// TIA Portal V17 export
// export: Created 2025-07-01T14:26:11.8460779Z, ExportSetting WithDefaults, DisplayName Totally Integrated Automation Portal, DisplayVersion V17 Update 8, DisplayName TIA Portal Openness, DisplayVersion V17 Update 8, DisplayName TIA Portal Version Control Interface, DisplayVersion V17, DisplayName SINAMICS Startdrive Advanced, DisplayVersion V17 SP2, DisplayName SINAMICS Startdrive G110M, G120, G120C, G120D, G120P, G115D, DisplayVersion V17 SP2, DisplayName SINAMICS Startdrive G130, G150, S120, S150, SINAMICS MV, S210, DisplayVersion V17 SP2, DisplayName STEP 7 Professional, DisplayVersion V17 Update 8, DisplayName SINUMERIK ONE STEP 7 Toolbox, DisplayVersion V17 Update 12, DisplayName SINUMERIK ONE PLC Basic Program Plus, DisplayVersion V17 Update 12, DisplayName SINUMERIK 840D sl STEP 7 Toolbox, DisplayVersion V17 Update 12, DisplayName STEP 7 Safety, DisplayVersion V17 Update 6, DisplayName WinCC Advanced, DisplayVersion V17 Update 8
FUNCTION "FC16013_METHOD_CALLS_U2_STA2_MEAS" : Void   // FC16013, LAD
{ S7_Optimized_Access := 'FALSE' }
VERSION : 0.1
// STATUS VALUES:
// 0 = IDLE
// 1 = CALIBRATING
// 2 = ANALYZING 
// -1 = ERROR
// stored: AutoNumber false, IsIECCheckEnabled false, SetENOAutomatically false, UDAEnableTagReadback false
   VAR_TEMP
      AUX_WSTRING_PART_ID_STA2 : WString;
      AUX_WCHARS : Array[0..63] of WChar;
      index : Int;
      ALARM_AUX : Bool;
      STATUS_BLKMOV : Int;   // STATUS BLKMOV
      ZERO : Int;
   END_VAR
   VAR CONSTANT
      VERSIONS_MAJOR : UInt := 2;
      VERSIONS_MINOR : UInt;
      FC_NUMBER : DInt := 16013;
   END_VAR
   VAR_TEMP   // added for the SCL form of the ladder/FBD networks
      _w1 : Bool;
      _w2 : Bool;
      _w3 : Bool;
      _w4 : Bool;
   END_VAR
BEGIN

REGION Network 1: ZERO
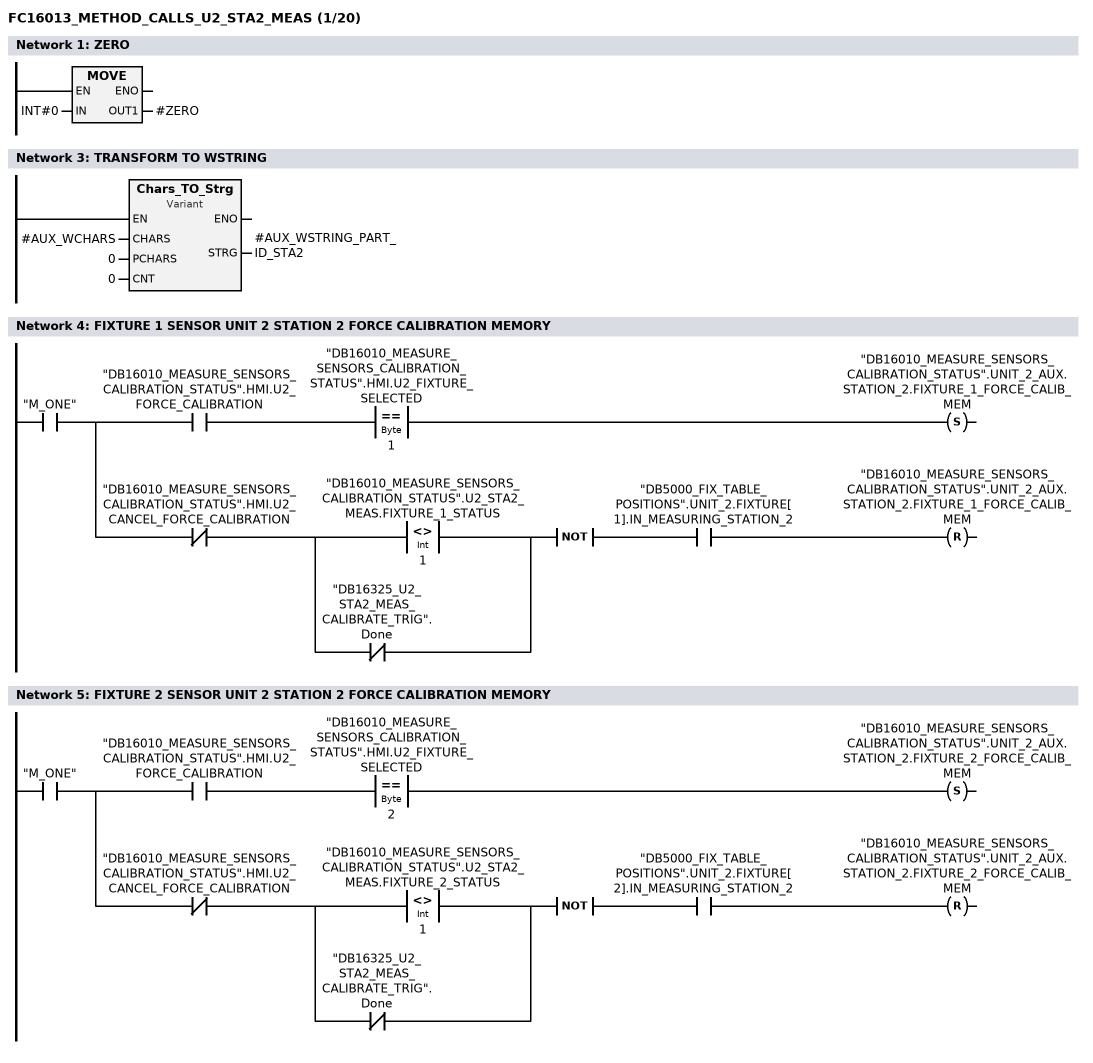
   RUNG wire#powerrail
      { S7_GenerateENO := "TRUE" } Move(in := INT#0, out1 => #ZERO)
   END_RUNG
   // the same network as SCL:
   #ZERO := INT#0;
END_REGION

REGION Network 2 (SCL): TRANSFORM TO WCHARS
   FOR #index := 0 TO 63 DO
       #AUX_WCHARS[#index] := CHAR_TO_WCHAR("DB8000_PART_STATUS".UNIT_2.STATION_2.PART_A.PART_ID[#index]);
   END_FOR;
END_REGION

REGION Network 3: TRANSFORM TO WSTRING
   RUNG wire#powerrail
      { S7_Templates := "[ptr_type := Variant, str_type := WString]" } Chars_TO_Strg(Chars := #AUX_WCHARS, pChars := 0, Cnt := 0, Strg => #AUX_WSTRING_PART_ID_STA2)
   END_RUNG
   // the same network as SCL:
   Chars_TO_Strg(Chars := #AUX_WCHARS, pChars := 0, Cnt := 0, Strg => #AUX_WSTRING_PART_ID_STA2);
END_REGION

REGION Network 4: FIXTURE 1 SENSOR UNIT 2 STATION 2 FORCE CALIBRATION MEMORY
   RUNG wire#powerrail
      Contact( "M_ONE" )
      wire#w1
      Contact( "DB16010_MEASURE_SENSORS_CALIBRATION_STATUS".HMI.U2_FORCE_CALIBRATION )
      { S7_Templates := "SrcType := Byte" } EQ_Contact(in1 := "DB16010_MEASURE_SENSORS_CALIBRATION_STATUS".HMI.U2_FIXTURE_SELECTED, in2 := 1)
      S_Coil( "DB16010_MEASURE_SENSORS_CALIBRATION_STATUS".UNIT_2_AUX.STATION_2.FIXTURE_1_FORCE_CALIB_MEM )
   END_RUNG
   RUNG wire#w1
      I_Contact( "DB16010_MEASURE_SENSORS_CALIBRATION_STATUS".HMI.U2_CANCEL_FORCE_CALIBRATION )
      wire#w2
      { S7_Templates := "SrcType := Int" } NE_Contact(in1 := "DB16010_MEASURE_SENSORS_CALIBRATION_STATUS".U2_STA2_MEAS.FIXTURE_1_STATUS, in2 := 1)
      wire#w3
      Not()
      Contact( "DB5000_FIX_TABLE_POSITIONS".UNIT_2.FIXTURE[1].IN_MEASURING_STATION_2 )
      R_Coil( "DB16010_MEASURE_SENSORS_CALIBRATION_STATUS".UNIT_2_AUX.STATION_2.FIXTURE_1_FORCE_CALIB_MEM )
   END_RUNG
   RUNG wire#w2
      I_Contact( "DB16325_U2_STA2_MEAS_CALIBRATE_TRIG".Done )
   END_RUNG wire#w3
   // the same network as SCL:
   IF "M_ONE" AND "DB16010_MEASURE_SENSORS_CALIBRATION_STATUS".HMI.U2_FORCE_CALIBRATION AND ("DB16010_MEASURE_SENSORS_CALIBRATION_STATUS".HMI.U2_FIXTURE_SELECTED = 1) THEN
       "DB16010_MEASURE_SENSORS_CALIBRATION_STATUS".UNIT_2_AUX.STATION_2.FIXTURE_1_FORCE_CALIB_MEM := TRUE;
   END_IF;
   IF NOT ("M_ONE" AND NOT "DB16010_MEASURE_SENSORS_CALIBRATION_STATUS".HMI.U2_CANCEL_FORCE_CALIBRATION AND (("DB16010_MEASURE_SENSORS_CALIBRATION_STATUS".U2_STA2_MEAS.FIXTURE_1_STATUS <> 1) OR NOT "DB16325_U2_STA2_MEAS_CALIBRATE_TRIG".Done)) AND "DB5000_FIX_TABLE_POSITIONS".UNIT_2.FIXTURE[1].IN_MEASURING_STATION_2 THEN
       "DB16010_MEASURE_SENSORS_CALIBRATION_STATUS".UNIT_2_AUX.STATION_2.FIXTURE_1_FORCE_CALIB_MEM := FALSE;
   END_IF;
END_REGION

REGION Network 5: FIXTURE 2 SENSOR UNIT 2 STATION 2 FORCE CALIBRATION MEMORY
   RUNG wire#powerrail
      Contact( "M_ONE" )
      wire#w1
      Contact( "DB16010_MEASURE_SENSORS_CALIBRATION_STATUS".HMI.U2_FORCE_CALIBRATION )
      { S7_Templates := "SrcType := Byte" } EQ_Contact(in1 := "DB16010_MEASURE_SENSORS_CALIBRATION_STATUS".HMI.U2_FIXTURE_SELECTED, in2 := 2)
      S_Coil( "DB16010_MEASURE_SENSORS_CALIBRATION_STATUS".UNIT_2_AUX.STATION_2.FIXTURE_2_FORCE_CALIB_MEM )
   END_RUNG
   RUNG wire#w1
      I_Contact( "DB16010_MEASURE_SENSORS_CALIBRATION_STATUS".HMI.U2_CANCEL_FORCE_CALIBRATION )
      wire#w2
      { S7_Templates := "SrcType := Int" } NE_Contact(in1 := "DB16010_MEASURE_SENSORS_CALIBRATION_STATUS".U2_STA2_MEAS.FIXTURE_2_STATUS, in2 := 1)
      wire#w3
      Not()
      Contact( "DB5000_FIX_TABLE_POSITIONS".UNIT_2.FIXTURE[2].IN_MEASURING_STATION_2 )
      R_Coil( "DB16010_MEASURE_SENSORS_CALIBRATION_STATUS".UNIT_2_AUX.STATION_2.FIXTURE_2_FORCE_CALIB_MEM )
   END_RUNG
   RUNG wire#w2
      I_Contact( "DB16325_U2_STA2_MEAS_CALIBRATE_TRIG".Done )
   END_RUNG wire#w3
   // the same network as SCL:
   IF "M_ONE" AND "DB16010_MEASURE_SENSORS_CALIBRATION_STATUS".HMI.U2_FORCE_CALIBRATION AND ("DB16010_MEASURE_SENSORS_CALIBRATION_STATUS".HMI.U2_FIXTURE_SELECTED = 2) THEN
       "DB16010_MEASURE_SENSORS_CALIBRATION_STATUS".UNIT_2_AUX.STATION_2.FIXTURE_2_FORCE_CALIB_MEM := TRUE;
   END_IF;
   IF NOT ("M_ONE" AND NOT "DB16010_MEASURE_SENSORS_CALIBRATION_STATUS".HMI.U2_CANCEL_FORCE_CALIBRATION AND (("DB16010_MEASURE_SENSORS_CALIBRATION_STATUS".U2_STA2_MEAS.FIXTURE_2_STATUS <> 1) OR NOT "DB16325_U2_STA2_MEAS_CALIBRATE_TRIG".Done)) AND "DB5000_FIX_TABLE_POSITIONS".UNIT_2.FIXTURE[2].IN_MEASURING_STATION_2 THEN
       "DB16010_MEASURE_SENSORS_CALIBRATION_STATUS".UNIT_2_AUX.STATION_2.FIXTURE_2_FORCE_CALIB_MEM := FALSE;
   END_IF;
END_REGION

REGION Network 6: FIXTURE 3 SENSOR UNIT 2 STATION 2 FORCE CALIBRATION MEMORY
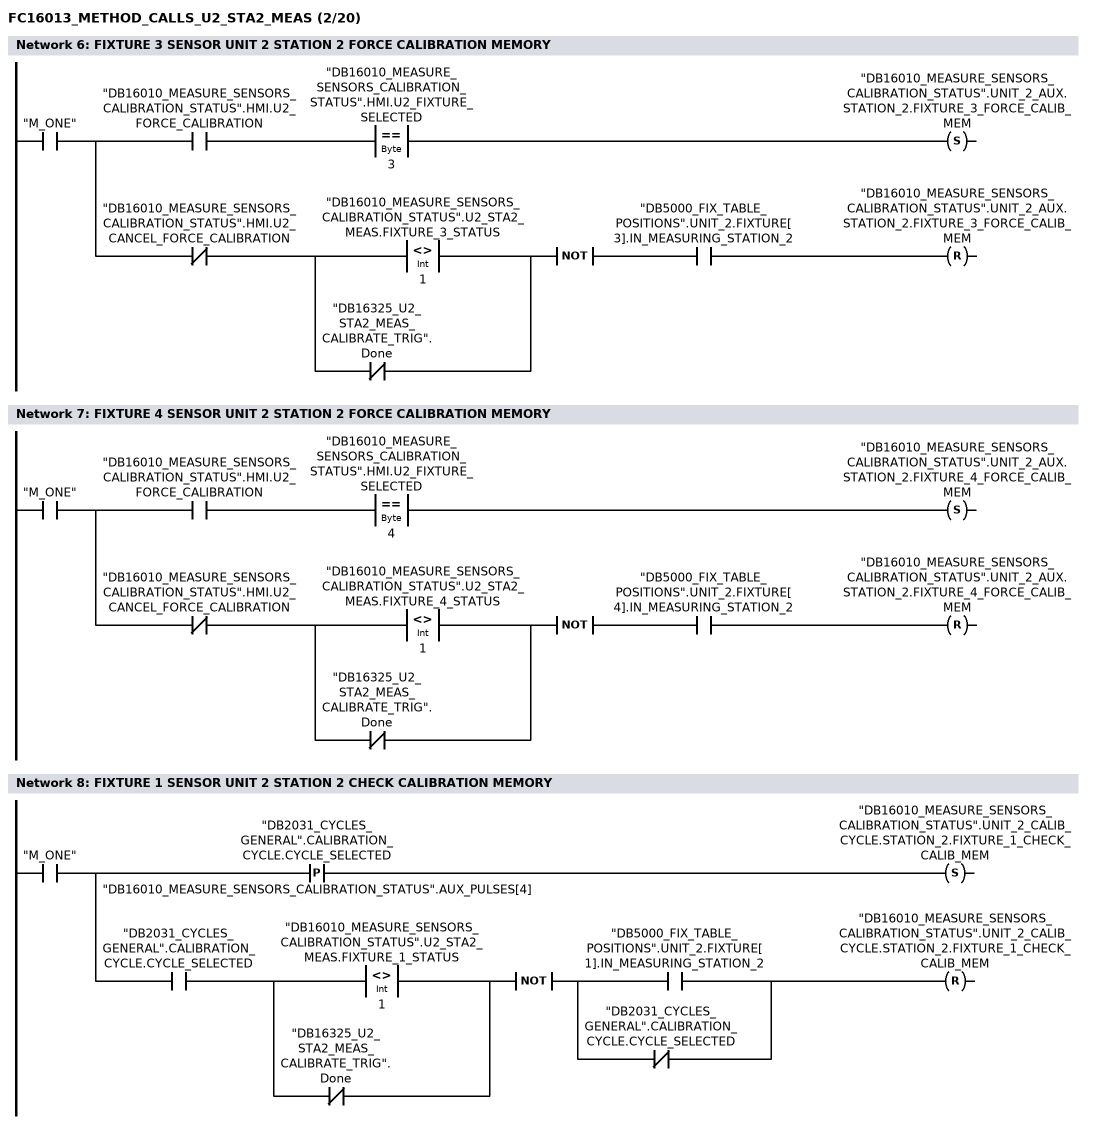
   RUNG wire#powerrail
      Contact( "M_ONE" )
      wire#w1
      Contact( "DB16010_MEASURE_SENSORS_CALIBRATION_STATUS".HMI.U2_FORCE_CALIBRATION )
      { S7_Templates := "SrcType := Byte" } EQ_Contact(in1 := "DB16010_MEASURE_SENSORS_CALIBRATION_STATUS".HMI.U2_FIXTURE_SELECTED, in2 := 3)
      S_Coil( "DB16010_MEASURE_SENSORS_CALIBRATION_STATUS".UNIT_2_AUX.STATION_2.FIXTURE_3_FORCE_CALIB_MEM )
   END_RUNG
   RUNG wire#w1
      I_Contact( "DB16010_MEASURE_SENSORS_CALIBRATION_STATUS".HMI.U2_CANCEL_FORCE_CALIBRATION )
      wire#w2
      { S7_Templates := "SrcType := Int" } NE_Contact(in1 := "DB16010_MEASURE_SENSORS_CALIBRATION_STATUS".U2_STA2_MEAS.FIXTURE_3_STATUS, in2 := 1)
      wire#w3
      Not()
      Contact( "DB5000_FIX_TABLE_POSITIONS".UNIT_2.FIXTURE[3].IN_MEASURING_STATION_2 )
      R_Coil( "DB16010_MEASURE_SENSORS_CALIBRATION_STATUS".UNIT_2_AUX.STATION_2.FIXTURE_3_FORCE_CALIB_MEM )
   END_RUNG
   RUNG wire#w2
      I_Contact( "DB16325_U2_STA2_MEAS_CALIBRATE_TRIG".Done )
   END_RUNG wire#w3
   // the same network as SCL:
   IF "M_ONE" AND "DB16010_MEASURE_SENSORS_CALIBRATION_STATUS".HMI.U2_FORCE_CALIBRATION AND ("DB16010_MEASURE_SENSORS_CALIBRATION_STATUS".HMI.U2_FIXTURE_SELECTED = 3) THEN
       "DB16010_MEASURE_SENSORS_CALIBRATION_STATUS".UNIT_2_AUX.STATION_2.FIXTURE_3_FORCE_CALIB_MEM := TRUE;
   END_IF;
   IF NOT ("M_ONE" AND NOT "DB16010_MEASURE_SENSORS_CALIBRATION_STATUS".HMI.U2_CANCEL_FORCE_CALIBRATION AND (("DB16010_MEASURE_SENSORS_CALIBRATION_STATUS".U2_STA2_MEAS.FIXTURE_3_STATUS <> 1) OR NOT "DB16325_U2_STA2_MEAS_CALIBRATE_TRIG".Done)) AND "DB5000_FIX_TABLE_POSITIONS".UNIT_2.FIXTURE[3].IN_MEASURING_STATION_2 THEN
       "DB16010_MEASURE_SENSORS_CALIBRATION_STATUS".UNIT_2_AUX.STATION_2.FIXTURE_3_FORCE_CALIB_MEM := FALSE;
   END_IF;
END_REGION

REGION Network 7: FIXTURE 4 SENSOR UNIT 2 STATION 2 FORCE CALIBRATION MEMORY
   RUNG wire#powerrail
      Contact( "M_ONE" )
      wire#w1
      Contact( "DB16010_MEASURE_SENSORS_CALIBRATION_STATUS".HMI.U2_FORCE_CALIBRATION )
      { S7_Templates := "SrcType := Byte" } EQ_Contact(in1 := "DB16010_MEASURE_SENSORS_CALIBRATION_STATUS".HMI.U2_FIXTURE_SELECTED, in2 := 4)
      S_Coil( "DB16010_MEASURE_SENSORS_CALIBRATION_STATUS".UNIT_2_AUX.STATION_2.FIXTURE_4_FORCE_CALIB_MEM )
   END_RUNG
   RUNG wire#w1
      I_Contact( "DB16010_MEASURE_SENSORS_CALIBRATION_STATUS".HMI.U2_CANCEL_FORCE_CALIBRATION )
      wire#w2
      { S7_Templates := "SrcType := Int" } NE_Contact(in1 := "DB16010_MEASURE_SENSORS_CALIBRATION_STATUS".U2_STA2_MEAS.FIXTURE_4_STATUS, in2 := 1)
      wire#w3
      Not()
      Contact( "DB5000_FIX_TABLE_POSITIONS".UNIT_2.FIXTURE[4].IN_MEASURING_STATION_2 )
      R_Coil( "DB16010_MEASURE_SENSORS_CALIBRATION_STATUS".UNIT_2_AUX.STATION_2.FIXTURE_4_FORCE_CALIB_MEM )
   END_RUNG
   RUNG wire#w2
      I_Contact( "DB16325_U2_STA2_MEAS_CALIBRATE_TRIG".Done )
   END_RUNG wire#w3
   // the same network as SCL:
   IF "M_ONE" AND "DB16010_MEASURE_SENSORS_CALIBRATION_STATUS".HMI.U2_FORCE_CALIBRATION AND ("DB16010_MEASURE_SENSORS_CALIBRATION_STATUS".HMI.U2_FIXTURE_SELECTED = 4) THEN
       "DB16010_MEASURE_SENSORS_CALIBRATION_STATUS".UNIT_2_AUX.STATION_2.FIXTURE_4_FORCE_CALIB_MEM := TRUE;
   END_IF;
   IF NOT ("M_ONE" AND NOT "DB16010_MEASURE_SENSORS_CALIBRATION_STATUS".HMI.U2_CANCEL_FORCE_CALIBRATION AND (("DB16010_MEASURE_SENSORS_CALIBRATION_STATUS".U2_STA2_MEAS.FIXTURE_4_STATUS <> 1) OR NOT "DB16325_U2_STA2_MEAS_CALIBRATE_TRIG".Done)) AND "DB5000_FIX_TABLE_POSITIONS".UNIT_2.FIXTURE[4].IN_MEASURING_STATION_2 THEN
       "DB16010_MEASURE_SENSORS_CALIBRATION_STATUS".UNIT_2_AUX.STATION_2.FIXTURE_4_FORCE_CALIB_MEM := FALSE;
   END_IF;
END_REGION

REGION Network 8: FIXTURE 1 SENSOR UNIT 2 STATION 2 CHECK CALIBRATION MEMORY
   RUNG wire#powerrail
      Contact( "M_ONE" )
      wire#w1
      P_Contact(operand := "DB2031_CYCLES_GENERAL".CALIBRATION_CYCLE.CYCLE_SELECTED, bit := "DB16010_MEASURE_SENSORS_CALIBRATION_STATUS".AUX_PULSES[4])
      S_Coil( "DB16010_MEASURE_SENSORS_CALIBRATION_STATUS".UNIT_2_CALIB_CYCLE.STATION_2.FIXTURE_1_CHECK_CALIB_MEM )
   END_RUNG
   RUNG wire#w1
      Contact( "DB2031_CYCLES_GENERAL".CALIBRATION_CYCLE.CYCLE_SELECTED )
      wire#w2
      { S7_Templates := "SrcType := Int" } NE_Contact(in1 := "DB16010_MEASURE_SENSORS_CALIBRATION_STATUS".U2_STA2_MEAS.FIXTURE_1_STATUS, in2 := 1)
      wire#w3
      Not()
      wire#w4
      Contact( "DB5000_FIX_TABLE_POSITIONS".UNIT_2.FIXTURE[1].IN_MEASURING_STATION_2 )
      wire#w5
      R_Coil( "DB16010_MEASURE_SENSORS_CALIBRATION_STATUS".UNIT_2_CALIB_CYCLE.STATION_2.FIXTURE_1_CHECK_CALIB_MEM )
   END_RUNG
   RUNG wire#w2
      I_Contact( "DB16325_U2_STA2_MEAS_CALIBRATE_TRIG".Done )
   END_RUNG wire#w3
   RUNG wire#w4
      I_Contact( "DB2031_CYCLES_GENERAL".CALIBRATION_CYCLE.CYCLE_SELECTED )
   END_RUNG wire#w5
   // the same network as SCL:
   #_w1 := "M_ONE" AND "DB2031_CYCLES_GENERAL".CALIBRATION_CYCLE.CYCLE_SELECTED AND NOT "DB16010_MEASURE_SENSORS_CALIBRATION_STATUS".AUX_PULSES[4];   // rising edge of "DB2031_CYCLES_GENERAL".CALIBRATION_CYCLE.CYCLE_SELECTED
   "DB16010_MEASURE_SENSORS_CALIBRATION_STATUS".AUX_PULSES[4] := "DB2031_CYCLES_GENERAL".CALIBRATION_CYCLE.CYCLE_SELECTED;
   IF #_w1 THEN
       "DB16010_MEASURE_SENSORS_CALIBRATION_STATUS".UNIT_2_CALIB_CYCLE.STATION_2.FIXTURE_1_CHECK_CALIB_MEM := TRUE;
   END_IF;
   IF NOT ("M_ONE" AND "DB2031_CYCLES_GENERAL".CALIBRATION_CYCLE.CYCLE_SELECTED AND (("DB16010_MEASURE_SENSORS_CALIBRATION_STATUS".U2_STA2_MEAS.FIXTURE_1_STATUS <> 1) OR NOT "DB16325_U2_STA2_MEAS_CALIBRATE_TRIG".Done)) AND ("DB5000_FIX_TABLE_POSITIONS".UNIT_2.FIXTURE[1].IN_MEASURING_STATION_2 OR NOT "DB2031_CYCLES_GENERAL".CALIBRATION_CYCLE.CYCLE_SELECTED) THEN
       "DB16010_MEASURE_SENSORS_CALIBRATION_STATUS".UNIT_2_CALIB_CYCLE.STATION_2.FIXTURE_1_CHECK_CALIB_MEM := FALSE;
   END_IF;
END_REGION

REGION Network 9: FIXTURE 2 SENSOR UNIT 2 STATION 2 CHECK CALIBRATION MEMORY
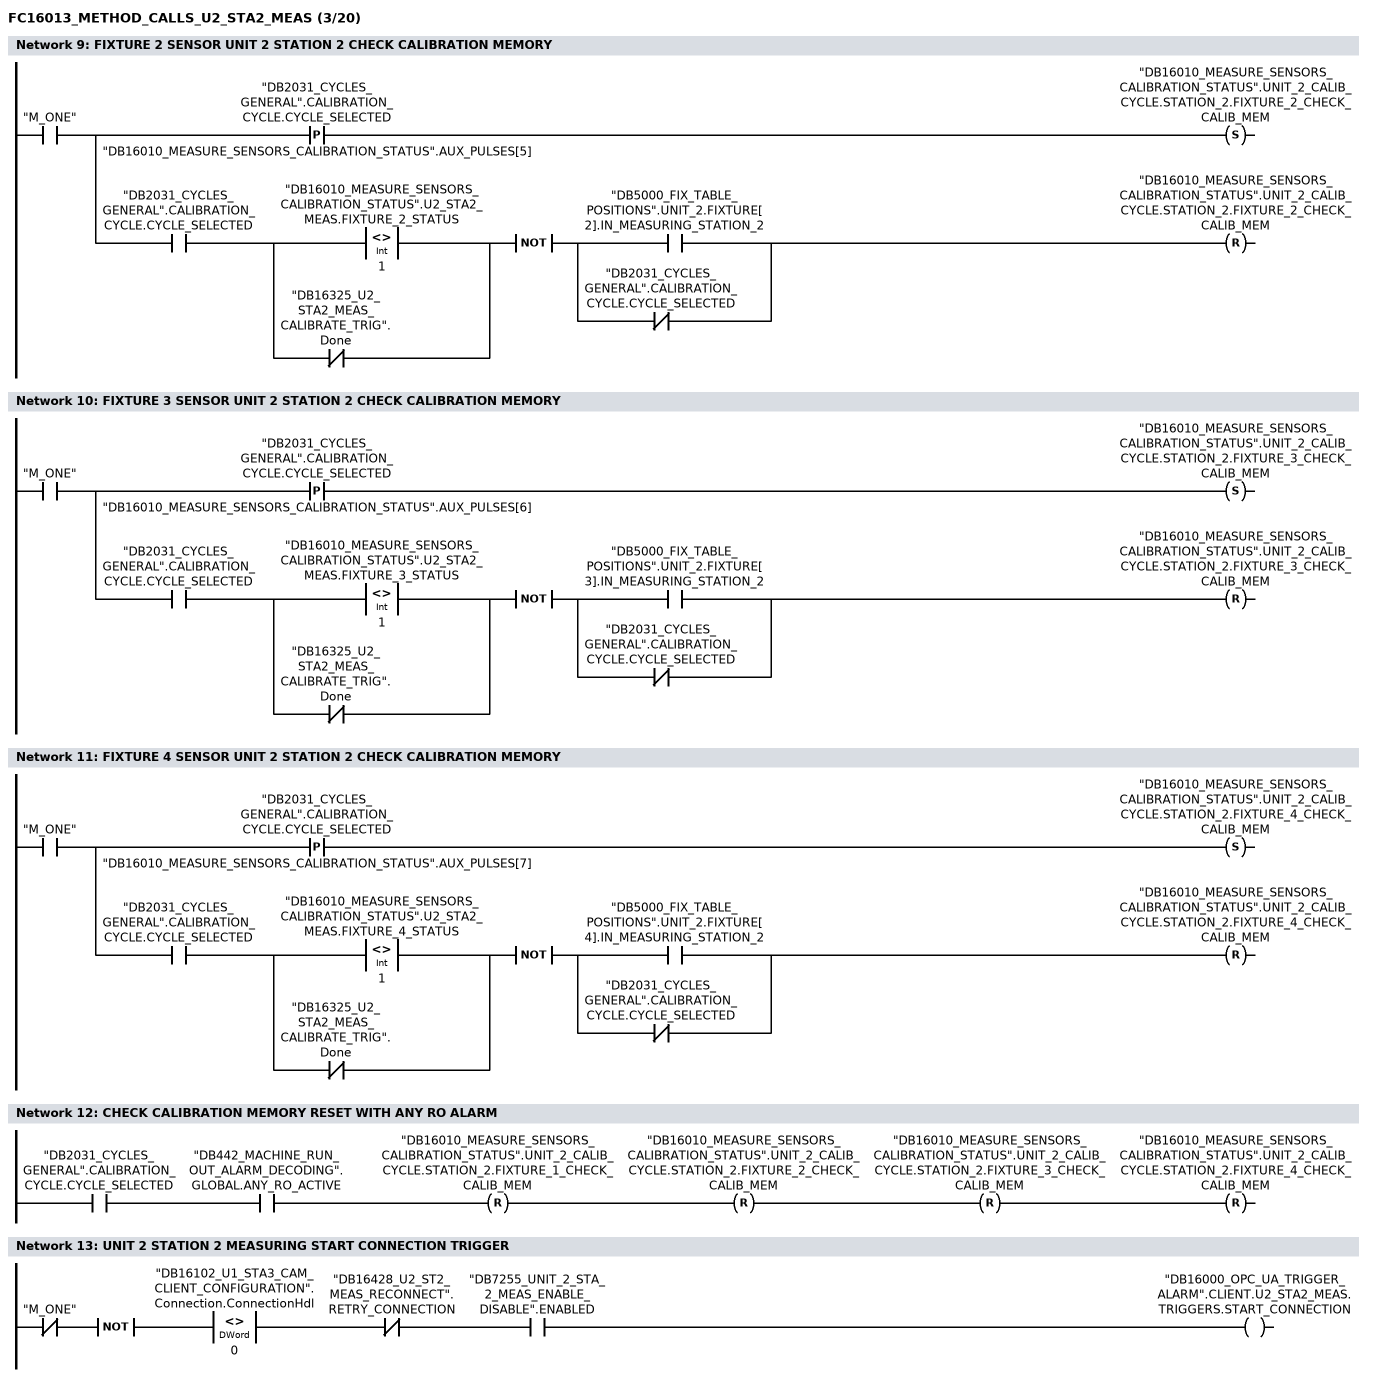
   RUNG wire#powerrail
      Contact( "M_ONE" )
      wire#w1
      P_Contact(operand := "DB2031_CYCLES_GENERAL".CALIBRATION_CYCLE.CYCLE_SELECTED, bit := "DB16010_MEASURE_SENSORS_CALIBRATION_STATUS".AUX_PULSES[5])
      S_Coil( "DB16010_MEASURE_SENSORS_CALIBRATION_STATUS".UNIT_2_CALIB_CYCLE.STATION_2.FIXTURE_2_CHECK_CALIB_MEM )
   END_RUNG
   RUNG wire#w1
      Contact( "DB2031_CYCLES_GENERAL".CALIBRATION_CYCLE.CYCLE_SELECTED )
      wire#w2
      { S7_Templates := "SrcType := Int" } NE_Contact(in1 := "DB16010_MEASURE_SENSORS_CALIBRATION_STATUS".U2_STA2_MEAS.FIXTURE_2_STATUS, in2 := 1)
      wire#w3
      Not()
      wire#w4
      Contact( "DB5000_FIX_TABLE_POSITIONS".UNIT_2.FIXTURE[2].IN_MEASURING_STATION_2 )
      wire#w5
      R_Coil( "DB16010_MEASURE_SENSORS_CALIBRATION_STATUS".UNIT_2_CALIB_CYCLE.STATION_2.FIXTURE_2_CHECK_CALIB_MEM )
   END_RUNG
   RUNG wire#w2
      I_Contact( "DB16325_U2_STA2_MEAS_CALIBRATE_TRIG".Done )
   END_RUNG wire#w3
   RUNG wire#w4
      I_Contact( "DB2031_CYCLES_GENERAL".CALIBRATION_CYCLE.CYCLE_SELECTED )
   END_RUNG wire#w5
   // the same network as SCL:
   #_w1 := "M_ONE" AND "DB2031_CYCLES_GENERAL".CALIBRATION_CYCLE.CYCLE_SELECTED AND NOT "DB16010_MEASURE_SENSORS_CALIBRATION_STATUS".AUX_PULSES[5];   // rising edge of "DB2031_CYCLES_GENERAL".CALIBRATION_CYCLE.CYCLE_SELECTED
   "DB16010_MEASURE_SENSORS_CALIBRATION_STATUS".AUX_PULSES[5] := "DB2031_CYCLES_GENERAL".CALIBRATION_CYCLE.CYCLE_SELECTED;
   IF #_w1 THEN
       "DB16010_MEASURE_SENSORS_CALIBRATION_STATUS".UNIT_2_CALIB_CYCLE.STATION_2.FIXTURE_2_CHECK_CALIB_MEM := TRUE;
   END_IF;
   IF NOT ("M_ONE" AND "DB2031_CYCLES_GENERAL".CALIBRATION_CYCLE.CYCLE_SELECTED AND (("DB16010_MEASURE_SENSORS_CALIBRATION_STATUS".U2_STA2_MEAS.FIXTURE_2_STATUS <> 1) OR NOT "DB16325_U2_STA2_MEAS_CALIBRATE_TRIG".Done)) AND ("DB5000_FIX_TABLE_POSITIONS".UNIT_2.FIXTURE[2].IN_MEASURING_STATION_2 OR NOT "DB2031_CYCLES_GENERAL".CALIBRATION_CYCLE.CYCLE_SELECTED) THEN
       "DB16010_MEASURE_SENSORS_CALIBRATION_STATUS".UNIT_2_CALIB_CYCLE.STATION_2.FIXTURE_2_CHECK_CALIB_MEM := FALSE;
   END_IF;
END_REGION

REGION Network 10: FIXTURE 3 SENSOR UNIT 2 STATION 2 CHECK CALIBRATION MEMORY
   RUNG wire#powerrail
      Contact( "M_ONE" )
      wire#w1
      P_Contact(operand := "DB2031_CYCLES_GENERAL".CALIBRATION_CYCLE.CYCLE_SELECTED, bit := "DB16010_MEASURE_SENSORS_CALIBRATION_STATUS".AUX_PULSES[6])
      S_Coil( "DB16010_MEASURE_SENSORS_CALIBRATION_STATUS".UNIT_2_CALIB_CYCLE.STATION_2.FIXTURE_3_CHECK_CALIB_MEM )
   END_RUNG
   RUNG wire#w1
      Contact( "DB2031_CYCLES_GENERAL".CALIBRATION_CYCLE.CYCLE_SELECTED )
      wire#w2
      { S7_Templates := "SrcType := Int" } NE_Contact(in1 := "DB16010_MEASURE_SENSORS_CALIBRATION_STATUS".U2_STA2_MEAS.FIXTURE_3_STATUS, in2 := 1)
      wire#w3
      Not()
      wire#w4
      Contact( "DB5000_FIX_TABLE_POSITIONS".UNIT_2.FIXTURE[3].IN_MEASURING_STATION_2 )
      wire#w5
      R_Coil( "DB16010_MEASURE_SENSORS_CALIBRATION_STATUS".UNIT_2_CALIB_CYCLE.STATION_2.FIXTURE_3_CHECK_CALIB_MEM )
   END_RUNG
   RUNG wire#w2
      I_Contact( "DB16325_U2_STA2_MEAS_CALIBRATE_TRIG".Done )
   END_RUNG wire#w3
   RUNG wire#w4
      I_Contact( "DB2031_CYCLES_GENERAL".CALIBRATION_CYCLE.CYCLE_SELECTED )
   END_RUNG wire#w5
   // the same network as SCL:
   #_w1 := "M_ONE" AND "DB2031_CYCLES_GENERAL".CALIBRATION_CYCLE.CYCLE_SELECTED AND NOT "DB16010_MEASURE_SENSORS_CALIBRATION_STATUS".AUX_PULSES[6];   // rising edge of "DB2031_CYCLES_GENERAL".CALIBRATION_CYCLE.CYCLE_SELECTED
   "DB16010_MEASURE_SENSORS_CALIBRATION_STATUS".AUX_PULSES[6] := "DB2031_CYCLES_GENERAL".CALIBRATION_CYCLE.CYCLE_SELECTED;
   IF #_w1 THEN
       "DB16010_MEASURE_SENSORS_CALIBRATION_STATUS".UNIT_2_CALIB_CYCLE.STATION_2.FIXTURE_3_CHECK_CALIB_MEM := TRUE;
   END_IF;
   IF NOT ("M_ONE" AND "DB2031_CYCLES_GENERAL".CALIBRATION_CYCLE.CYCLE_SELECTED AND (("DB16010_MEASURE_SENSORS_CALIBRATION_STATUS".U2_STA2_MEAS.FIXTURE_3_STATUS <> 1) OR NOT "DB16325_U2_STA2_MEAS_CALIBRATE_TRIG".Done)) AND ("DB5000_FIX_TABLE_POSITIONS".UNIT_2.FIXTURE[3].IN_MEASURING_STATION_2 OR NOT "DB2031_CYCLES_GENERAL".CALIBRATION_CYCLE.CYCLE_SELECTED) THEN
       "DB16010_MEASURE_SENSORS_CALIBRATION_STATUS".UNIT_2_CALIB_CYCLE.STATION_2.FIXTURE_3_CHECK_CALIB_MEM := FALSE;
   END_IF;
END_REGION

REGION Network 11: FIXTURE 4 SENSOR UNIT 2 STATION 2 CHECK CALIBRATION MEMORY
   RUNG wire#powerrail
      Contact( "M_ONE" )
      wire#w1
      P_Contact(operand := "DB2031_CYCLES_GENERAL".CALIBRATION_CYCLE.CYCLE_SELECTED, bit := "DB16010_MEASURE_SENSORS_CALIBRATION_STATUS".AUX_PULSES[7])
      S_Coil( "DB16010_MEASURE_SENSORS_CALIBRATION_STATUS".UNIT_2_CALIB_CYCLE.STATION_2.FIXTURE_4_CHECK_CALIB_MEM )
   END_RUNG
   RUNG wire#w1
      Contact( "DB2031_CYCLES_GENERAL".CALIBRATION_CYCLE.CYCLE_SELECTED )
      wire#w2
      { S7_Templates := "SrcType := Int" } NE_Contact(in1 := "DB16010_MEASURE_SENSORS_CALIBRATION_STATUS".U2_STA2_MEAS.FIXTURE_4_STATUS, in2 := 1)
      wire#w3
      Not()
      wire#w4
      Contact( "DB5000_FIX_TABLE_POSITIONS".UNIT_2.FIXTURE[4].IN_MEASURING_STATION_2 )
      wire#w5
      R_Coil( "DB16010_MEASURE_SENSORS_CALIBRATION_STATUS".UNIT_2_CALIB_CYCLE.STATION_2.FIXTURE_4_CHECK_CALIB_MEM )
   END_RUNG
   RUNG wire#w2
      I_Contact( "DB16325_U2_STA2_MEAS_CALIBRATE_TRIG".Done )
   END_RUNG wire#w3
   RUNG wire#w4
      I_Contact( "DB2031_CYCLES_GENERAL".CALIBRATION_CYCLE.CYCLE_SELECTED )
   END_RUNG wire#w5
   // the same network as SCL:
   #_w1 := "M_ONE" AND "DB2031_CYCLES_GENERAL".CALIBRATION_CYCLE.CYCLE_SELECTED AND NOT "DB16010_MEASURE_SENSORS_CALIBRATION_STATUS".AUX_PULSES[7];   // rising edge of "DB2031_CYCLES_GENERAL".CALIBRATION_CYCLE.CYCLE_SELECTED
   "DB16010_MEASURE_SENSORS_CALIBRATION_STATUS".AUX_PULSES[7] := "DB2031_CYCLES_GENERAL".CALIBRATION_CYCLE.CYCLE_SELECTED;
   IF #_w1 THEN
       "DB16010_MEASURE_SENSORS_CALIBRATION_STATUS".UNIT_2_CALIB_CYCLE.STATION_2.FIXTURE_4_CHECK_CALIB_MEM := TRUE;
   END_IF;
   IF NOT ("M_ONE" AND "DB2031_CYCLES_GENERAL".CALIBRATION_CYCLE.CYCLE_SELECTED AND (("DB16010_MEASURE_SENSORS_CALIBRATION_STATUS".U2_STA2_MEAS.FIXTURE_4_STATUS <> 1) OR NOT "DB16325_U2_STA2_MEAS_CALIBRATE_TRIG".Done)) AND ("DB5000_FIX_TABLE_POSITIONS".UNIT_2.FIXTURE[4].IN_MEASURING_STATION_2 OR NOT "DB2031_CYCLES_GENERAL".CALIBRATION_CYCLE.CYCLE_SELECTED) THEN
       "DB16010_MEASURE_SENSORS_CALIBRATION_STATUS".UNIT_2_CALIB_CYCLE.STATION_2.FIXTURE_4_CHECK_CALIB_MEM := FALSE;
   END_IF;
END_REGION

REGION Network 12: CHECK CALIBRATION MEMORY RESET WITH ANY RO ALARM
   RUNG wire#powerrail
      Contact( "DB2031_CYCLES_GENERAL".CALIBRATION_CYCLE.CYCLE_SELECTED )
      Contact( "DB442_MACHINE_RUN_OUT_ALARM_DECODING".GLOBAL.ANY_RO_ACTIVE )
      R_Coil( "DB16010_MEASURE_SENSORS_CALIBRATION_STATUS".UNIT_2_CALIB_CYCLE.STATION_2.FIXTURE_1_CHECK_CALIB_MEM )
      R_Coil( "DB16010_MEASURE_SENSORS_CALIBRATION_STATUS".UNIT_2_CALIB_CYCLE.STATION_2.FIXTURE_2_CHECK_CALIB_MEM )
      R_Coil( "DB16010_MEASURE_SENSORS_CALIBRATION_STATUS".UNIT_2_CALIB_CYCLE.STATION_2.FIXTURE_3_CHECK_CALIB_MEM )
      R_Coil( "DB16010_MEASURE_SENSORS_CALIBRATION_STATUS".UNIT_2_CALIB_CYCLE.STATION_2.FIXTURE_4_CHECK_CALIB_MEM )
   END_RUNG
   // the same network as SCL:
   IF "DB2031_CYCLES_GENERAL".CALIBRATION_CYCLE.CYCLE_SELECTED AND "DB442_MACHINE_RUN_OUT_ALARM_DECODING".GLOBAL.ANY_RO_ACTIVE THEN
       "DB16010_MEASURE_SENSORS_CALIBRATION_STATUS".UNIT_2_CALIB_CYCLE.STATION_2.FIXTURE_1_CHECK_CALIB_MEM := FALSE;
       "DB16010_MEASURE_SENSORS_CALIBRATION_STATUS".UNIT_2_CALIB_CYCLE.STATION_2.FIXTURE_2_CHECK_CALIB_MEM := FALSE;
       "DB16010_MEASURE_SENSORS_CALIBRATION_STATUS".UNIT_2_CALIB_CYCLE.STATION_2.FIXTURE_3_CHECK_CALIB_MEM := FALSE;
       "DB16010_MEASURE_SENSORS_CALIBRATION_STATUS".UNIT_2_CALIB_CYCLE.STATION_2.FIXTURE_4_CHECK_CALIB_MEM := FALSE;
   END_IF;
END_REGION

REGION Network 13: UNIT 2 STATION 2 MEASURING START CONNECTION TRIGGER
   RUNG wire#powerrail
      I_Contact( "M_ONE" )
      Not()
      { S7_Templates := "SrcType := DWord" } NE_Contact(in1 := "DB16102_U1_STA3_CAM_CLIENT_CONFIGURATION".Connection.ConnectionHdl, in2 := 0)
      I_Contact( "DB16428_U2_ST2_MEAS_RECONNECT".RETRY_CONNECTION )
      Contact( "DB7255_UNIT_2_STA_2_MEAS_ENABLE_DISABLE".ENABLED )
      Coil( "DB16000_OPC_UA_TRIGGER_ALARM".CLIENT.U2_STA2_MEAS.TRIGGERS.START_CONNECTION )
   END_RUNG
   // the same network as SCL:
   "DB16000_OPC_UA_TRIGGER_ALARM".CLIENT.U2_STA2_MEAS.TRIGGERS.START_CONNECTION := NOT (NOT "M_ONE") AND ("DB16102_U1_STA3_CAM_CLIENT_CONFIGURATION".Connection.ConnectionHdl <> 0) AND NOT "DB16428_U2_ST2_MEAS_RECONNECT".RETRY_CONNECTION AND "DB7255_UNIT_2_STA_2_MEAS_ENABLE_DISABLE".ENABLED;
END_REGION

REGION Network 14: UNIT 2 STATION 2 MEASURING GET INDEX LIST TRIGGER
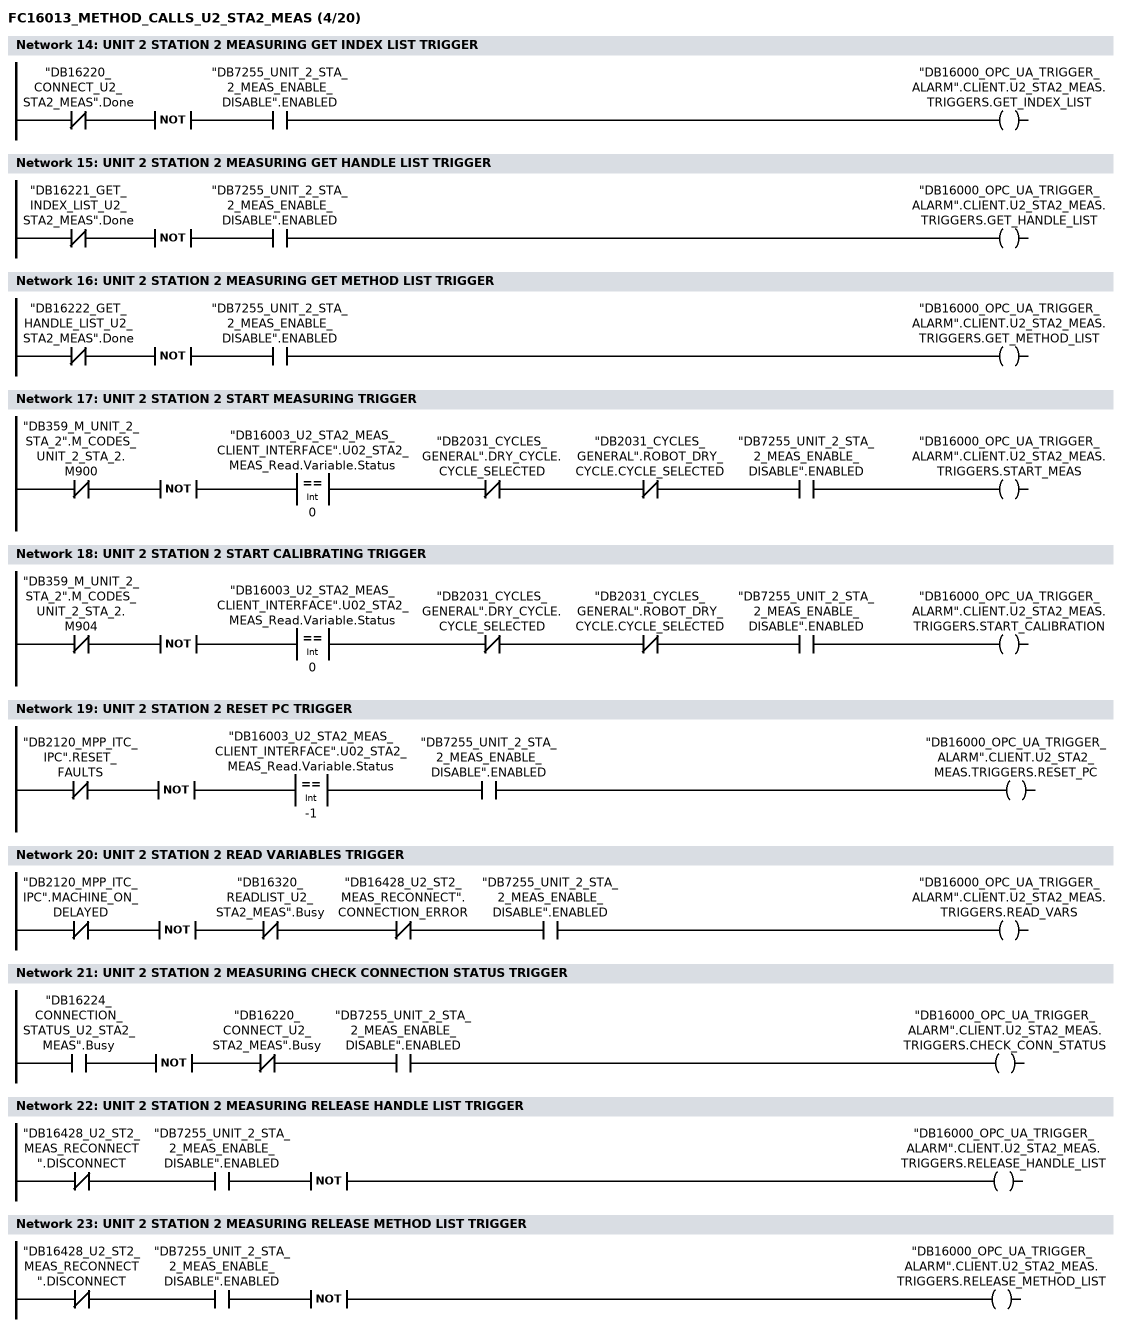
   RUNG wire#powerrail
      I_Contact( "DB16220_CONNECT_U2_STA2_MEAS".Done )
      Not()
      Contact( "DB7255_UNIT_2_STA_2_MEAS_ENABLE_DISABLE".ENABLED )
      Coil( "DB16000_OPC_UA_TRIGGER_ALARM".CLIENT.U2_STA2_MEAS.TRIGGERS.GET_INDEX_LIST )
   END_RUNG
   // the same network as SCL:
   "DB16000_OPC_UA_TRIGGER_ALARM".CLIENT.U2_STA2_MEAS.TRIGGERS.GET_INDEX_LIST := NOT (NOT "DB16220_CONNECT_U2_STA2_MEAS".Done) AND "DB7255_UNIT_2_STA_2_MEAS_ENABLE_DISABLE".ENABLED;
END_REGION

REGION Network 15: UNIT 2 STATION 2 MEASURING GET HANDLE LIST TRIGGER
   RUNG wire#powerrail
      I_Contact( "DB16221_GET_INDEX_LIST_U2_STA2_MEAS".Done )
      Not()
      Contact( "DB7255_UNIT_2_STA_2_MEAS_ENABLE_DISABLE".ENABLED )
      Coil( "DB16000_OPC_UA_TRIGGER_ALARM".CLIENT.U2_STA2_MEAS.TRIGGERS.GET_HANDLE_LIST )
   END_RUNG
   // the same network as SCL:
   "DB16000_OPC_UA_TRIGGER_ALARM".CLIENT.U2_STA2_MEAS.TRIGGERS.GET_HANDLE_LIST := NOT (NOT "DB16221_GET_INDEX_LIST_U2_STA2_MEAS".Done) AND "DB7255_UNIT_2_STA_2_MEAS_ENABLE_DISABLE".ENABLED;
END_REGION

REGION Network 16: UNIT 2 STATION 2 MEASURING GET METHOD LIST TRIGGER
   RUNG wire#powerrail
      I_Contact( "DB16222_GET_HANDLE_LIST_U2_STA2_MEAS".Done )
      Not()
      Contact( "DB7255_UNIT_2_STA_2_MEAS_ENABLE_DISABLE".ENABLED )
      Coil( "DB16000_OPC_UA_TRIGGER_ALARM".CLIENT.U2_STA2_MEAS.TRIGGERS.GET_METHOD_LIST )
   END_RUNG
   // the same network as SCL:
   "DB16000_OPC_UA_TRIGGER_ALARM".CLIENT.U2_STA2_MEAS.TRIGGERS.GET_METHOD_LIST := NOT (NOT "DB16222_GET_HANDLE_LIST_U2_STA2_MEAS".Done) AND "DB7255_UNIT_2_STA_2_MEAS_ENABLE_DISABLE".ENABLED;
END_REGION

REGION Network 17: UNIT 2 STATION 2 START MEASURING TRIGGER
   RUNG wire#powerrail
      I_Contact( "DB359_M_UNIT_2_STA_2".M_CODES_UNIT_2_STA_2.M900 )
      Not()
      { S7_Templates := "SrcType := Int" } EQ_Contact(in1 := "DB16003_U2_STA2_MEAS_CLIENT_INTERFACE".U02_STA2_MEAS_Read.Variable.Status, in2 := 0)
      I_Contact( "DB2031_CYCLES_GENERAL".DRY_CYCLE.CYCLE_SELECTED )
      I_Contact( "DB2031_CYCLES_GENERAL".ROBOT_DRY_CYCLE.CYCLE_SELECTED )
      Contact( "DB7255_UNIT_2_STA_2_MEAS_ENABLE_DISABLE".ENABLED )
      Coil( "DB16000_OPC_UA_TRIGGER_ALARM".CLIENT.U2_STA2_MEAS.TRIGGERS.START_MEAS )
   END_RUNG
   // the same network as SCL:
   "DB16000_OPC_UA_TRIGGER_ALARM".CLIENT.U2_STA2_MEAS.TRIGGERS.START_MEAS := NOT (NOT "DB359_M_UNIT_2_STA_2".M_CODES_UNIT_2_STA_2.M900) AND ("DB16003_U2_STA2_MEAS_CLIENT_INTERFACE".U02_STA2_MEAS_Read.Variable.Status = 0) AND NOT "DB2031_CYCLES_GENERAL".DRY_CYCLE.CYCLE_SELECTED AND NOT "DB2031_CYCLES_GENERAL".ROBOT_DRY_CYCLE.CYCLE_SELECTED AND "DB7255_UNIT_2_STA_2_MEAS_ENABLE_DISABLE".ENABLED;
END_REGION

REGION Network 18: UNIT 2 STATION 2 START CALIBRATING TRIGGER
   RUNG wire#powerrail
      I_Contact( "DB359_M_UNIT_2_STA_2".M_CODES_UNIT_2_STA_2.M904 )
      Not()
      { S7_Templates := "SrcType := Int" } EQ_Contact(in1 := "DB16003_U2_STA2_MEAS_CLIENT_INTERFACE".U02_STA2_MEAS_Read.Variable.Status, in2 := 0)
      I_Contact( "DB2031_CYCLES_GENERAL".DRY_CYCLE.CYCLE_SELECTED )
      I_Contact( "DB2031_CYCLES_GENERAL".ROBOT_DRY_CYCLE.CYCLE_SELECTED )
      Contact( "DB7255_UNIT_2_STA_2_MEAS_ENABLE_DISABLE".ENABLED )
      Coil( "DB16000_OPC_UA_TRIGGER_ALARM".CLIENT.U2_STA2_MEAS.TRIGGERS.START_CALIBRATION )
   END_RUNG
   // the same network as SCL:
   "DB16000_OPC_UA_TRIGGER_ALARM".CLIENT.U2_STA2_MEAS.TRIGGERS.START_CALIBRATION := NOT (NOT "DB359_M_UNIT_2_STA_2".M_CODES_UNIT_2_STA_2.M904) AND ("DB16003_U2_STA2_MEAS_CLIENT_INTERFACE".U02_STA2_MEAS_Read.Variable.Status = 0) AND NOT "DB2031_CYCLES_GENERAL".DRY_CYCLE.CYCLE_SELECTED AND NOT "DB2031_CYCLES_GENERAL".ROBOT_DRY_CYCLE.CYCLE_SELECTED AND "DB7255_UNIT_2_STA_2_MEAS_ENABLE_DISABLE".ENABLED;
END_REGION

REGION Network 19: UNIT 2 STATION 2 RESET PC TRIGGER
   RUNG wire#powerrail
      I_Contact( "DB2120_MPP_ITC_IPC".RESET_FAULTS )
      Not()
      { S7_Templates := "SrcType := Int" } EQ_Contact(in1 := "DB16003_U2_STA2_MEAS_CLIENT_INTERFACE".U02_STA2_MEAS_Read.Variable.Status, in2 := -1)
      Contact( "DB7255_UNIT_2_STA_2_MEAS_ENABLE_DISABLE".ENABLED )
      Coil( "DB16000_OPC_UA_TRIGGER_ALARM".CLIENT.U2_STA2_MEAS.TRIGGERS.RESET_PC )
   END_RUNG
   // the same network as SCL:
   "DB16000_OPC_UA_TRIGGER_ALARM".CLIENT.U2_STA2_MEAS.TRIGGERS.RESET_PC := NOT (NOT "DB2120_MPP_ITC_IPC".RESET_FAULTS) AND ("DB16003_U2_STA2_MEAS_CLIENT_INTERFACE".U02_STA2_MEAS_Read.Variable.Status = (-1)) AND "DB7255_UNIT_2_STA_2_MEAS_ENABLE_DISABLE".ENABLED;
END_REGION

REGION Network 20: UNIT 2 STATION 2 READ VARIABLES TRIGGER
   RUNG wire#powerrail
      I_Contact( "DB2120_MPP_ITC_IPC".MACHINE_ON_DELAYED )
      Not()
      I_Contact( "DB16320_READLIST_U2_STA2_MEAS".Busy )
      I_Contact( "DB16428_U2_ST2_MEAS_RECONNECT".CONNECTION_ERROR )
      Contact( "DB7255_UNIT_2_STA_2_MEAS_ENABLE_DISABLE".ENABLED )
      Coil( "DB16000_OPC_UA_TRIGGER_ALARM".CLIENT.U2_STA2_MEAS.TRIGGERS.READ_VARS )
   END_RUNG
   // the same network as SCL:
   "DB16000_OPC_UA_TRIGGER_ALARM".CLIENT.U2_STA2_MEAS.TRIGGERS.READ_VARS := NOT (NOT "DB2120_MPP_ITC_IPC".MACHINE_ON_DELAYED) AND NOT "DB16320_READLIST_U2_STA2_MEAS".Busy AND NOT "DB16428_U2_ST2_MEAS_RECONNECT".CONNECTION_ERROR AND "DB7255_UNIT_2_STA_2_MEAS_ENABLE_DISABLE".ENABLED;
END_REGION

REGION Network 21: UNIT 2 STATION 2 MEASURING CHECK CONNECTION STATUS TRIGGER
   RUNG wire#powerrail
      Contact( "DB16224_CONNECTION_STATUS_U2_STA2_MEAS".Busy )
      Not()
      I_Contact( "DB16220_CONNECT_U2_STA2_MEAS".Busy )
      Contact( "DB7255_UNIT_2_STA_2_MEAS_ENABLE_DISABLE".ENABLED )
      Coil( "DB16000_OPC_UA_TRIGGER_ALARM".CLIENT.U2_STA2_MEAS.TRIGGERS.CHECK_CONN_STATUS )
   END_RUNG
   // the same network as SCL:
   "DB16000_OPC_UA_TRIGGER_ALARM".CLIENT.U2_STA2_MEAS.TRIGGERS.CHECK_CONN_STATUS := NOT "DB16224_CONNECTION_STATUS_U2_STA2_MEAS".Busy AND NOT "DB16220_CONNECT_U2_STA2_MEAS".Busy AND "DB7255_UNIT_2_STA_2_MEAS_ENABLE_DISABLE".ENABLED;
END_REGION

REGION Network 22: UNIT 2 STATION 2 MEASURING RELEASE HANDLE LIST TRIGGER
   RUNG wire#powerrail
      I_Contact( "DB16428_U2_ST2_MEAS_RECONNECT".DISCONNECT )
      Contact( "DB7255_UNIT_2_STA_2_MEAS_ENABLE_DISABLE".ENABLED )
      Not()
      Coil( "DB16000_OPC_UA_TRIGGER_ALARM".CLIENT.U2_STA2_MEAS.TRIGGERS.RELEASE_HANDLE_LIST )
   END_RUNG
   // the same network as SCL:
   "DB16000_OPC_UA_TRIGGER_ALARM".CLIENT.U2_STA2_MEAS.TRIGGERS.RELEASE_HANDLE_LIST := NOT (NOT "DB16428_U2_ST2_MEAS_RECONNECT".DISCONNECT AND "DB7255_UNIT_2_STA_2_MEAS_ENABLE_DISABLE".ENABLED);
END_REGION

REGION Network 23: UNIT 2 STATION 2 MEASURING RELEASE METHOD LIST TRIGGER
   RUNG wire#powerrail
      I_Contact( "DB16428_U2_ST2_MEAS_RECONNECT".DISCONNECT )
      Contact( "DB7255_UNIT_2_STA_2_MEAS_ENABLE_DISABLE".ENABLED )
      Not()
      Coil( "DB16000_OPC_UA_TRIGGER_ALARM".CLIENT.U2_STA2_MEAS.TRIGGERS.RELEASE_METHOD_LIST )
   END_RUNG
   // the same network as SCL:
   "DB16000_OPC_UA_TRIGGER_ALARM".CLIENT.U2_STA2_MEAS.TRIGGERS.RELEASE_METHOD_LIST := NOT (NOT "DB16428_U2_ST2_MEAS_RECONNECT".DISCONNECT AND "DB7255_UNIT_2_STA_2_MEAS_ENABLE_DISABLE".ENABLED);
END_REGION

REGION Network 24: UNIT 2 STATION 2 MEASURING STOP CONNECTION TRIGGER
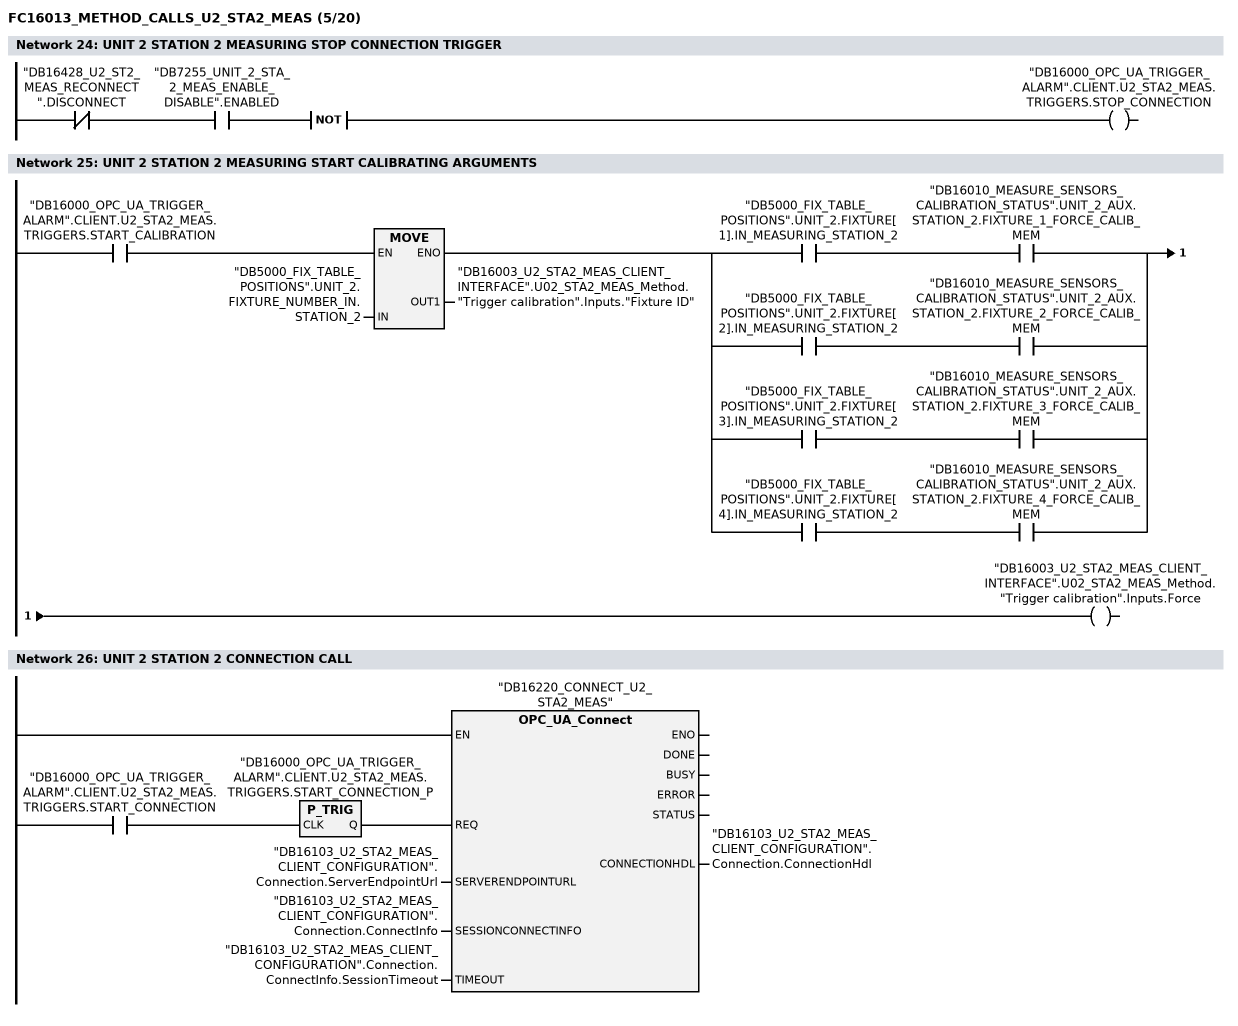
   RUNG wire#powerrail
      I_Contact( "DB16428_U2_ST2_MEAS_RECONNECT".DISCONNECT )
      Contact( "DB7255_UNIT_2_STA_2_MEAS_ENABLE_DISABLE".ENABLED )
      Not()
      Coil( "DB16000_OPC_UA_TRIGGER_ALARM".CLIENT.U2_STA2_MEAS.TRIGGERS.STOP_CONNECTION )
   END_RUNG
   // the same network as SCL:
   "DB16000_OPC_UA_TRIGGER_ALARM".CLIENT.U2_STA2_MEAS.TRIGGERS.STOP_CONNECTION := NOT (NOT "DB16428_U2_ST2_MEAS_RECONNECT".DISCONNECT AND "DB7255_UNIT_2_STA_2_MEAS_ENABLE_DISABLE".ENABLED);
END_REGION

REGION Network 25: UNIT 2 STATION 2 MEASURING START CALIBRATING ARGUMENTS
   RUNG wire#powerrail
      Contact( "DB16000_OPC_UA_TRIGGER_ALARM".CLIENT.U2_STA2_MEAS.TRIGGERS.START_CALIBRATION )
      Move(in := "DB5000_FIX_TABLE_POSITIONS".UNIT_2.FIXTURE_NUMBER_IN.STATION_2, out1 => "DB16003_U2_STA2_MEAS_CLIENT_INTERFACE".U02_STA2_MEAS_Method."Trigger calibration".Inputs."Fixture ID")
      wire#w1
      Contact( "DB5000_FIX_TABLE_POSITIONS".UNIT_2.FIXTURE[1].IN_MEASURING_STATION_2 )
      Contact( "DB16010_MEASURE_SENSORS_CALIBRATION_STATUS".UNIT_2_AUX.STATION_2.FIXTURE_1_FORCE_CALIB_MEM )
      wire#w2
      Coil( "DB16003_U2_STA2_MEAS_CLIENT_INTERFACE".U02_STA2_MEAS_Method."Trigger calibration".Inputs.Force )
   END_RUNG
   RUNG wire#w1
      Contact( "DB5000_FIX_TABLE_POSITIONS".UNIT_2.FIXTURE[2].IN_MEASURING_STATION_2 )
      Contact( "DB16010_MEASURE_SENSORS_CALIBRATION_STATUS".UNIT_2_AUX.STATION_2.FIXTURE_2_FORCE_CALIB_MEM )
   END_RUNG wire#w2
   RUNG wire#w1
      Contact( "DB5000_FIX_TABLE_POSITIONS".UNIT_2.FIXTURE[3].IN_MEASURING_STATION_2 )
      Contact( "DB16010_MEASURE_SENSORS_CALIBRATION_STATUS".UNIT_2_AUX.STATION_2.FIXTURE_3_FORCE_CALIB_MEM )
   END_RUNG wire#w2
   RUNG wire#w1
      Contact( "DB5000_FIX_TABLE_POSITIONS".UNIT_2.FIXTURE[4].IN_MEASURING_STATION_2 )
      Contact( "DB16010_MEASURE_SENSORS_CALIBRATION_STATUS".UNIT_2_AUX.STATION_2.FIXTURE_4_FORCE_CALIB_MEM )
   END_RUNG wire#w2
   // the same network as SCL:
   IF "DB16000_OPC_UA_TRIGGER_ALARM".CLIENT.U2_STA2_MEAS.TRIGGERS.START_CALIBRATION THEN
       "DB16003_U2_STA2_MEAS_CLIENT_INTERFACE".U02_STA2_MEAS_Method."Trigger calibration".Inputs."Fixture ID" := "DB5000_FIX_TABLE_POSITIONS".UNIT_2.FIXTURE_NUMBER_IN.STATION_2;
   END_IF;
   "DB16003_U2_STA2_MEAS_CLIENT_INTERFACE".U02_STA2_MEAS_Method."Trigger calibration".Inputs.Force := "DB16000_OPC_UA_TRIGGER_ALARM".CLIENT.U2_STA2_MEAS.TRIGGERS.START_CALIBRATION AND (("DB5000_FIX_TABLE_POSITIONS".UNIT_2.FIXTURE[1].IN_MEASURING_STATION_2 AND "DB16010_MEASURE_SENSORS_CALIBRATION_STATUS".UNIT_2_AUX.STATION_2.FIXTURE_1_FORCE_CALIB_MEM) OR ("DB5000_FIX_TABLE_POSITIONS".UNIT_2.FIXTURE[2].IN_MEASURING_STATION_2 AND "DB16010_MEASURE_SENSORS_CALIBRATION_STATUS".UNIT_2_AUX.STATION_2.FIXTURE_2_FORCE_CALIB_MEM) OR ("DB5000_FIX_TABLE_POSITIONS".UNIT_2.FIXTURE[3].IN_MEASURING_STATION_2 AND "DB16010_MEASURE_SENSORS_CALIBRATION_STATUS".UNIT_2_AUX.STATION_2.FIXTURE_3_FORCE_CALIB_MEM) OR ("DB5000_FIX_TABLE_POSITIONS".UNIT_2.FIXTURE[4].IN_MEASURING_STATION_2 AND "DB16010_MEASURE_SENSORS_CALIBRATION_STATUS".UNIT_2_AUX.STATION_2.FIXTURE_4_FORCE_CALIB_MEM));
END_REGION

REGION Network 26: UNIT 2 STATION 2 CONNECTION CALL
   RUNG wire#powerrail
      "DB16220_CONNECT_U2_STA2_MEAS".OPC_UA_Connect(REQ := wire#w1, ServerEndpointUrl := "DB16103_U2_STA2_MEAS_CLIENT_CONFIGURATION".Connection.ServerEndpointUrl, SessionConnectInfo := "DB16103_U2_STA2_MEAS_CLIENT_CONFIGURATION".Connection.ConnectInfo, Timeout := "DB16103_U2_STA2_MEAS_CLIENT_CONFIGURATION".Connection.ConnectInfo.SessionTimeout, Done =>, Busy =>, Error =>, Status =>, ConnectionHdl => "DB16103_U2_STA2_MEAS_CLIENT_CONFIGURATION".Connection.ConnectionHdl)
   END_RUNG
   RUNG wire#powerrail
      Contact( "DB16000_OPC_UA_TRIGGER_ALARM".CLIENT.U2_STA2_MEAS.TRIGGERS.START_CONNECTION )
      P_Trig( "DB16000_OPC_UA_TRIGGER_ALARM".CLIENT.U2_STA2_MEAS.TRIGGERS.START_CONNECTION_P )
   END_RUNG wire#w1
   // the same network as SCL:
   #_w1 := "DB16000_OPC_UA_TRIGGER_ALARM".CLIENT.U2_STA2_MEAS.TRIGGERS.START_CONNECTION AND NOT "DB16000_OPC_UA_TRIGGER_ALARM".CLIENT.U2_STA2_MEAS.TRIGGERS.START_CONNECTION_P;   // rising edge
   "DB16000_OPC_UA_TRIGGER_ALARM".CLIENT.U2_STA2_MEAS.TRIGGERS.START_CONNECTION_P := "DB16000_OPC_UA_TRIGGER_ALARM".CLIENT.U2_STA2_MEAS.TRIGGERS.START_CONNECTION;
   "DB16220_CONNECT_U2_STA2_MEAS"(REQ := #_w1,   // OPC_UA_Connect
                           ServerEndpointUrl := "DB16103_U2_STA2_MEAS_CLIENT_CONFIGURATION".Connection.ServerEndpointUrl,
                           SessionConnectInfo := "DB16103_U2_STA2_MEAS_CLIENT_CONFIGURATION".Connection.ConnectInfo,
                           Timeout := "DB16103_U2_STA2_MEAS_CLIENT_CONFIGURATION".Connection.ConnectInfo.SessionTimeout,
                           ConnectionHdl => "DB16103_U2_STA2_MEAS_CLIENT_CONFIGURATION".Connection.ConnectionHdl);
END_REGION

REGION Network 27: UNIT 2 STATION 2 GET INDEX LIST CALL
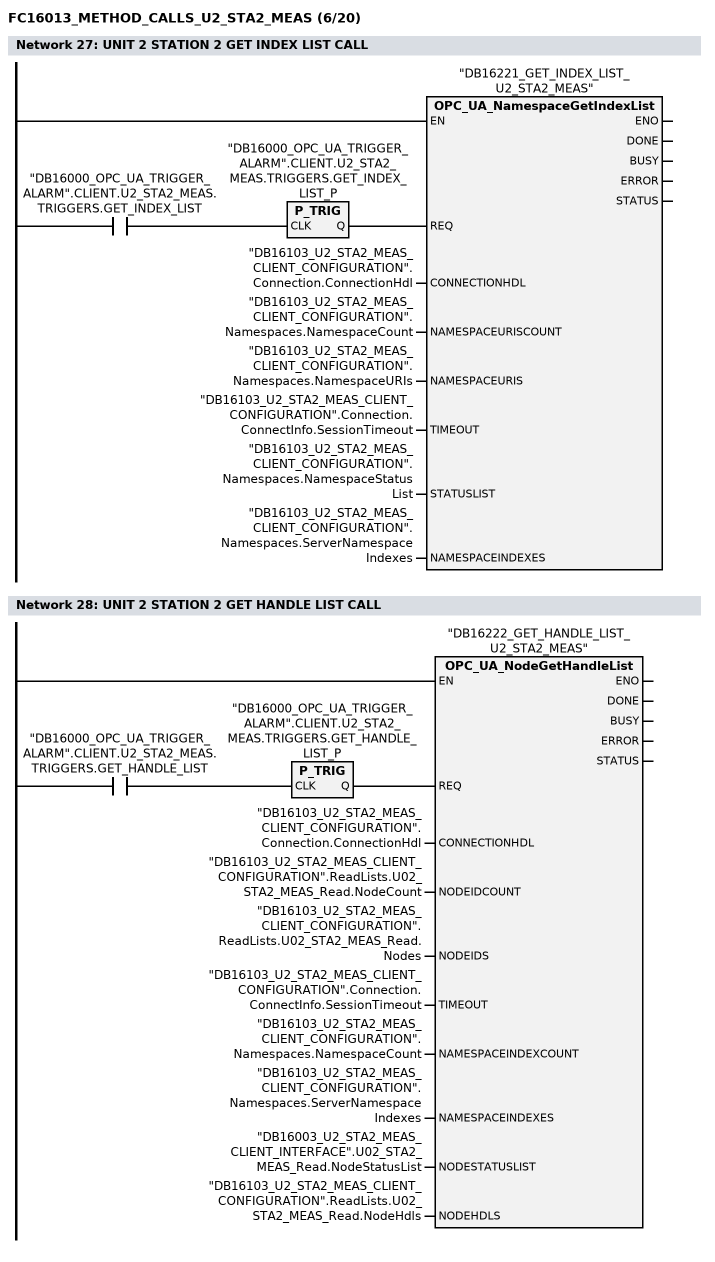
   RUNG wire#powerrail
      "DB16221_GET_INDEX_LIST_U2_STA2_MEAS".OPC_UA_NamespaceGetIndexList(REQ := wire#w1, ConnectionHdl := "DB16103_U2_STA2_MEAS_CLIENT_CONFIGURATION".Connection.ConnectionHdl, NamespaceUrisCount := "DB16103_U2_STA2_MEAS_CLIENT_CONFIGURATION".Namespaces.NamespaceCount, NamespaceUris := "DB16103_U2_STA2_MEAS_CLIENT_CONFIGURATION".Namespaces.NamespaceURIs, Timeout := "DB16103_U2_STA2_MEAS_CLIENT_CONFIGURATION".Connection.ConnectInfo.SessionTimeout, StatusList := "DB16103_U2_STA2_MEAS_CLIENT_CONFIGURATION".Namespaces.NamespaceStatusList, NamespaceIndexes := "DB16103_U2_STA2_MEAS_CLIENT_CONFIGURATION".Namespaces.ServerNamespaceIndexes, Done =>, Busy =>, Error =>, Status =>)
   END_RUNG
   RUNG wire#powerrail
      Contact( "DB16000_OPC_UA_TRIGGER_ALARM".CLIENT.U2_STA2_MEAS.TRIGGERS.GET_INDEX_LIST )
      P_Trig( "DB16000_OPC_UA_TRIGGER_ALARM".CLIENT.U2_STA2_MEAS.TRIGGERS.GET_INDEX_LIST_P )
   END_RUNG wire#w1
   // the same network as SCL:
   #_w1 := "DB16000_OPC_UA_TRIGGER_ALARM".CLIENT.U2_STA2_MEAS.TRIGGERS.GET_INDEX_LIST AND NOT "DB16000_OPC_UA_TRIGGER_ALARM".CLIENT.U2_STA2_MEAS.TRIGGERS.GET_INDEX_LIST_P;   // rising edge
   "DB16000_OPC_UA_TRIGGER_ALARM".CLIENT.U2_STA2_MEAS.TRIGGERS.GET_INDEX_LIST_P := "DB16000_OPC_UA_TRIGGER_ALARM".CLIENT.U2_STA2_MEAS.TRIGGERS.GET_INDEX_LIST;
   "DB16221_GET_INDEX_LIST_U2_STA2_MEAS"(REQ := #_w1,   // OPC_UA_NamespaceGetIndexList
                           ConnectionHdl := "DB16103_U2_STA2_MEAS_CLIENT_CONFIGURATION".Connection.ConnectionHdl,
                           NamespaceUrisCount := "DB16103_U2_STA2_MEAS_CLIENT_CONFIGURATION".Namespaces.NamespaceCount,
                           NamespaceUris := "DB16103_U2_STA2_MEAS_CLIENT_CONFIGURATION".Namespaces.NamespaceURIs,
                           Timeout := "DB16103_U2_STA2_MEAS_CLIENT_CONFIGURATION".Connection.ConnectInfo.SessionTimeout,
                           StatusList := "DB16103_U2_STA2_MEAS_CLIENT_CONFIGURATION".Namespaces.NamespaceStatusList,
                           NamespaceIndexes := "DB16103_U2_STA2_MEAS_CLIENT_CONFIGURATION".Namespaces.ServerNamespaceIndexes);
END_REGION

REGION Network 28: UNIT 2 STATION 2 GET HANDLE LIST CALL
   RUNG wire#powerrail
      "DB16222_GET_HANDLE_LIST_U2_STA2_MEAS".OPC_UA_NodeGetHandleList(REQ := wire#w1, ConnectionHdl := "DB16103_U2_STA2_MEAS_CLIENT_CONFIGURATION".Connection.ConnectionHdl, NodeIDCount := "DB16103_U2_STA2_MEAS_CLIENT_CONFIGURATION".ReadLists.U02_STA2_MEAS_Read.NodeCount, NodeIDs := "DB16103_U2_STA2_MEAS_CLIENT_CONFIGURATION".ReadLists.U02_STA2_MEAS_Read.Nodes, Timeout := "DB16103_U2_STA2_MEAS_CLIENT_CONFIGURATION".Connection.ConnectInfo.SessionTimeout, NamespaceIndexCount := "DB16103_U2_STA2_MEAS_CLIENT_CONFIGURATION".Namespaces.NamespaceCount, NamespaceIndexes := "DB16103_U2_STA2_MEAS_CLIENT_CONFIGURATION".Namespaces.ServerNamespaceIndexes, NodeStatusList := "DB16003_U2_STA2_MEAS_CLIENT_INTERFACE".U02_STA2_MEAS_Read.NodeStatusList, NodeHdls := "DB16103_U2_STA2_MEAS_CLIENT_CONFIGURATION".ReadLists.U02_STA2_MEAS_Read.NodeHdls, Done =>, Busy =>, Error =>, Status =>)
   END_RUNG
   RUNG wire#powerrail
      Contact( "DB16000_OPC_UA_TRIGGER_ALARM".CLIENT.U2_STA2_MEAS.TRIGGERS.GET_HANDLE_LIST )
      P_Trig( "DB16000_OPC_UA_TRIGGER_ALARM".CLIENT.U2_STA2_MEAS.TRIGGERS.GET_HANDLE_LIST_P )
   END_RUNG wire#w1
   // the same network as SCL:
   #_w1 := "DB16000_OPC_UA_TRIGGER_ALARM".CLIENT.U2_STA2_MEAS.TRIGGERS.GET_HANDLE_LIST AND NOT "DB16000_OPC_UA_TRIGGER_ALARM".CLIENT.U2_STA2_MEAS.TRIGGERS.GET_HANDLE_LIST_P;   // rising edge
   "DB16000_OPC_UA_TRIGGER_ALARM".CLIENT.U2_STA2_MEAS.TRIGGERS.GET_HANDLE_LIST_P := "DB16000_OPC_UA_TRIGGER_ALARM".CLIENT.U2_STA2_MEAS.TRIGGERS.GET_HANDLE_LIST;
   "DB16222_GET_HANDLE_LIST_U2_STA2_MEAS"(REQ := #_w1,   // OPC_UA_NodeGetHandleList
                           ConnectionHdl := "DB16103_U2_STA2_MEAS_CLIENT_CONFIGURATION".Connection.ConnectionHdl,
                           NodeIDCount := "DB16103_U2_STA2_MEAS_CLIENT_CONFIGURATION".ReadLists.U02_STA2_MEAS_Read.NodeCount,
                           NodeIDs := "DB16103_U2_STA2_MEAS_CLIENT_CONFIGURATION".ReadLists.U02_STA2_MEAS_Read.Nodes,
                           Timeout := "DB16103_U2_STA2_MEAS_CLIENT_CONFIGURATION".Connection.ConnectInfo.SessionTimeout,
                           NamespaceIndexCount := "DB16103_U2_STA2_MEAS_CLIENT_CONFIGURATION".Namespaces.NamespaceCount,
                           NamespaceIndexes := "DB16103_U2_STA2_MEAS_CLIENT_CONFIGURATION".Namespaces.ServerNamespaceIndexes,
                           NodeStatusList := "DB16003_U2_STA2_MEAS_CLIENT_INTERFACE".U02_STA2_MEAS_Read.NodeStatusList,
                           NodeHdls := "DB16103_U2_STA2_MEAS_CLIENT_CONFIGURATION".ReadLists.U02_STA2_MEAS_Read.NodeHdls);
END_REGION

REGION Network 29: UNIT 2 STATION 2 GET METHOD LIST CALL
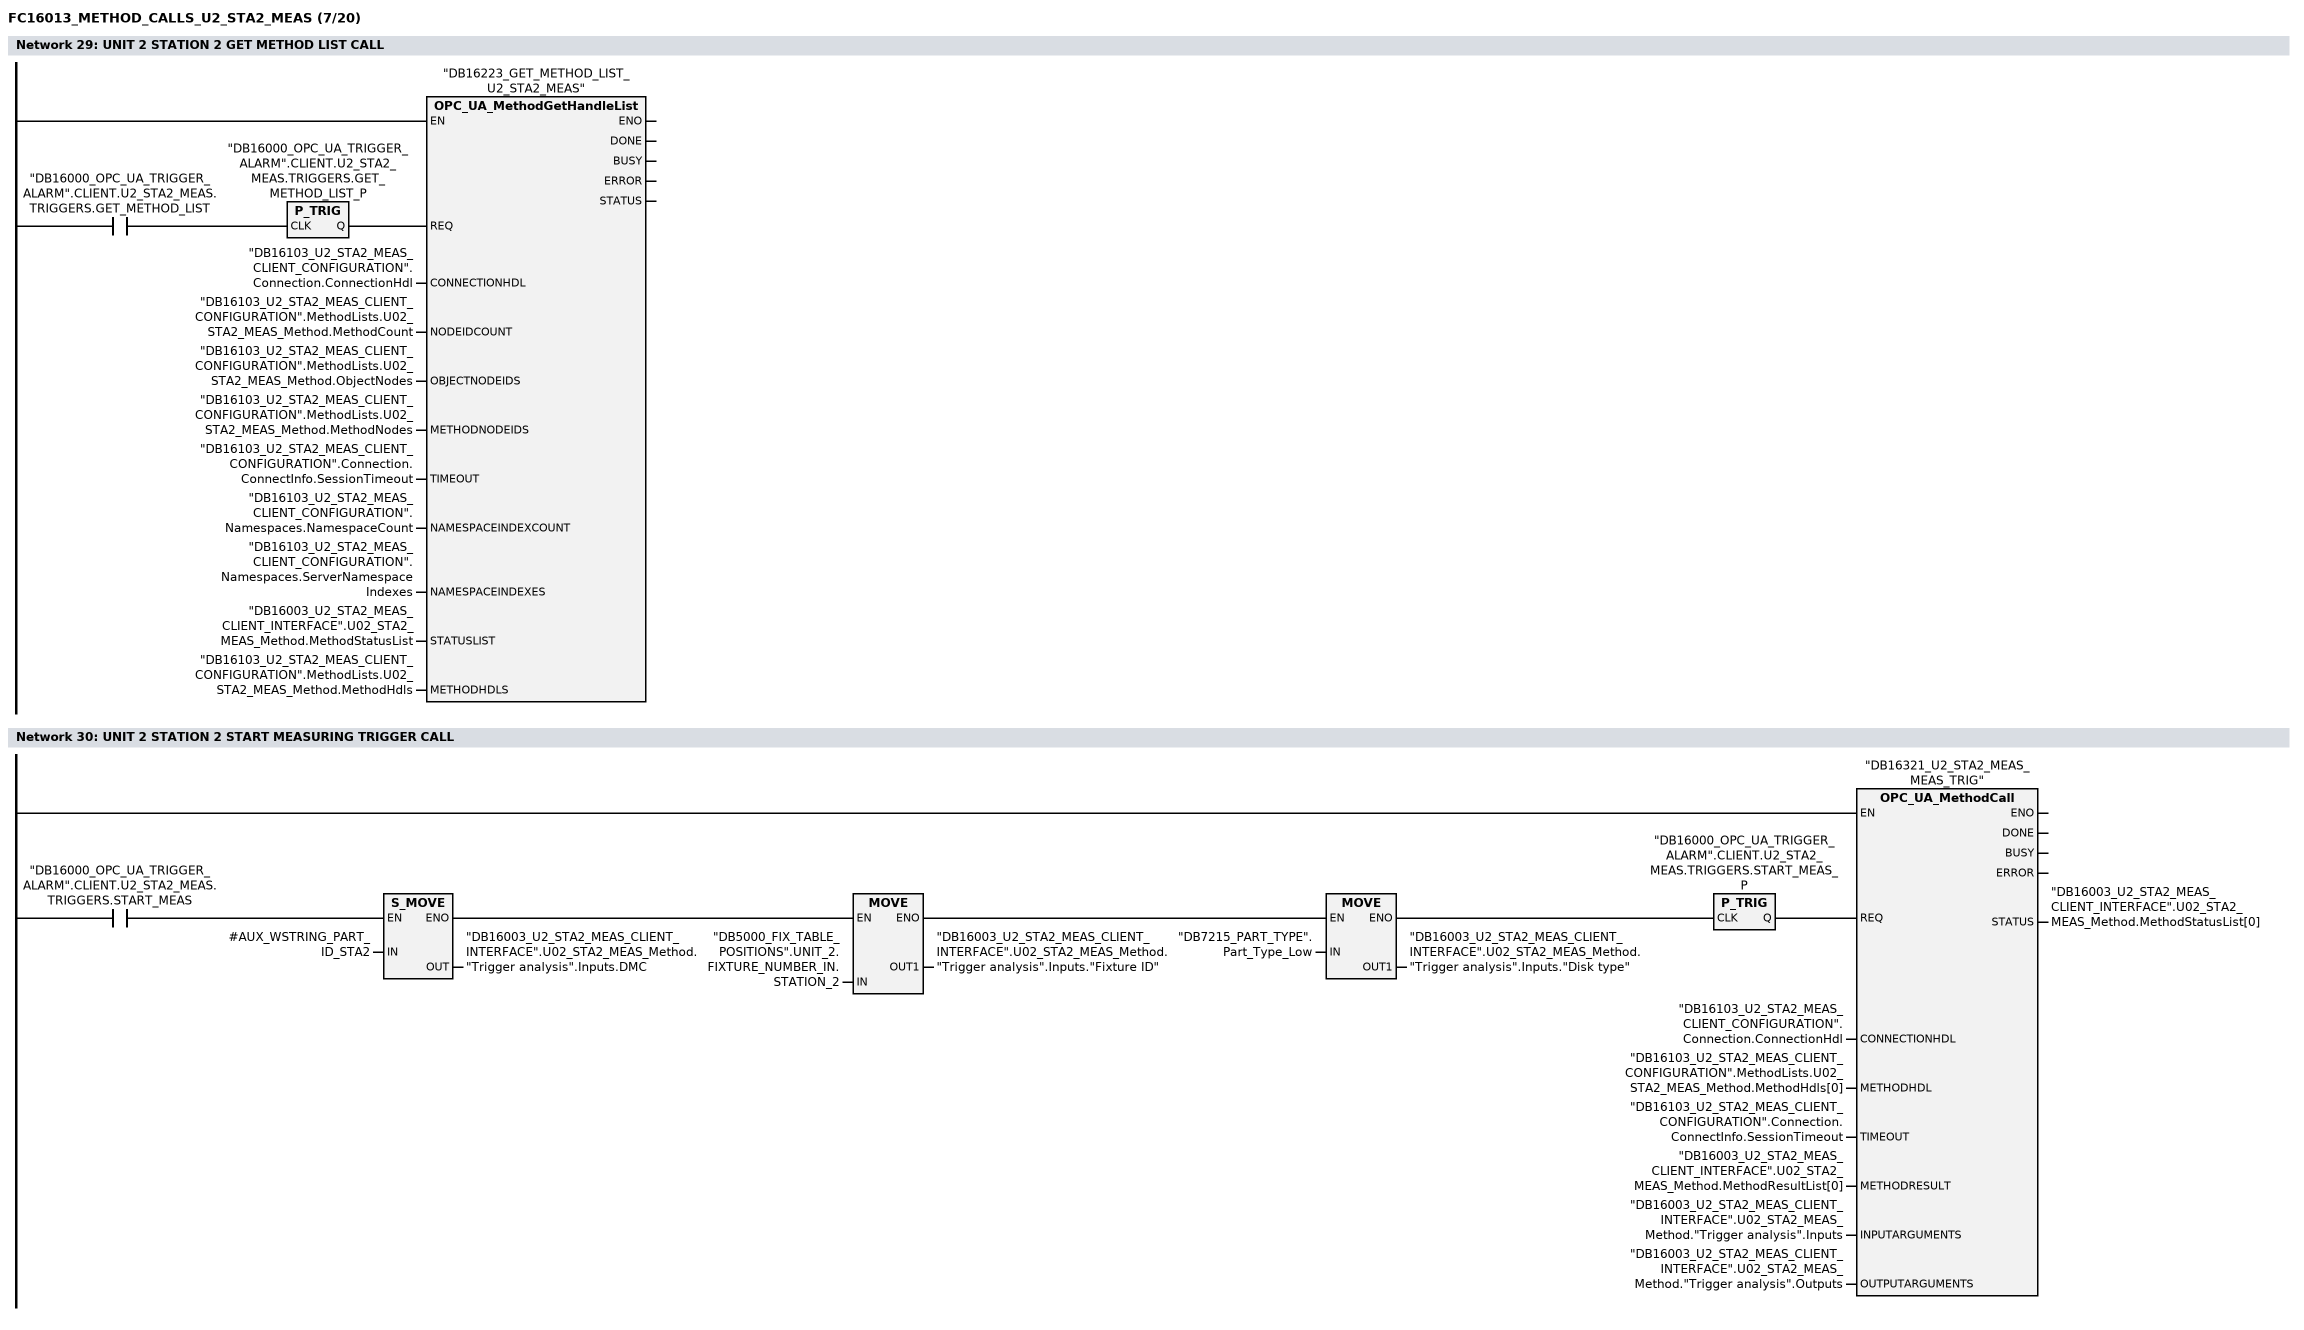
   RUNG wire#powerrail
      "DB16223_GET_METHOD_LIST_U2_STA2_MEAS".OPC_UA_MethodGetHandleList(REQ := wire#w1, ConnectionHdl := "DB16103_U2_STA2_MEAS_CLIENT_CONFIGURATION".Connection.ConnectionHdl, NodeIDCount := "DB16103_U2_STA2_MEAS_CLIENT_CONFIGURATION".MethodLists.U02_STA2_MEAS_Method.MethodCount, ObjectNodeIDs := "DB16103_U2_STA2_MEAS_CLIENT_CONFIGURATION".MethodLists.U02_STA2_MEAS_Method.ObjectNodes, MethodNodeIDs := "DB16103_U2_STA2_MEAS_CLIENT_CONFIGURATION".MethodLists.U02_STA2_MEAS_Method.MethodNodes, Timeout := "DB16103_U2_STA2_MEAS_CLIENT_CONFIGURATION".Connection.ConnectInfo.SessionTimeout, NamespaceIndexCount := "DB16103_U2_STA2_MEAS_CLIENT_CONFIGURATION".Namespaces.NamespaceCount, NamespaceIndexes := "DB16103_U2_STA2_MEAS_CLIENT_CONFIGURATION".Namespaces.ServerNamespaceIndexes, StatusList := "DB16003_U2_STA2_MEAS_CLIENT_INTERFACE".U02_STA2_MEAS_Method.MethodStatusList, MethodHdls := "DB16103_U2_STA2_MEAS_CLIENT_CONFIGURATION".MethodLists.U02_STA2_MEAS_Method.MethodHdls, Done =>, Busy =>, Error =>, Status =>)
   END_RUNG
   RUNG wire#powerrail
      Contact( "DB16000_OPC_UA_TRIGGER_ALARM".CLIENT.U2_STA2_MEAS.TRIGGERS.GET_METHOD_LIST )
      P_Trig( "DB16000_OPC_UA_TRIGGER_ALARM".CLIENT.U2_STA2_MEAS.TRIGGERS.GET_METHOD_LIST_P )
   END_RUNG wire#w1
   // the same network as SCL:
   #_w1 := "DB16000_OPC_UA_TRIGGER_ALARM".CLIENT.U2_STA2_MEAS.TRIGGERS.GET_METHOD_LIST AND NOT "DB16000_OPC_UA_TRIGGER_ALARM".CLIENT.U2_STA2_MEAS.TRIGGERS.GET_METHOD_LIST_P;   // rising edge
   "DB16000_OPC_UA_TRIGGER_ALARM".CLIENT.U2_STA2_MEAS.TRIGGERS.GET_METHOD_LIST_P := "DB16000_OPC_UA_TRIGGER_ALARM".CLIENT.U2_STA2_MEAS.TRIGGERS.GET_METHOD_LIST;
   "DB16223_GET_METHOD_LIST_U2_STA2_MEAS"(REQ := #_w1,   // OPC_UA_MethodGetHandleList
                           ConnectionHdl := "DB16103_U2_STA2_MEAS_CLIENT_CONFIGURATION".Connection.ConnectionHdl,
                           NodeIDCount := "DB16103_U2_STA2_MEAS_CLIENT_CONFIGURATION".MethodLists.U02_STA2_MEAS_Method.MethodCount,
                           ObjectNodeIDs := "DB16103_U2_STA2_MEAS_CLIENT_CONFIGURATION".MethodLists.U02_STA2_MEAS_Method.ObjectNodes,
                           MethodNodeIDs := "DB16103_U2_STA2_MEAS_CLIENT_CONFIGURATION".MethodLists.U02_STA2_MEAS_Method.MethodNodes,
                           Timeout := "DB16103_U2_STA2_MEAS_CLIENT_CONFIGURATION".Connection.ConnectInfo.SessionTimeout,
                           NamespaceIndexCount := "DB16103_U2_STA2_MEAS_CLIENT_CONFIGURATION".Namespaces.NamespaceCount,
                           NamespaceIndexes := "DB16103_U2_STA2_MEAS_CLIENT_CONFIGURATION".Namespaces.ServerNamespaceIndexes,
                           StatusList := "DB16003_U2_STA2_MEAS_CLIENT_INTERFACE".U02_STA2_MEAS_Method.MethodStatusList,
                           MethodHdls := "DB16103_U2_STA2_MEAS_CLIENT_CONFIGURATION".MethodLists.U02_STA2_MEAS_Method.MethodHdls);
END_REGION

REGION Network 30: UNIT 2 STATION 2 START MEASURING TRIGGER CALL
   RUNG wire#powerrail
      "DB16321_U2_STA2_MEAS_MEAS_TRIG".OPC_UA_MethodCall(REQ := wire#w1, ConnectionHdl := "DB16103_U2_STA2_MEAS_CLIENT_CONFIGURATION".Connection.ConnectionHdl, MethodHdl := "DB16103_U2_STA2_MEAS_CLIENT_CONFIGURATION".MethodLists.U02_STA2_MEAS_Method.MethodHdls[0], Timeout := "DB16103_U2_STA2_MEAS_CLIENT_CONFIGURATION".Connection.ConnectInfo.SessionTimeout, MethodResult := "DB16003_U2_STA2_MEAS_CLIENT_INTERFACE".U02_STA2_MEAS_Method.MethodResultList[0], InputArguments := "DB16003_U2_STA2_MEAS_CLIENT_INTERFACE".U02_STA2_MEAS_Method."Trigger analysis".Inputs, OutputArguments := "DB16003_U2_STA2_MEAS_CLIENT_INTERFACE".U02_STA2_MEAS_Method."Trigger analysis".Outputs, Done =>, Busy =>, Error =>, Status => "DB16003_U2_STA2_MEAS_CLIENT_INTERFACE".U02_STA2_MEAS_Method.MethodStatusList[0])
   END_RUNG
   RUNG wire#powerrail
      Contact( "DB16000_OPC_UA_TRIGGER_ALARM".CLIENT.U2_STA2_MEAS.TRIGGERS.START_MEAS )
      S_Move(in := #AUX_WSTRING_PART_ID_STA2, out => "DB16003_U2_STA2_MEAS_CLIENT_INTERFACE".U02_STA2_MEAS_Method."Trigger analysis".Inputs.DMC)
      Move(in := "DB5000_FIX_TABLE_POSITIONS".UNIT_2.FIXTURE_NUMBER_IN.STATION_2, out1 => "DB16003_U2_STA2_MEAS_CLIENT_INTERFACE".U02_STA2_MEAS_Method."Trigger analysis".Inputs."Fixture ID")
      Move(in := "DB7215_PART_TYPE".Part_Type_Low, out1 => "DB16003_U2_STA2_MEAS_CLIENT_INTERFACE".U02_STA2_MEAS_Method."Trigger analysis".Inputs."Disk type")
      P_Trig( "DB16000_OPC_UA_TRIGGER_ALARM".CLIENT.U2_STA2_MEAS.TRIGGERS.START_MEAS_P )
   END_RUNG wire#w1
   // the same network as SCL:
   IF "DB16000_OPC_UA_TRIGGER_ALARM".CLIENT.U2_STA2_MEAS.TRIGGERS.START_MEAS THEN
       "DB16003_U2_STA2_MEAS_CLIENT_INTERFACE".U02_STA2_MEAS_Method."Trigger analysis".Inputs.DMC := #AUX_WSTRING_PART_ID_STA2;
       "DB16003_U2_STA2_MEAS_CLIENT_INTERFACE".U02_STA2_MEAS_Method."Trigger analysis".Inputs."Fixture ID" := "DB5000_FIX_TABLE_POSITIONS".UNIT_2.FIXTURE_NUMBER_IN.STATION_2;
       "DB16003_U2_STA2_MEAS_CLIENT_INTERFACE".U02_STA2_MEAS_Method."Trigger analysis".Inputs."Disk type" := "DB7215_PART_TYPE".Part_Type_Low;
   END_IF;
   #_w1 := "DB16000_OPC_UA_TRIGGER_ALARM".CLIENT.U2_STA2_MEAS.TRIGGERS.START_MEAS AND NOT "DB16000_OPC_UA_TRIGGER_ALARM".CLIENT.U2_STA2_MEAS.TRIGGERS.START_MEAS_P;   // rising edge
   "DB16000_OPC_UA_TRIGGER_ALARM".CLIENT.U2_STA2_MEAS.TRIGGERS.START_MEAS_P := "DB16000_OPC_UA_TRIGGER_ALARM".CLIENT.U2_STA2_MEAS.TRIGGERS.START_MEAS;
   "DB16321_U2_STA2_MEAS_MEAS_TRIG"(REQ := #_w1,   // OPC_UA_MethodCall
                           ConnectionHdl := "DB16103_U2_STA2_MEAS_CLIENT_CONFIGURATION".Connection.ConnectionHdl,
                           MethodHdl := "DB16103_U2_STA2_MEAS_CLIENT_CONFIGURATION".MethodLists.U02_STA2_MEAS_Method.MethodHdls[0],
                           Timeout := "DB16103_U2_STA2_MEAS_CLIENT_CONFIGURATION".Connection.ConnectInfo.SessionTimeout,
                           MethodResult := "DB16003_U2_STA2_MEAS_CLIENT_INTERFACE".U02_STA2_MEAS_Method.MethodResultList[0],
                           InputArguments := "DB16003_U2_STA2_MEAS_CLIENT_INTERFACE".U02_STA2_MEAS_Method."Trigger analysis".Inputs,
                           OutputArguments := "DB16003_U2_STA2_MEAS_CLIENT_INTERFACE".U02_STA2_MEAS_Method."Trigger analysis".Outputs,
                           Status => "DB16003_U2_STA2_MEAS_CLIENT_INTERFACE".U02_STA2_MEAS_Method.MethodStatusList[0]);
END_REGION

REGION Network 31: UNIT 2 STATION 2 START CALIBRATING TRIGGER CALL
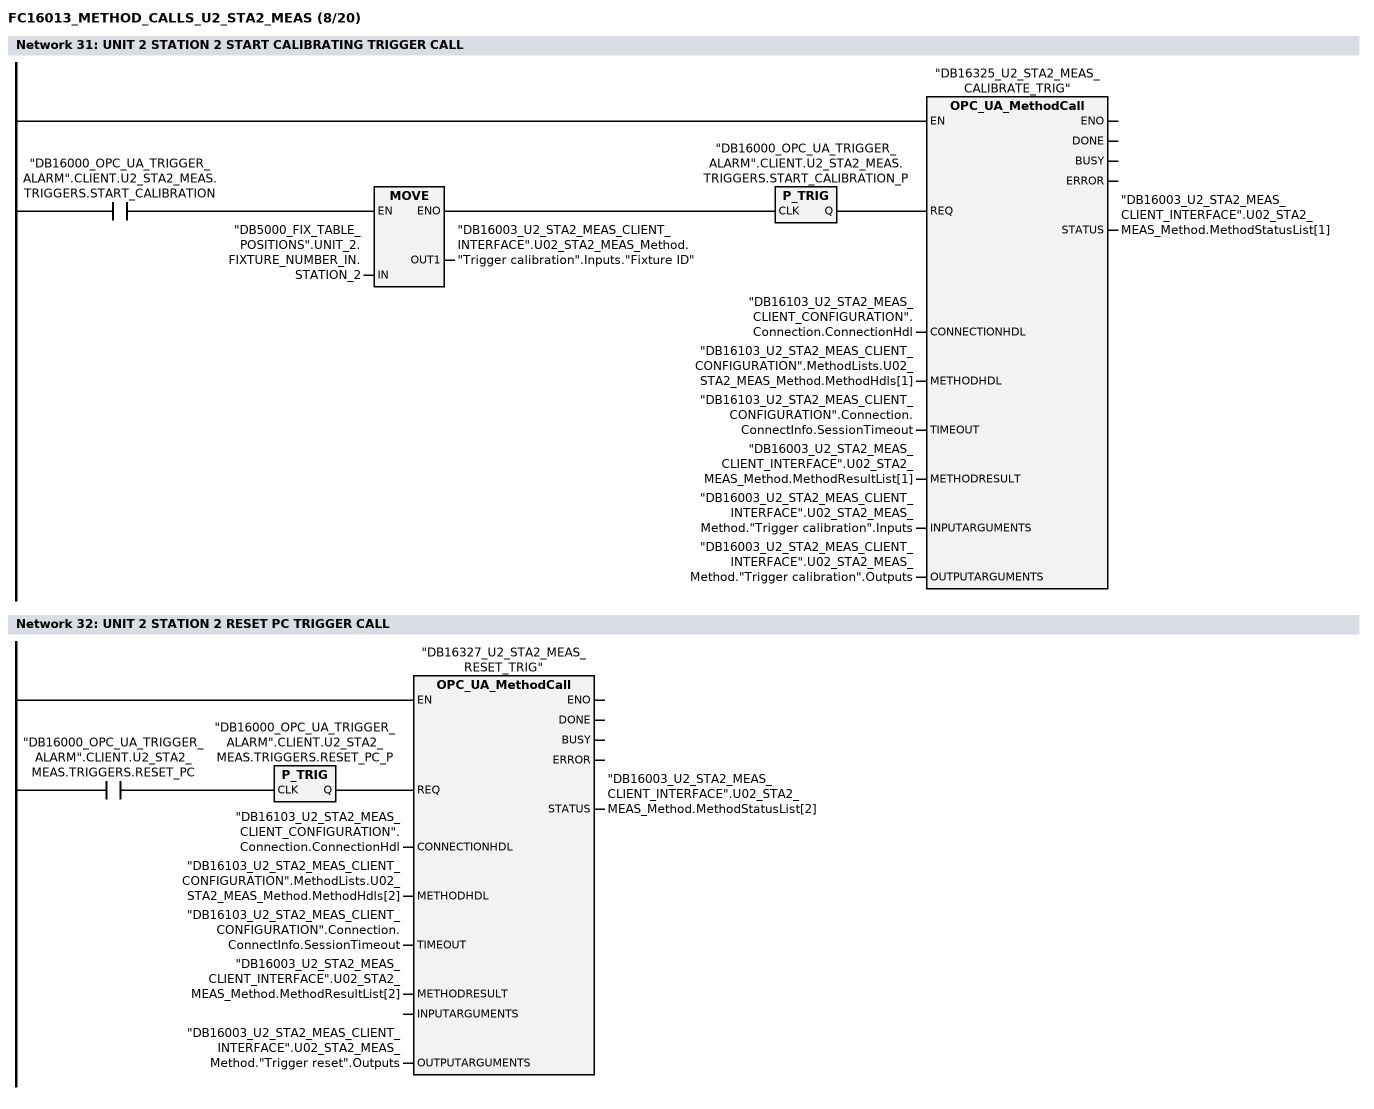
   RUNG wire#powerrail
      "DB16325_U2_STA2_MEAS_CALIBRATE_TRIG".OPC_UA_MethodCall(REQ := wire#w1, ConnectionHdl := "DB16103_U2_STA2_MEAS_CLIENT_CONFIGURATION".Connection.ConnectionHdl, MethodHdl := "DB16103_U2_STA2_MEAS_CLIENT_CONFIGURATION".MethodLists.U02_STA2_MEAS_Method.MethodHdls[1], Timeout := "DB16103_U2_STA2_MEAS_CLIENT_CONFIGURATION".Connection.ConnectInfo.SessionTimeout, MethodResult := "DB16003_U2_STA2_MEAS_CLIENT_INTERFACE".U02_STA2_MEAS_Method.MethodResultList[1], InputArguments := "DB16003_U2_STA2_MEAS_CLIENT_INTERFACE".U02_STA2_MEAS_Method."Trigger calibration".Inputs, OutputArguments := "DB16003_U2_STA2_MEAS_CLIENT_INTERFACE".U02_STA2_MEAS_Method."Trigger calibration".Outputs, Done =>, Busy =>, Error =>, Status => "DB16003_U2_STA2_MEAS_CLIENT_INTERFACE".U02_STA2_MEAS_Method.MethodStatusList[1])
   END_RUNG
   RUNG wire#powerrail
      Contact( "DB16000_OPC_UA_TRIGGER_ALARM".CLIENT.U2_STA2_MEAS.TRIGGERS.START_CALIBRATION )
      Move(in := "DB5000_FIX_TABLE_POSITIONS".UNIT_2.FIXTURE_NUMBER_IN.STATION_2, out1 => "DB16003_U2_STA2_MEAS_CLIENT_INTERFACE".U02_STA2_MEAS_Method."Trigger calibration".Inputs."Fixture ID")
      P_Trig( "DB16000_OPC_UA_TRIGGER_ALARM".CLIENT.U2_STA2_MEAS.TRIGGERS.START_CALIBRATION_P )
   END_RUNG wire#w1
   // the same network as SCL:
   IF "DB16000_OPC_UA_TRIGGER_ALARM".CLIENT.U2_STA2_MEAS.TRIGGERS.START_CALIBRATION THEN
       "DB16003_U2_STA2_MEAS_CLIENT_INTERFACE".U02_STA2_MEAS_Method."Trigger calibration".Inputs."Fixture ID" := "DB5000_FIX_TABLE_POSITIONS".UNIT_2.FIXTURE_NUMBER_IN.STATION_2;
   END_IF;
   #_w1 := "DB16000_OPC_UA_TRIGGER_ALARM".CLIENT.U2_STA2_MEAS.TRIGGERS.START_CALIBRATION AND NOT "DB16000_OPC_UA_TRIGGER_ALARM".CLIENT.U2_STA2_MEAS.TRIGGERS.START_CALIBRATION_P;   // rising edge
   "DB16000_OPC_UA_TRIGGER_ALARM".CLIENT.U2_STA2_MEAS.TRIGGERS.START_CALIBRATION_P := "DB16000_OPC_UA_TRIGGER_ALARM".CLIENT.U2_STA2_MEAS.TRIGGERS.START_CALIBRATION;
   "DB16325_U2_STA2_MEAS_CALIBRATE_TRIG"(REQ := #_w1,   // OPC_UA_MethodCall
                           ConnectionHdl := "DB16103_U2_STA2_MEAS_CLIENT_CONFIGURATION".Connection.ConnectionHdl,
                           MethodHdl := "DB16103_U2_STA2_MEAS_CLIENT_CONFIGURATION".MethodLists.U02_STA2_MEAS_Method.MethodHdls[1],
                           Timeout := "DB16103_U2_STA2_MEAS_CLIENT_CONFIGURATION".Connection.ConnectInfo.SessionTimeout,
                           MethodResult := "DB16003_U2_STA2_MEAS_CLIENT_INTERFACE".U02_STA2_MEAS_Method.MethodResultList[1],
                           InputArguments := "DB16003_U2_STA2_MEAS_CLIENT_INTERFACE".U02_STA2_MEAS_Method."Trigger calibration".Inputs,
                           OutputArguments := "DB16003_U2_STA2_MEAS_CLIENT_INTERFACE".U02_STA2_MEAS_Method."Trigger calibration".Outputs,
                           Status => "DB16003_U2_STA2_MEAS_CLIENT_INTERFACE".U02_STA2_MEAS_Method.MethodStatusList[1]);
END_REGION

REGION Network 32: UNIT 2 STATION 2 RESET PC TRIGGER CALL
   RUNG wire#powerrail
      "DB16327_U2_STA2_MEAS_RESET_TRIG".OPC_UA_MethodCall(REQ := wire#w1, ConnectionHdl := "DB16103_U2_STA2_MEAS_CLIENT_CONFIGURATION".Connection.ConnectionHdl, MethodHdl := "DB16103_U2_STA2_MEAS_CLIENT_CONFIGURATION".MethodLists.U02_STA2_MEAS_Method.MethodHdls[2], Timeout := "DB16103_U2_STA2_MEAS_CLIENT_CONFIGURATION".Connection.ConnectInfo.SessionTimeout, MethodResult := "DB16003_U2_STA2_MEAS_CLIENT_INTERFACE".U02_STA2_MEAS_Method.MethodResultList[2], InputArguments :=, OutputArguments := "DB16003_U2_STA2_MEAS_CLIENT_INTERFACE".U02_STA2_MEAS_Method."Trigger reset".Outputs, Done =>, Busy =>, Error =>, Status => "DB16003_U2_STA2_MEAS_CLIENT_INTERFACE".U02_STA2_MEAS_Method.MethodStatusList[2])
   END_RUNG
   RUNG wire#powerrail
      Contact( "DB16000_OPC_UA_TRIGGER_ALARM".CLIENT.U2_STA2_MEAS.TRIGGERS.RESET_PC )
      P_Trig( "DB16000_OPC_UA_TRIGGER_ALARM".CLIENT.U2_STA2_MEAS.TRIGGERS.RESET_PC_P )
   END_RUNG wire#w1
   // the same network as SCL:
   #_w1 := "DB16000_OPC_UA_TRIGGER_ALARM".CLIENT.U2_STA2_MEAS.TRIGGERS.RESET_PC AND NOT "DB16000_OPC_UA_TRIGGER_ALARM".CLIENT.U2_STA2_MEAS.TRIGGERS.RESET_PC_P;   // rising edge
   "DB16000_OPC_UA_TRIGGER_ALARM".CLIENT.U2_STA2_MEAS.TRIGGERS.RESET_PC_P := "DB16000_OPC_UA_TRIGGER_ALARM".CLIENT.U2_STA2_MEAS.TRIGGERS.RESET_PC;
   "DB16327_U2_STA2_MEAS_RESET_TRIG"(REQ := #_w1,   // OPC_UA_MethodCall
                           ConnectionHdl := "DB16103_U2_STA2_MEAS_CLIENT_CONFIGURATION".Connection.ConnectionHdl,
                           MethodHdl := "DB16103_U2_STA2_MEAS_CLIENT_CONFIGURATION".MethodLists.U02_STA2_MEAS_Method.MethodHdls[2],
                           Timeout := "DB16103_U2_STA2_MEAS_CLIENT_CONFIGURATION".Connection.ConnectInfo.SessionTimeout,
                           MethodResult := "DB16003_U2_STA2_MEAS_CLIENT_INTERFACE".U02_STA2_MEAS_Method.MethodResultList[2],
                           OutputArguments := "DB16003_U2_STA2_MEAS_CLIENT_INTERFACE".U02_STA2_MEAS_Method."Trigger reset".Outputs,
                           Status => "DB16003_U2_STA2_MEAS_CLIENT_INTERFACE".U02_STA2_MEAS_Method.MethodStatusList[2]);
END_REGION

REGION Network 33: UNIT 2 STATION 2 READ VARIABLES TRIGGER CALL
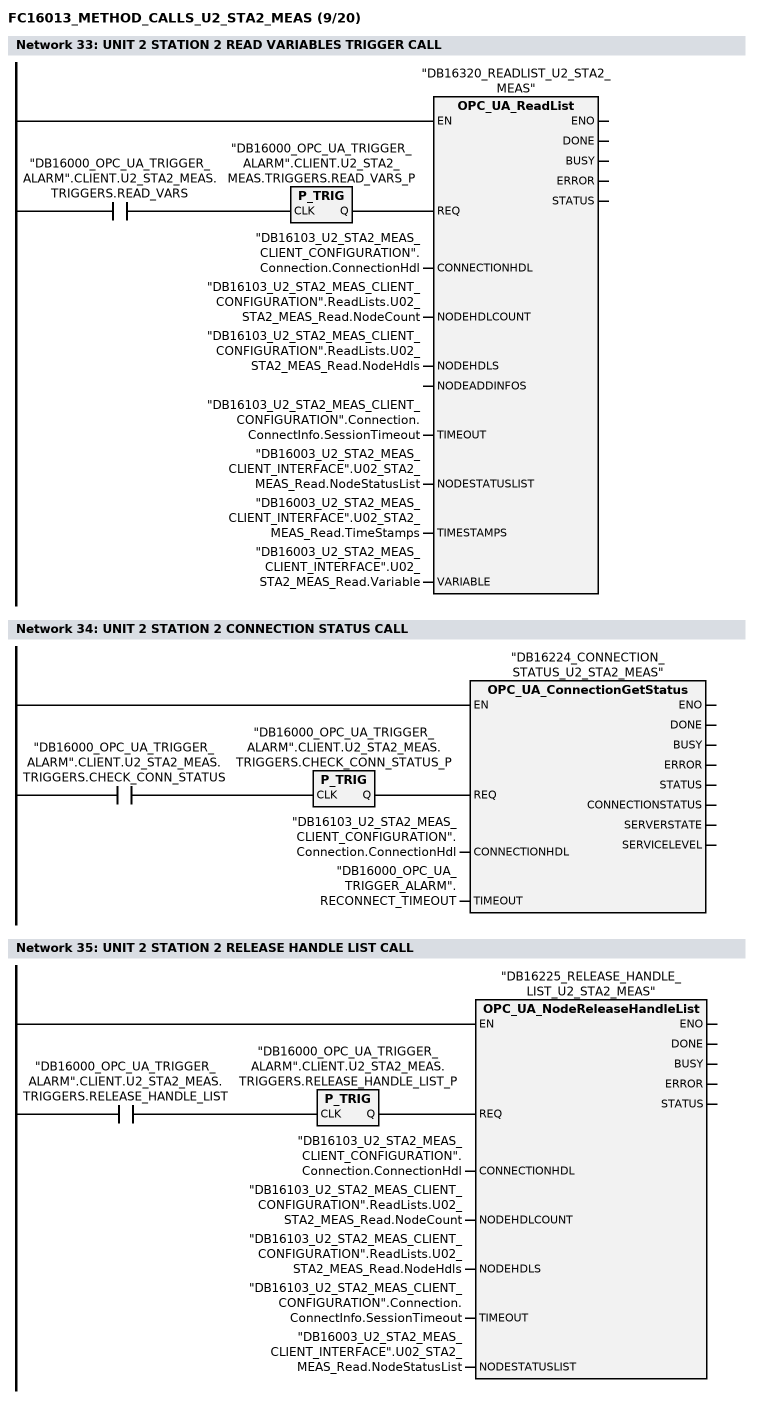
   RUNG wire#powerrail
      "DB16320_READLIST_U2_STA2_MEAS".OPC_UA_ReadList(REQ := wire#w1, ConnectionHdl := "DB16103_U2_STA2_MEAS_CLIENT_CONFIGURATION".Connection.ConnectionHdl, NodeHdlCount := "DB16103_U2_STA2_MEAS_CLIENT_CONFIGURATION".ReadLists.U02_STA2_MEAS_Read.NodeCount, NodeHdls := "DB16103_U2_STA2_MEAS_CLIENT_CONFIGURATION".ReadLists.U02_STA2_MEAS_Read.NodeHdls, NodeAddInfos :=, Timeout := "DB16103_U2_STA2_MEAS_CLIENT_CONFIGURATION".Connection.ConnectInfo.SessionTimeout, NodeStatusList := "DB16003_U2_STA2_MEAS_CLIENT_INTERFACE".U02_STA2_MEAS_Read.NodeStatusList, TimeStamps := "DB16003_U2_STA2_MEAS_CLIENT_INTERFACE".U02_STA2_MEAS_Read.TimeStamps, Variable := "DB16003_U2_STA2_MEAS_CLIENT_INTERFACE".U02_STA2_MEAS_Read.Variable, Done =>, Busy =>, Error =>, Status =>)
   END_RUNG
   RUNG wire#powerrail
      Contact( "DB16000_OPC_UA_TRIGGER_ALARM".CLIENT.U2_STA2_MEAS.TRIGGERS.READ_VARS )
      P_Trig( "DB16000_OPC_UA_TRIGGER_ALARM".CLIENT.U2_STA2_MEAS.TRIGGERS.READ_VARS_P )
   END_RUNG wire#w1
   // the same network as SCL:
   #_w1 := "DB16000_OPC_UA_TRIGGER_ALARM".CLIENT.U2_STA2_MEAS.TRIGGERS.READ_VARS AND NOT "DB16000_OPC_UA_TRIGGER_ALARM".CLIENT.U2_STA2_MEAS.TRIGGERS.READ_VARS_P;   // rising edge
   "DB16000_OPC_UA_TRIGGER_ALARM".CLIENT.U2_STA2_MEAS.TRIGGERS.READ_VARS_P := "DB16000_OPC_UA_TRIGGER_ALARM".CLIENT.U2_STA2_MEAS.TRIGGERS.READ_VARS;
   "DB16320_READLIST_U2_STA2_MEAS"(REQ := #_w1,   // OPC_UA_ReadList
                           ConnectionHdl := "DB16103_U2_STA2_MEAS_CLIENT_CONFIGURATION".Connection.ConnectionHdl,
                           NodeHdlCount := "DB16103_U2_STA2_MEAS_CLIENT_CONFIGURATION".ReadLists.U02_STA2_MEAS_Read.NodeCount,
                           NodeHdls := "DB16103_U2_STA2_MEAS_CLIENT_CONFIGURATION".ReadLists.U02_STA2_MEAS_Read.NodeHdls,
                           Timeout := "DB16103_U2_STA2_MEAS_CLIENT_CONFIGURATION".Connection.ConnectInfo.SessionTimeout,
                           NodeStatusList := "DB16003_U2_STA2_MEAS_CLIENT_INTERFACE".U02_STA2_MEAS_Read.NodeStatusList,
                           TimeStamps := "DB16003_U2_STA2_MEAS_CLIENT_INTERFACE".U02_STA2_MEAS_Read.TimeStamps,
                           Variable := "DB16003_U2_STA2_MEAS_CLIENT_INTERFACE".U02_STA2_MEAS_Read.Variable);
END_REGION

REGION Network 34: UNIT 2 STATION 2 CONNECTION STATUS CALL
   RUNG wire#powerrail
      "DB16224_CONNECTION_STATUS_U2_STA2_MEAS".OPC_UA_ConnectionGetStatus(REQ := wire#w1, ConnectionHdl := "DB16103_U2_STA2_MEAS_CLIENT_CONFIGURATION".Connection.ConnectionHdl, Timeout := "DB16000_OPC_UA_TRIGGER_ALARM".RECONNECT_TIMEOUT, Done =>, Busy =>, Error =>, Status =>, ConnectionStatus =>, ServerState =>, ServiceLevel =>)
   END_RUNG
   RUNG wire#powerrail
      Contact( "DB16000_OPC_UA_TRIGGER_ALARM".CLIENT.U2_STA2_MEAS.TRIGGERS.CHECK_CONN_STATUS )
      P_Trig( "DB16000_OPC_UA_TRIGGER_ALARM".CLIENT.U2_STA2_MEAS.TRIGGERS.CHECK_CONN_STATUS_P )
   END_RUNG wire#w1
   // the same network as SCL:
   #_w1 := "DB16000_OPC_UA_TRIGGER_ALARM".CLIENT.U2_STA2_MEAS.TRIGGERS.CHECK_CONN_STATUS AND NOT "DB16000_OPC_UA_TRIGGER_ALARM".CLIENT.U2_STA2_MEAS.TRIGGERS.CHECK_CONN_STATUS_P;   // rising edge
   "DB16000_OPC_UA_TRIGGER_ALARM".CLIENT.U2_STA2_MEAS.TRIGGERS.CHECK_CONN_STATUS_P := "DB16000_OPC_UA_TRIGGER_ALARM".CLIENT.U2_STA2_MEAS.TRIGGERS.CHECK_CONN_STATUS;
   "DB16224_CONNECTION_STATUS_U2_STA2_MEAS"(REQ := #_w1,   // OPC_UA_ConnectionGetStatus
                           ConnectionHdl := "DB16103_U2_STA2_MEAS_CLIENT_CONFIGURATION".Connection.ConnectionHdl,
                           Timeout := "DB16000_OPC_UA_TRIGGER_ALARM".RECONNECT_TIMEOUT);
END_REGION

REGION Network 35: UNIT 2 STATION 2 RELEASE HANDLE LIST CALL
   RUNG wire#powerrail
      "DB16225_RELEASE_HANDLE_LIST_U2_STA2_MEAS".OPC_UA_NodeReleaseHandleList(REQ := wire#w1, ConnectionHdl := "DB16103_U2_STA2_MEAS_CLIENT_CONFIGURATION".Connection.ConnectionHdl, NodeHdlCount := "DB16103_U2_STA2_MEAS_CLIENT_CONFIGURATION".ReadLists.U02_STA2_MEAS_Read.NodeCount, NodeHdls := "DB16103_U2_STA2_MEAS_CLIENT_CONFIGURATION".ReadLists.U02_STA2_MEAS_Read.NodeHdls, Timeout := "DB16103_U2_STA2_MEAS_CLIENT_CONFIGURATION".Connection.ConnectInfo.SessionTimeout, NodeStatusList := "DB16003_U2_STA2_MEAS_CLIENT_INTERFACE".U02_STA2_MEAS_Read.NodeStatusList, Done =>, Busy =>, Error =>, Status =>)
   END_RUNG
   RUNG wire#powerrail
      Contact( "DB16000_OPC_UA_TRIGGER_ALARM".CLIENT.U2_STA2_MEAS.TRIGGERS.RELEASE_HANDLE_LIST )
      P_Trig( "DB16000_OPC_UA_TRIGGER_ALARM".CLIENT.U2_STA2_MEAS.TRIGGERS.RELEASE_HANDLE_LIST_P )
   END_RUNG wire#w1
   // the same network as SCL:
   #_w1 := "DB16000_OPC_UA_TRIGGER_ALARM".CLIENT.U2_STA2_MEAS.TRIGGERS.RELEASE_HANDLE_LIST AND NOT "DB16000_OPC_UA_TRIGGER_ALARM".CLIENT.U2_STA2_MEAS.TRIGGERS.RELEASE_HANDLE_LIST_P;   // rising edge
   "DB16000_OPC_UA_TRIGGER_ALARM".CLIENT.U2_STA2_MEAS.TRIGGERS.RELEASE_HANDLE_LIST_P := "DB16000_OPC_UA_TRIGGER_ALARM".CLIENT.U2_STA2_MEAS.TRIGGERS.RELEASE_HANDLE_LIST;
   "DB16225_RELEASE_HANDLE_LIST_U2_STA2_MEAS"(REQ := #_w1,   // OPC_UA_NodeReleaseHandleList
                           ConnectionHdl := "DB16103_U2_STA2_MEAS_CLIENT_CONFIGURATION".Connection.ConnectionHdl,
                           NodeHdlCount := "DB16103_U2_STA2_MEAS_CLIENT_CONFIGURATION".ReadLists.U02_STA2_MEAS_Read.NodeCount,
                           NodeHdls := "DB16103_U2_STA2_MEAS_CLIENT_CONFIGURATION".ReadLists.U02_STA2_MEAS_Read.NodeHdls,
                           Timeout := "DB16103_U2_STA2_MEAS_CLIENT_CONFIGURATION".Connection.ConnectInfo.SessionTimeout,
                           NodeStatusList := "DB16003_U2_STA2_MEAS_CLIENT_INTERFACE".U02_STA2_MEAS_Read.NodeStatusList);
END_REGION

REGION Network 36: UNIT 2 STATION 2 RELEASE METHOD HANDLE LIST CALL
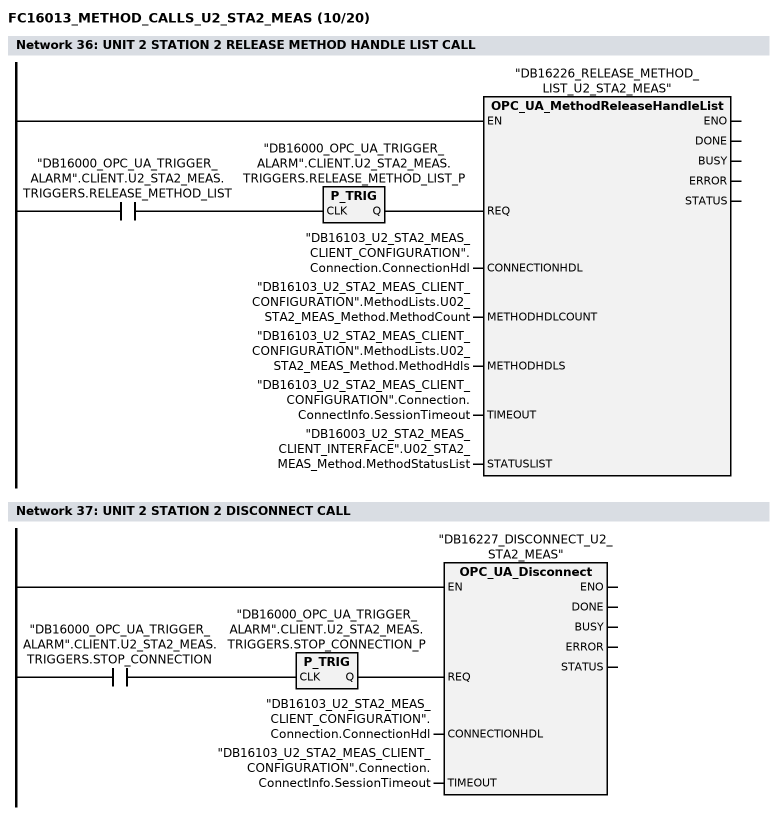
   RUNG wire#powerrail
      "DB16226_RELEASE_METHOD_LIST_U2_STA2_MEAS".OPC_UA_MethodReleaseHandleList(REQ := wire#w1, ConnectionHdl := "DB16103_U2_STA2_MEAS_CLIENT_CONFIGURATION".Connection.ConnectionHdl, MethodHdlCount := "DB16103_U2_STA2_MEAS_CLIENT_CONFIGURATION".MethodLists.U02_STA2_MEAS_Method.MethodCount, MethodHdls := "DB16103_U2_STA2_MEAS_CLIENT_CONFIGURATION".MethodLists.U02_STA2_MEAS_Method.MethodHdls, Timeout := "DB16103_U2_STA2_MEAS_CLIENT_CONFIGURATION".Connection.ConnectInfo.SessionTimeout, StatusList := "DB16003_U2_STA2_MEAS_CLIENT_INTERFACE".U02_STA2_MEAS_Method.MethodStatusList, Done =>, Busy =>, Error =>, Status =>)
   END_RUNG
   RUNG wire#powerrail
      Contact( "DB16000_OPC_UA_TRIGGER_ALARM".CLIENT.U2_STA2_MEAS.TRIGGERS.RELEASE_METHOD_LIST )
      P_Trig( "DB16000_OPC_UA_TRIGGER_ALARM".CLIENT.U2_STA2_MEAS.TRIGGERS.RELEASE_METHOD_LIST_P )
   END_RUNG wire#w1
   // the same network as SCL:
   #_w1 := "DB16000_OPC_UA_TRIGGER_ALARM".CLIENT.U2_STA2_MEAS.TRIGGERS.RELEASE_METHOD_LIST AND NOT "DB16000_OPC_UA_TRIGGER_ALARM".CLIENT.U2_STA2_MEAS.TRIGGERS.RELEASE_METHOD_LIST_P;   // rising edge
   "DB16000_OPC_UA_TRIGGER_ALARM".CLIENT.U2_STA2_MEAS.TRIGGERS.RELEASE_METHOD_LIST_P := "DB16000_OPC_UA_TRIGGER_ALARM".CLIENT.U2_STA2_MEAS.TRIGGERS.RELEASE_METHOD_LIST;
   "DB16226_RELEASE_METHOD_LIST_U2_STA2_MEAS"(REQ := #_w1,   // OPC_UA_MethodReleaseHandleList
                           ConnectionHdl := "DB16103_U2_STA2_MEAS_CLIENT_CONFIGURATION".Connection.ConnectionHdl,
                           MethodHdlCount := "DB16103_U2_STA2_MEAS_CLIENT_CONFIGURATION".MethodLists.U02_STA2_MEAS_Method.MethodCount,
                           MethodHdls := "DB16103_U2_STA2_MEAS_CLIENT_CONFIGURATION".MethodLists.U02_STA2_MEAS_Method.MethodHdls,
                           Timeout := "DB16103_U2_STA2_MEAS_CLIENT_CONFIGURATION".Connection.ConnectInfo.SessionTimeout,
                           StatusList := "DB16003_U2_STA2_MEAS_CLIENT_INTERFACE".U02_STA2_MEAS_Method.MethodStatusList);
END_REGION

REGION Network 37: UNIT 2 STATION 2 DISCONNECT CALL
   RUNG wire#powerrail
      "DB16227_DISCONNECT_U2_STA2_MEAS".OPC_UA_Disconnect(REQ := wire#w1, ConnectionHdl := "DB16103_U2_STA2_MEAS_CLIENT_CONFIGURATION".Connection.ConnectionHdl, Timeout := "DB16103_U2_STA2_MEAS_CLIENT_CONFIGURATION".Connection.ConnectInfo.SessionTimeout, Done =>, Busy =>, Error =>, Status =>)
   END_RUNG
   RUNG wire#powerrail
      Contact( "DB16000_OPC_UA_TRIGGER_ALARM".CLIENT.U2_STA2_MEAS.TRIGGERS.STOP_CONNECTION )
      P_Trig( "DB16000_OPC_UA_TRIGGER_ALARM".CLIENT.U2_STA2_MEAS.TRIGGERS.STOP_CONNECTION_P )
   END_RUNG wire#w1
   // the same network as SCL:
   #_w1 := "DB16000_OPC_UA_TRIGGER_ALARM".CLIENT.U2_STA2_MEAS.TRIGGERS.STOP_CONNECTION AND NOT "DB16000_OPC_UA_TRIGGER_ALARM".CLIENT.U2_STA2_MEAS.TRIGGERS.STOP_CONNECTION_P;   // rising edge
   "DB16000_OPC_UA_TRIGGER_ALARM".CLIENT.U2_STA2_MEAS.TRIGGERS.STOP_CONNECTION_P := "DB16000_OPC_UA_TRIGGER_ALARM".CLIENT.U2_STA2_MEAS.TRIGGERS.STOP_CONNECTION;
   "DB16227_DISCONNECT_U2_STA2_MEAS"(REQ := #_w1,   // OPC_UA_Disconnect
                           ConnectionHdl := "DB16103_U2_STA2_MEAS_CLIENT_CONFIGURATION".Connection.ConnectionHdl,
                           Timeout := "DB16103_U2_STA2_MEAS_CLIENT_CONFIGURATION".Connection.ConnectInfo.SessionTimeout);
END_REGION

REGION Network 38: UNIT 2 STATION 2 MEAS RECONNECT
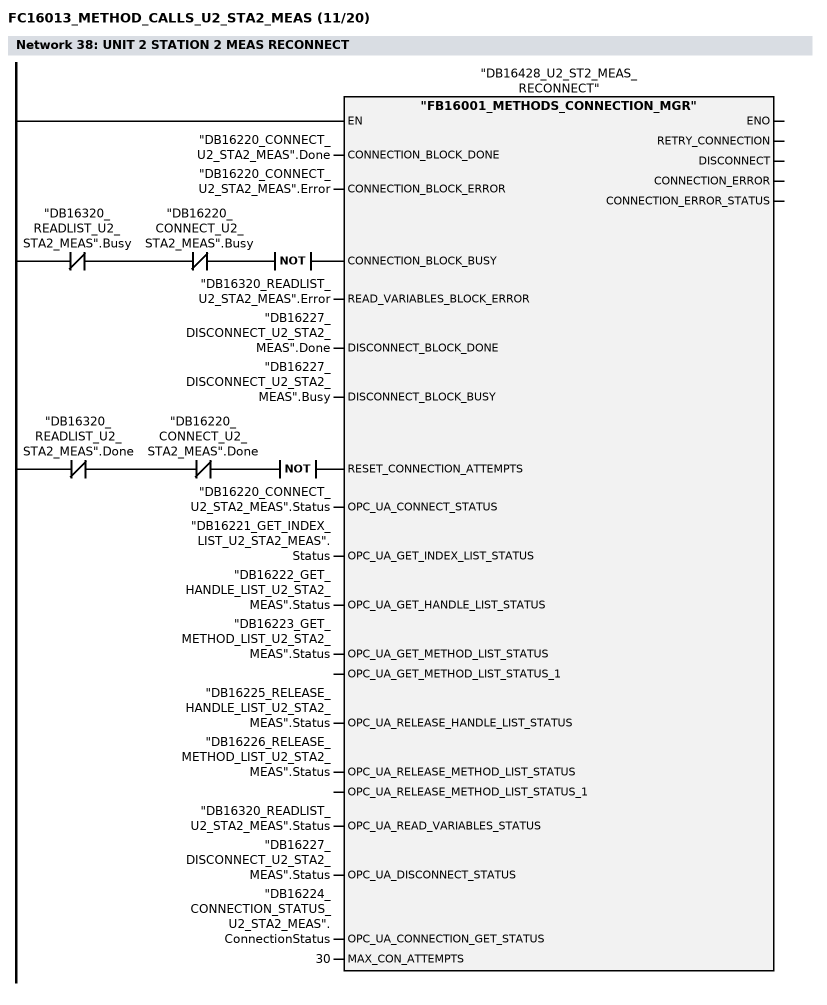
   RUNG wire#powerrail
      "DB16428_U2_ST2_MEAS_RECONNECT"(CONNECTION_BLOCK_BUSY := wire#w1, RESET_CONNECTION_ATTEMPTS := wire#w2, CONNECTION_BLOCK_DONE := "DB16220_CONNECT_U2_STA2_MEAS".Done, CONNECTION_BLOCK_ERROR := "DB16220_CONNECT_U2_STA2_MEAS".Error, READ_VARIABLES_BLOCK_ERROR := "DB16320_READLIST_U2_STA2_MEAS".Error, DISCONNECT_BLOCK_DONE := "DB16227_DISCONNECT_U2_STA2_MEAS".Done, DISCONNECT_BLOCK_BUSY := "DB16227_DISCONNECT_U2_STA2_MEAS".Busy, OPC_UA_CONNECT_STATUS := "DB16220_CONNECT_U2_STA2_MEAS".Status, OPC_UA_GET_INDEX_LIST_STATUS := "DB16221_GET_INDEX_LIST_U2_STA2_MEAS".Status, OPC_UA_GET_HANDLE_LIST_STATUS := "DB16222_GET_HANDLE_LIST_U2_STA2_MEAS".Status, OPC_UA_GET_METHOD_LIST_STATUS := "DB16223_GET_METHOD_LIST_U2_STA2_MEAS".Status, OPC_UA_GET_METHOD_LIST_STATUS_1 :=, OPC_UA_RELEASE_HANDLE_LIST_STATUS := "DB16225_RELEASE_HANDLE_LIST_U2_STA2_MEAS".Status, OPC_UA_RELEASE_METHOD_LIST_STATUS := "DB16226_RELEASE_METHOD_LIST_U2_STA2_MEAS".Status, OPC_UA_RELEASE_METHOD_LIST_STATUS_1 :=, OPC_UA_READ_VARIABLES_STATUS := "DB16320_READLIST_U2_STA2_MEAS".Status, OPC_UA_DISCONNECT_STATUS := "DB16227_DISCONNECT_U2_STA2_MEAS".Status, OPC_UA_CONNECTION_GET_STATUS := "DB16224_CONNECTION_STATUS_U2_STA2_MEAS".ConnectionStatus, MAX_CON_ATTEMPTS := 30, RETRY_CONNECTION =>, DISCONNECT =>, CONNECTION_ERROR =>, CONNECTION_ERROR_STATUS =>)
   END_RUNG
   RUNG wire#powerrail
      I_Contact( "DB16320_READLIST_U2_STA2_MEAS".Busy )
      I_Contact( "DB16220_CONNECT_U2_STA2_MEAS".Busy )
      Not()
   END_RUNG wire#w1
   RUNG wire#powerrail
      I_Contact( "DB16320_READLIST_U2_STA2_MEAS".Done )
      I_Contact( "DB16220_CONNECT_U2_STA2_MEAS".Done )
      Not()
   END_RUNG wire#w2
   // the same network as SCL:
   "DB16428_U2_ST2_MEAS_RECONNECT"(CONNECTION_BLOCK_DONE := "DB16220_CONNECT_U2_STA2_MEAS".Done,   // "FB16001_METHODS_CONNECTION_MGR"
                           CONNECTION_BLOCK_ERROR := "DB16220_CONNECT_U2_STA2_MEAS".Error,
                           CONNECTION_BLOCK_BUSY := NOT (NOT "DB16320_READLIST_U2_STA2_MEAS".Busy AND NOT "DB16220_CONNECT_U2_STA2_MEAS".Busy),
                           READ_VARIABLES_BLOCK_ERROR := "DB16320_READLIST_U2_STA2_MEAS".Error,
                           DISCONNECT_BLOCK_DONE := "DB16227_DISCONNECT_U2_STA2_MEAS".Done,
                           DISCONNECT_BLOCK_BUSY := "DB16227_DISCONNECT_U2_STA2_MEAS".Busy,
                           RESET_CONNECTION_ATTEMPTS := NOT (NOT "DB16320_READLIST_U2_STA2_MEAS".Done AND NOT "DB16220_CONNECT_U2_STA2_MEAS".Done),
                           OPC_UA_CONNECT_STATUS := "DB16220_CONNECT_U2_STA2_MEAS".Status,
                           OPC_UA_GET_INDEX_LIST_STATUS := "DB16221_GET_INDEX_LIST_U2_STA2_MEAS".Status,
                           OPC_UA_GET_HANDLE_LIST_STATUS := "DB16222_GET_HANDLE_LIST_U2_STA2_MEAS".Status,
                           OPC_UA_GET_METHOD_LIST_STATUS := "DB16223_GET_METHOD_LIST_U2_STA2_MEAS".Status,
                           OPC_UA_RELEASE_HANDLE_LIST_STATUS := "DB16225_RELEASE_HANDLE_LIST_U2_STA2_MEAS".Status,
                           OPC_UA_RELEASE_METHOD_LIST_STATUS := "DB16226_RELEASE_METHOD_LIST_U2_STA2_MEAS".Status,
                           OPC_UA_READ_VARIABLES_STATUS := "DB16320_READLIST_U2_STA2_MEAS".Status,
                           OPC_UA_DISCONNECT_STATUS := "DB16227_DISCONNECT_U2_STA2_MEAS".Status,
                           OPC_UA_CONNECTION_GET_STATUS := "DB16224_CONNECTION_STATUS_U2_STA2_MEAS".ConnectionStatus,
                           MAX_CON_ATTEMPTS := 30);
END_REGION

REGION Network 39: UNIT 2 FIXTURES CALIBRATION STATUS UPDATE
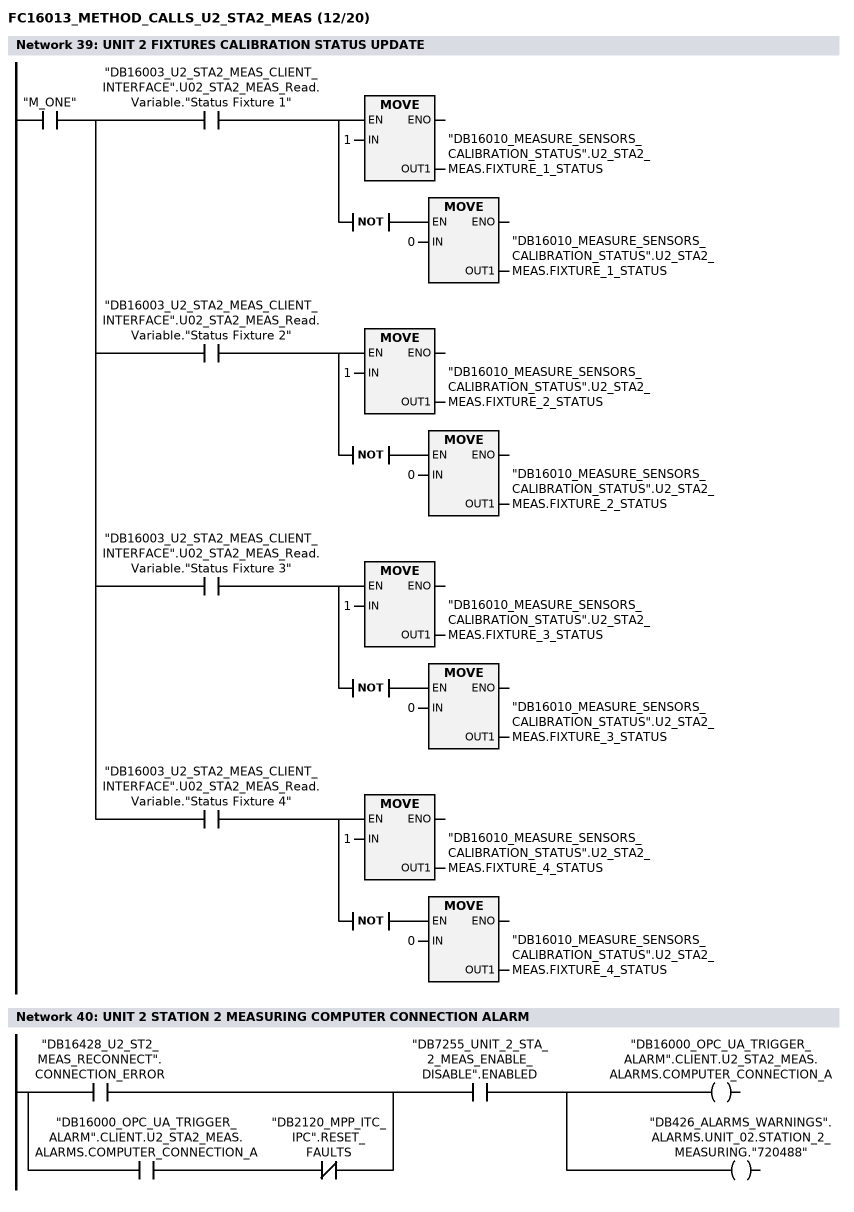
   RUNG wire#powerrail
      Contact( "M_ONE" )
      wire#w1
      Contact( "DB16003_U2_STA2_MEAS_CLIENT_INTERFACE".U02_STA2_MEAS_Read.Variable."Status Fixture 1" )
      wire#w2
      Move(in := 1, out1 => "DB16010_MEASURE_SENSORS_CALIBRATION_STATUS".U2_STA2_MEAS.FIXTURE_1_STATUS)
   END_RUNG
   RUNG wire#w2
      Not()
      Move(in := 0, out1 => "DB16010_MEASURE_SENSORS_CALIBRATION_STATUS".U2_STA2_MEAS.FIXTURE_1_STATUS)
   END_RUNG
   RUNG wire#w1
      Contact( "DB16003_U2_STA2_MEAS_CLIENT_INTERFACE".U02_STA2_MEAS_Read.Variable."Status Fixture 2" )
      wire#w3
      Move(in := 1, out1 => "DB16010_MEASURE_SENSORS_CALIBRATION_STATUS".U2_STA2_MEAS.FIXTURE_2_STATUS)
   END_RUNG
   RUNG wire#w3
      Not()
      Move(in := 0, out1 => "DB16010_MEASURE_SENSORS_CALIBRATION_STATUS".U2_STA2_MEAS.FIXTURE_2_STATUS)
   END_RUNG
   RUNG wire#w1
      Contact( "DB16003_U2_STA2_MEAS_CLIENT_INTERFACE".U02_STA2_MEAS_Read.Variable."Status Fixture 3" )
      wire#w4
      Move(in := 1, out1 => "DB16010_MEASURE_SENSORS_CALIBRATION_STATUS".U2_STA2_MEAS.FIXTURE_3_STATUS)
   END_RUNG
   RUNG wire#w4
      Not()
      Move(in := 0, out1 => "DB16010_MEASURE_SENSORS_CALIBRATION_STATUS".U2_STA2_MEAS.FIXTURE_3_STATUS)
   END_RUNG
   RUNG wire#w1
      Contact( "DB16003_U2_STA2_MEAS_CLIENT_INTERFACE".U02_STA2_MEAS_Read.Variable."Status Fixture 4" )
      wire#w5
      Move(in := 1, out1 => "DB16010_MEASURE_SENSORS_CALIBRATION_STATUS".U2_STA2_MEAS.FIXTURE_4_STATUS)
   END_RUNG
   RUNG wire#w5
      Not()
      Move(in := 0, out1 => "DB16010_MEASURE_SENSORS_CALIBRATION_STATUS".U2_STA2_MEAS.FIXTURE_4_STATUS)
   END_RUNG
   // the same network as SCL:
   #_w1 := "M_ONE" AND "DB16003_U2_STA2_MEAS_CLIENT_INTERFACE".U02_STA2_MEAS_Read.Variable."Status Fixture 1";
   IF #_w1 THEN "DB16010_MEASURE_SENSORS_CALIBRATION_STATUS".U2_STA2_MEAS.FIXTURE_1_STATUS := 1; END_IF;
   IF NOT #_w1 THEN "DB16010_MEASURE_SENSORS_CALIBRATION_STATUS".U2_STA2_MEAS.FIXTURE_1_STATUS := 0; END_IF;
   #_w2 := "M_ONE" AND "DB16003_U2_STA2_MEAS_CLIENT_INTERFACE".U02_STA2_MEAS_Read.Variable."Status Fixture 2";
   IF #_w2 THEN "DB16010_MEASURE_SENSORS_CALIBRATION_STATUS".U2_STA2_MEAS.FIXTURE_2_STATUS := 1; END_IF;
   IF NOT #_w2 THEN "DB16010_MEASURE_SENSORS_CALIBRATION_STATUS".U2_STA2_MEAS.FIXTURE_2_STATUS := 0; END_IF;
   #_w3 := "M_ONE" AND "DB16003_U2_STA2_MEAS_CLIENT_INTERFACE".U02_STA2_MEAS_Read.Variable."Status Fixture 3";
   IF #_w3 THEN "DB16010_MEASURE_SENSORS_CALIBRATION_STATUS".U2_STA2_MEAS.FIXTURE_3_STATUS := 1; END_IF;
   IF NOT #_w3 THEN "DB16010_MEASURE_SENSORS_CALIBRATION_STATUS".U2_STA2_MEAS.FIXTURE_3_STATUS := 0; END_IF;
   #_w4 := "M_ONE" AND "DB16003_U2_STA2_MEAS_CLIENT_INTERFACE".U02_STA2_MEAS_Read.Variable."Status Fixture 4";
   IF #_w4 THEN "DB16010_MEASURE_SENSORS_CALIBRATION_STATUS".U2_STA2_MEAS.FIXTURE_4_STATUS := 1; END_IF;
   IF NOT #_w4 THEN "DB16010_MEASURE_SENSORS_CALIBRATION_STATUS".U2_STA2_MEAS.FIXTURE_4_STATUS := 0; END_IF;
END_REGION

REGION Network 40: UNIT 2 STATION 2 MEASURING COMPUTER CONNECTION ALARM
   RUNG wire#powerrail
      Contact( "DB16428_U2_ST2_MEAS_RECONNECT".CONNECTION_ERROR )
      wire#w1
      Contact( "DB7255_UNIT_2_STA_2_MEAS_ENABLE_DISABLE".ENABLED )
      wire#w2
      Coil( "DB16000_OPC_UA_TRIGGER_ALARM".CLIENT.U2_STA2_MEAS.ALARMS.COMPUTER_CONNECTION_A )
   END_RUNG
   RUNG wire#powerrail
      Contact( "DB16000_OPC_UA_TRIGGER_ALARM".CLIENT.U2_STA2_MEAS.ALARMS.COMPUTER_CONNECTION_A )
      I_Contact( "DB2120_MPP_ITC_IPC".RESET_FAULTS )
   END_RUNG wire#w1
   RUNG wire#w2
      Coil( "DB426_ALARMS_WARNINGS".ALARMS.UNIT_02.STATION_2_MEASURING."720488" )
   END_RUNG
   // the same network as SCL:
   "DB16000_OPC_UA_TRIGGER_ALARM".CLIENT.U2_STA2_MEAS.ALARMS.COMPUTER_CONNECTION_A := ("DB16428_U2_ST2_MEAS_RECONNECT".CONNECTION_ERROR OR ("DB16000_OPC_UA_TRIGGER_ALARM".CLIENT.U2_STA2_MEAS.ALARMS.COMPUTER_CONNECTION_A AND NOT "DB2120_MPP_ITC_IPC".RESET_FAULTS)) AND "DB7255_UNIT_2_STA_2_MEAS_ENABLE_DISABLE".ENABLED;
   "DB426_ALARMS_WARNINGS".ALARMS.UNIT_02.STATION_2_MEASURING."720488" := "DB16000_OPC_UA_TRIGGER_ALARM".CLIENT.U2_STA2_MEAS.ALARMS.COMPUTER_CONNECTION_A;
END_REGION

REGION Network 41: UNIT 2 STATION 2 MEASURING COMPUTER GET INDEX LIST ALARM
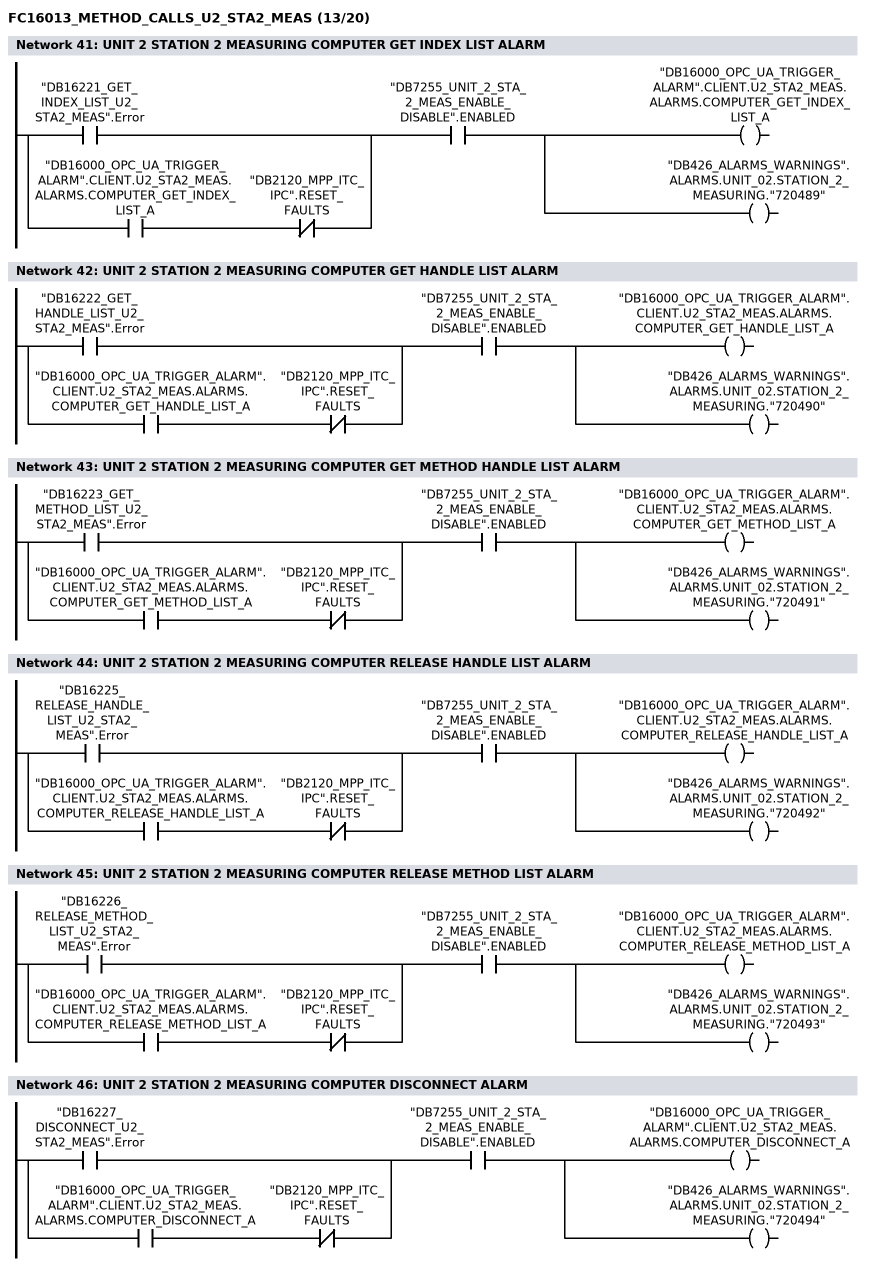
   RUNG wire#powerrail
      Contact( "DB16221_GET_INDEX_LIST_U2_STA2_MEAS".Error )
      wire#w1
      Contact( "DB7255_UNIT_2_STA_2_MEAS_ENABLE_DISABLE".ENABLED )
      wire#w2
      Coil( "DB16000_OPC_UA_TRIGGER_ALARM".CLIENT.U2_STA2_MEAS.ALARMS.COMPUTER_GET_INDEX_LIST_A )
   END_RUNG
   RUNG wire#powerrail
      Contact( "DB16000_OPC_UA_TRIGGER_ALARM".CLIENT.U2_STA2_MEAS.ALARMS.COMPUTER_GET_INDEX_LIST_A )
      I_Contact( "DB2120_MPP_ITC_IPC".RESET_FAULTS )
   END_RUNG wire#w1
   RUNG wire#w2
      Coil( "DB426_ALARMS_WARNINGS".ALARMS.UNIT_02.STATION_2_MEASURING."720489" )
   END_RUNG
   // the same network as SCL:
   "DB16000_OPC_UA_TRIGGER_ALARM".CLIENT.U2_STA2_MEAS.ALARMS.COMPUTER_GET_INDEX_LIST_A := ("DB16221_GET_INDEX_LIST_U2_STA2_MEAS".Error OR ("DB16000_OPC_UA_TRIGGER_ALARM".CLIENT.U2_STA2_MEAS.ALARMS.COMPUTER_GET_INDEX_LIST_A AND NOT "DB2120_MPP_ITC_IPC".RESET_FAULTS)) AND "DB7255_UNIT_2_STA_2_MEAS_ENABLE_DISABLE".ENABLED;
   "DB426_ALARMS_WARNINGS".ALARMS.UNIT_02.STATION_2_MEASURING."720489" := "DB16000_OPC_UA_TRIGGER_ALARM".CLIENT.U2_STA2_MEAS.ALARMS.COMPUTER_GET_INDEX_LIST_A;
END_REGION

REGION Network 42: UNIT 2 STATION 2 MEASURING COMPUTER GET HANDLE LIST ALARM
   RUNG wire#powerrail
      Contact( "DB16222_GET_HANDLE_LIST_U2_STA2_MEAS".Error )
      wire#w1
      Contact( "DB7255_UNIT_2_STA_2_MEAS_ENABLE_DISABLE".ENABLED )
      wire#w2
      Coil( "DB16000_OPC_UA_TRIGGER_ALARM".CLIENT.U2_STA2_MEAS.ALARMS.COMPUTER_GET_HANDLE_LIST_A )
   END_RUNG
   RUNG wire#powerrail
      Contact( "DB16000_OPC_UA_TRIGGER_ALARM".CLIENT.U2_STA2_MEAS.ALARMS.COMPUTER_GET_HANDLE_LIST_A )
      I_Contact( "DB2120_MPP_ITC_IPC".RESET_FAULTS )
   END_RUNG wire#w1
   RUNG wire#w2
      Coil( "DB426_ALARMS_WARNINGS".ALARMS.UNIT_02.STATION_2_MEASURING."720490" )
   END_RUNG
   // the same network as SCL:
   "DB16000_OPC_UA_TRIGGER_ALARM".CLIENT.U2_STA2_MEAS.ALARMS.COMPUTER_GET_HANDLE_LIST_A := ("DB16222_GET_HANDLE_LIST_U2_STA2_MEAS".Error OR ("DB16000_OPC_UA_TRIGGER_ALARM".CLIENT.U2_STA2_MEAS.ALARMS.COMPUTER_GET_HANDLE_LIST_A AND NOT "DB2120_MPP_ITC_IPC".RESET_FAULTS)) AND "DB7255_UNIT_2_STA_2_MEAS_ENABLE_DISABLE".ENABLED;
   "DB426_ALARMS_WARNINGS".ALARMS.UNIT_02.STATION_2_MEASURING."720490" := "DB16000_OPC_UA_TRIGGER_ALARM".CLIENT.U2_STA2_MEAS.ALARMS.COMPUTER_GET_HANDLE_LIST_A;
END_REGION

REGION Network 43: UNIT 2 STATION 2 MEASURING COMPUTER GET METHOD HANDLE LIST ALARM
   RUNG wire#powerrail
      Contact( "DB16223_GET_METHOD_LIST_U2_STA2_MEAS".Error )
      wire#w1
      Contact( "DB7255_UNIT_2_STA_2_MEAS_ENABLE_DISABLE".ENABLED )
      wire#w2
      Coil( "DB16000_OPC_UA_TRIGGER_ALARM".CLIENT.U2_STA2_MEAS.ALARMS.COMPUTER_GET_METHOD_LIST_A )
   END_RUNG
   RUNG wire#powerrail
      Contact( "DB16000_OPC_UA_TRIGGER_ALARM".CLIENT.U2_STA2_MEAS.ALARMS.COMPUTER_GET_METHOD_LIST_A )
      I_Contact( "DB2120_MPP_ITC_IPC".RESET_FAULTS )
   END_RUNG wire#w1
   RUNG wire#w2
      Coil( "DB426_ALARMS_WARNINGS".ALARMS.UNIT_02.STATION_2_MEASURING."720491" )
   END_RUNG
   // the same network as SCL:
   "DB16000_OPC_UA_TRIGGER_ALARM".CLIENT.U2_STA2_MEAS.ALARMS.COMPUTER_GET_METHOD_LIST_A := ("DB16223_GET_METHOD_LIST_U2_STA2_MEAS".Error OR ("DB16000_OPC_UA_TRIGGER_ALARM".CLIENT.U2_STA2_MEAS.ALARMS.COMPUTER_GET_METHOD_LIST_A AND NOT "DB2120_MPP_ITC_IPC".RESET_FAULTS)) AND "DB7255_UNIT_2_STA_2_MEAS_ENABLE_DISABLE".ENABLED;
   "DB426_ALARMS_WARNINGS".ALARMS.UNIT_02.STATION_2_MEASURING."720491" := "DB16000_OPC_UA_TRIGGER_ALARM".CLIENT.U2_STA2_MEAS.ALARMS.COMPUTER_GET_METHOD_LIST_A;
END_REGION

REGION Network 44: UNIT 2 STATION 2 MEASURING COMPUTER RELEASE HANDLE LIST ALARM
   RUNG wire#powerrail
      Contact( "DB16225_RELEASE_HANDLE_LIST_U2_STA2_MEAS".Error )
      wire#w1
      Contact( "DB7255_UNIT_2_STA_2_MEAS_ENABLE_DISABLE".ENABLED )
      wire#w2
      Coil( "DB16000_OPC_UA_TRIGGER_ALARM".CLIENT.U2_STA2_MEAS.ALARMS.COMPUTER_RELEASE_HANDLE_LIST_A )
   END_RUNG
   RUNG wire#powerrail
      Contact( "DB16000_OPC_UA_TRIGGER_ALARM".CLIENT.U2_STA2_MEAS.ALARMS.COMPUTER_RELEASE_HANDLE_LIST_A )
      I_Contact( "DB2120_MPP_ITC_IPC".RESET_FAULTS )
   END_RUNG wire#w1
   RUNG wire#w2
      Coil( "DB426_ALARMS_WARNINGS".ALARMS.UNIT_02.STATION_2_MEASURING."720492" )
   END_RUNG
   // the same network as SCL:
   "DB16000_OPC_UA_TRIGGER_ALARM".CLIENT.U2_STA2_MEAS.ALARMS.COMPUTER_RELEASE_HANDLE_LIST_A := ("DB16225_RELEASE_HANDLE_LIST_U2_STA2_MEAS".Error OR ("DB16000_OPC_UA_TRIGGER_ALARM".CLIENT.U2_STA2_MEAS.ALARMS.COMPUTER_RELEASE_HANDLE_LIST_A AND NOT "DB2120_MPP_ITC_IPC".RESET_FAULTS)) AND "DB7255_UNIT_2_STA_2_MEAS_ENABLE_DISABLE".ENABLED;
   "DB426_ALARMS_WARNINGS".ALARMS.UNIT_02.STATION_2_MEASURING."720492" := "DB16000_OPC_UA_TRIGGER_ALARM".CLIENT.U2_STA2_MEAS.ALARMS.COMPUTER_RELEASE_HANDLE_LIST_A;
END_REGION

REGION Network 45: UNIT 2 STATION 2 MEASURING COMPUTER RELEASE METHOD LIST ALARM
   RUNG wire#powerrail
      Contact( "DB16226_RELEASE_METHOD_LIST_U2_STA2_MEAS".Error )
      wire#w1
      Contact( "DB7255_UNIT_2_STA_2_MEAS_ENABLE_DISABLE".ENABLED )
      wire#w2
      Coil( "DB16000_OPC_UA_TRIGGER_ALARM".CLIENT.U2_STA2_MEAS.ALARMS.COMPUTER_RELEASE_METHOD_LIST_A )
   END_RUNG
   RUNG wire#powerrail
      Contact( "DB16000_OPC_UA_TRIGGER_ALARM".CLIENT.U2_STA2_MEAS.ALARMS.COMPUTER_RELEASE_METHOD_LIST_A )
      I_Contact( "DB2120_MPP_ITC_IPC".RESET_FAULTS )
   END_RUNG wire#w1
   RUNG wire#w2
      Coil( "DB426_ALARMS_WARNINGS".ALARMS.UNIT_02.STATION_2_MEASURING."720493" )
   END_RUNG
   // the same network as SCL:
   "DB16000_OPC_UA_TRIGGER_ALARM".CLIENT.U2_STA2_MEAS.ALARMS.COMPUTER_RELEASE_METHOD_LIST_A := ("DB16226_RELEASE_METHOD_LIST_U2_STA2_MEAS".Error OR ("DB16000_OPC_UA_TRIGGER_ALARM".CLIENT.U2_STA2_MEAS.ALARMS.COMPUTER_RELEASE_METHOD_LIST_A AND NOT "DB2120_MPP_ITC_IPC".RESET_FAULTS)) AND "DB7255_UNIT_2_STA_2_MEAS_ENABLE_DISABLE".ENABLED;
   "DB426_ALARMS_WARNINGS".ALARMS.UNIT_02.STATION_2_MEASURING."720493" := "DB16000_OPC_UA_TRIGGER_ALARM".CLIENT.U2_STA2_MEAS.ALARMS.COMPUTER_RELEASE_METHOD_LIST_A;
END_REGION

REGION Network 46: UNIT 2 STATION 2 MEASURING COMPUTER DISCONNECT ALARM
   RUNG wire#powerrail
      Contact( "DB16227_DISCONNECT_U2_STA2_MEAS".Error )
      wire#w1
      Contact( "DB7255_UNIT_2_STA_2_MEAS_ENABLE_DISABLE".ENABLED )
      wire#w2
      Coil( "DB16000_OPC_UA_TRIGGER_ALARM".CLIENT.U2_STA2_MEAS.ALARMS.COMPUTER_DISCONNECT_A )
   END_RUNG
   RUNG wire#powerrail
      Contact( "DB16000_OPC_UA_TRIGGER_ALARM".CLIENT.U2_STA2_MEAS.ALARMS.COMPUTER_DISCONNECT_A )
      I_Contact( "DB2120_MPP_ITC_IPC".RESET_FAULTS )
   END_RUNG wire#w1
   RUNG wire#w2
      Coil( "DB426_ALARMS_WARNINGS".ALARMS.UNIT_02.STATION_2_MEASURING."720494" )
   END_RUNG
   // the same network as SCL:
   "DB16000_OPC_UA_TRIGGER_ALARM".CLIENT.U2_STA2_MEAS.ALARMS.COMPUTER_DISCONNECT_A := ("DB16227_DISCONNECT_U2_STA2_MEAS".Error OR ("DB16000_OPC_UA_TRIGGER_ALARM".CLIENT.U2_STA2_MEAS.ALARMS.COMPUTER_DISCONNECT_A AND NOT "DB2120_MPP_ITC_IPC".RESET_FAULTS)) AND "DB7255_UNIT_2_STA_2_MEAS_ENABLE_DISABLE".ENABLED;
   "DB426_ALARMS_WARNINGS".ALARMS.UNIT_02.STATION_2_MEASURING."720494" := "DB16000_OPC_UA_TRIGGER_ALARM".CLIENT.U2_STA2_MEAS.ALARMS.COMPUTER_DISCONNECT_A;
END_REGION

REGION Network 47: UNIT 2 STATION 2 MEASURING METHOD CONNECTION ALARM
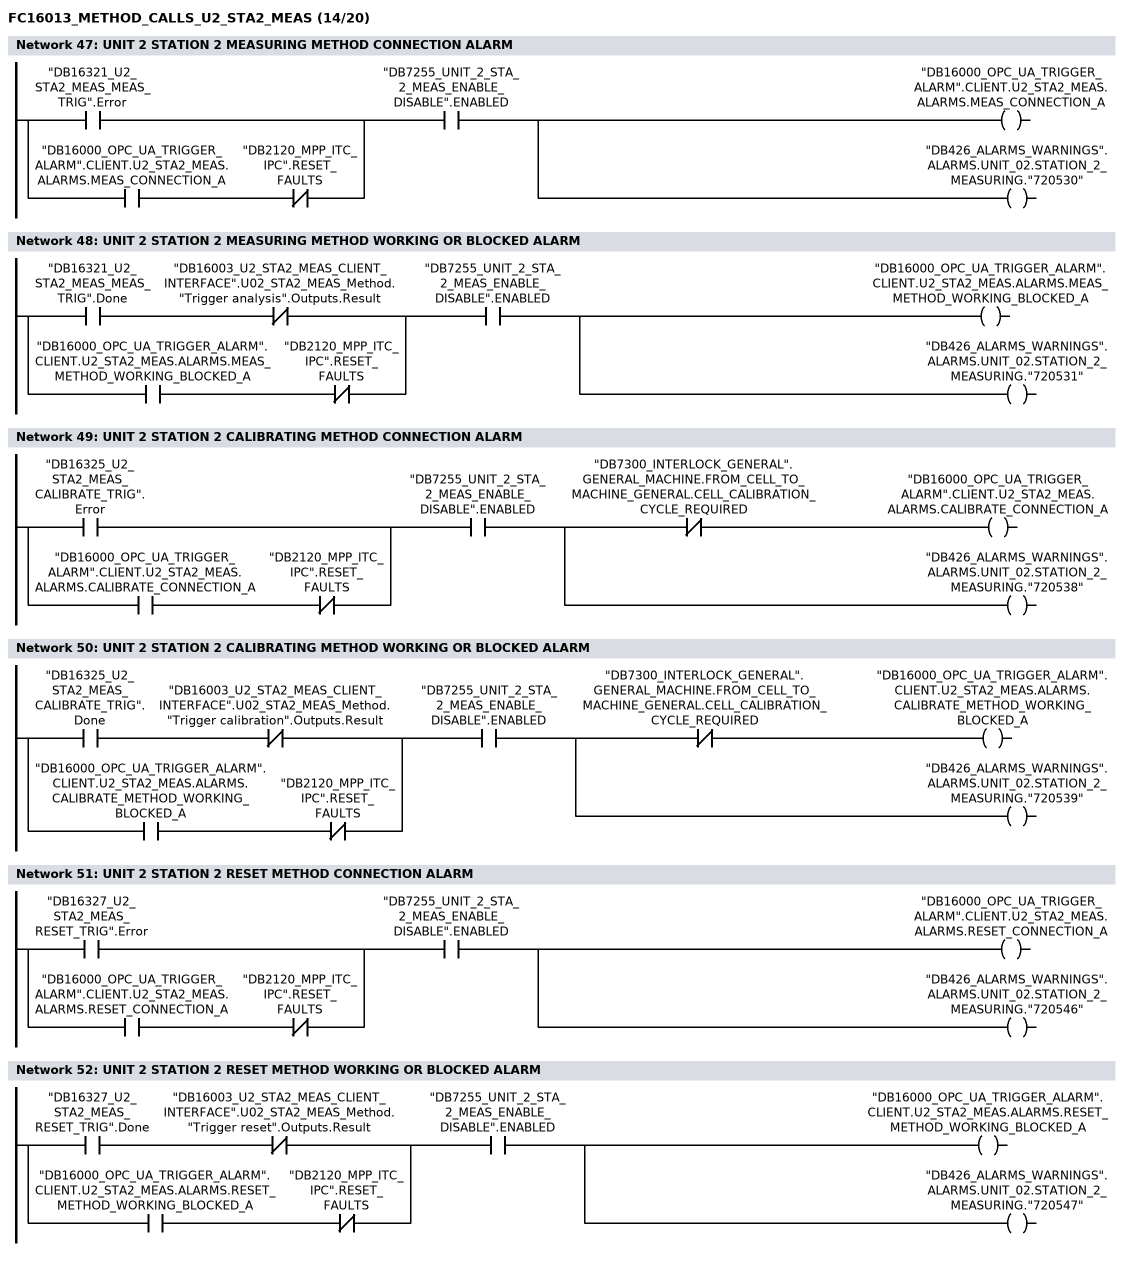
   RUNG wire#powerrail
      Contact( "DB16321_U2_STA2_MEAS_MEAS_TRIG".Error )
      wire#w1
      Contact( "DB7255_UNIT_2_STA_2_MEAS_ENABLE_DISABLE".ENABLED )
      wire#w2
      Coil( "DB16000_OPC_UA_TRIGGER_ALARM".CLIENT.U2_STA2_MEAS.ALARMS.MEAS_CONNECTION_A )
   END_RUNG
   RUNG wire#powerrail
      Contact( "DB16000_OPC_UA_TRIGGER_ALARM".CLIENT.U2_STA2_MEAS.ALARMS.MEAS_CONNECTION_A )
      I_Contact( "DB2120_MPP_ITC_IPC".RESET_FAULTS )
   END_RUNG wire#w1
   RUNG wire#w2
      Coil( "DB426_ALARMS_WARNINGS".ALARMS.UNIT_02.STATION_2_MEASURING."720530" )
   END_RUNG
   // the same network as SCL:
   "DB16000_OPC_UA_TRIGGER_ALARM".CLIENT.U2_STA2_MEAS.ALARMS.MEAS_CONNECTION_A := ("DB16321_U2_STA2_MEAS_MEAS_TRIG".Error OR ("DB16000_OPC_UA_TRIGGER_ALARM".CLIENT.U2_STA2_MEAS.ALARMS.MEAS_CONNECTION_A AND NOT "DB2120_MPP_ITC_IPC".RESET_FAULTS)) AND "DB7255_UNIT_2_STA_2_MEAS_ENABLE_DISABLE".ENABLED;
   "DB426_ALARMS_WARNINGS".ALARMS.UNIT_02.STATION_2_MEASURING."720530" := "DB16000_OPC_UA_TRIGGER_ALARM".CLIENT.U2_STA2_MEAS.ALARMS.MEAS_CONNECTION_A;
END_REGION

REGION Network 48: UNIT 2 STATION 2 MEASURING METHOD WORKING OR BLOCKED ALARM
   RUNG wire#powerrail
      Contact( "DB16321_U2_STA2_MEAS_MEAS_TRIG".Done )
      I_Contact( "DB16003_U2_STA2_MEAS_CLIENT_INTERFACE".U02_STA2_MEAS_Method."Trigger analysis".Outputs.Result )
      wire#w1
      Contact( "DB7255_UNIT_2_STA_2_MEAS_ENABLE_DISABLE".ENABLED )
      wire#w2
      Coil( "DB16000_OPC_UA_TRIGGER_ALARM".CLIENT.U2_STA2_MEAS.ALARMS.MEAS_METHOD_WORKING_BLOCKED_A )
   END_RUNG
   RUNG wire#powerrail
      Contact( "DB16000_OPC_UA_TRIGGER_ALARM".CLIENT.U2_STA2_MEAS.ALARMS.MEAS_METHOD_WORKING_BLOCKED_A )
      I_Contact( "DB2120_MPP_ITC_IPC".RESET_FAULTS )
   END_RUNG wire#w1
   RUNG wire#w2
      Coil( "DB426_ALARMS_WARNINGS".ALARMS.UNIT_02.STATION_2_MEASURING."720531" )
   END_RUNG
   // the same network as SCL:
   "DB16000_OPC_UA_TRIGGER_ALARM".CLIENT.U2_STA2_MEAS.ALARMS.MEAS_METHOD_WORKING_BLOCKED_A := (("DB16321_U2_STA2_MEAS_MEAS_TRIG".Done AND NOT "DB16003_U2_STA2_MEAS_CLIENT_INTERFACE".U02_STA2_MEAS_Method."Trigger analysis".Outputs.Result) OR ("DB16000_OPC_UA_TRIGGER_ALARM".CLIENT.U2_STA2_MEAS.ALARMS.MEAS_METHOD_WORKING_BLOCKED_A AND NOT "DB2120_MPP_ITC_IPC".RESET_FAULTS)) AND "DB7255_UNIT_2_STA_2_MEAS_ENABLE_DISABLE".ENABLED;
   "DB426_ALARMS_WARNINGS".ALARMS.UNIT_02.STATION_2_MEASURING."720531" := "DB16000_OPC_UA_TRIGGER_ALARM".CLIENT.U2_STA2_MEAS.ALARMS.MEAS_METHOD_WORKING_BLOCKED_A;
END_REGION

REGION Network 49: UNIT 2 STATION 2 CALIBRATING METHOD CONNECTION ALARM
   RUNG wire#powerrail
      Contact( "DB16325_U2_STA2_MEAS_CALIBRATE_TRIG".Error )
      wire#w1
      Contact( "DB7255_UNIT_2_STA_2_MEAS_ENABLE_DISABLE".ENABLED )
      wire#w2
      I_Contact( "DB7300_INTERLOCK_GENERAL".GENERAL_MACHINE.FROM_CELL_TO_MACHINE_GENERAL.CELL_CALIBRATION_CYCLE_REQUIRED )
      Coil( "DB16000_OPC_UA_TRIGGER_ALARM".CLIENT.U2_STA2_MEAS.ALARMS.CALIBRATE_CONNECTION_A )
   END_RUNG
   RUNG wire#powerrail
      Contact( "DB16000_OPC_UA_TRIGGER_ALARM".CLIENT.U2_STA2_MEAS.ALARMS.CALIBRATE_CONNECTION_A )
      I_Contact( "DB2120_MPP_ITC_IPC".RESET_FAULTS )
   END_RUNG wire#w1
   RUNG wire#w2
      Coil( "DB426_ALARMS_WARNINGS".ALARMS.UNIT_02.STATION_2_MEASURING."720538" )
   END_RUNG
   // the same network as SCL:
   #_w1 := ("DB16325_U2_STA2_MEAS_CALIBRATE_TRIG".Error OR ("DB16000_OPC_UA_TRIGGER_ALARM".CLIENT.U2_STA2_MEAS.ALARMS.CALIBRATE_CONNECTION_A AND NOT "DB2120_MPP_ITC_IPC".RESET_FAULTS)) AND "DB7255_UNIT_2_STA_2_MEAS_ENABLE_DISABLE".ENABLED;
   "DB16000_OPC_UA_TRIGGER_ALARM".CLIENT.U2_STA2_MEAS.ALARMS.CALIBRATE_CONNECTION_A := #_w1 AND NOT "DB7300_INTERLOCK_GENERAL".GENERAL_MACHINE.FROM_CELL_TO_MACHINE_GENERAL.CELL_CALIBRATION_CYCLE_REQUIRED;
   "DB426_ALARMS_WARNINGS".ALARMS.UNIT_02.STATION_2_MEASURING."720538" := #_w1;
END_REGION

REGION Network 50: UNIT 2 STATION 2 CALIBRATING METHOD WORKING OR BLOCKED ALARM
   RUNG wire#powerrail
      Contact( "DB16325_U2_STA2_MEAS_CALIBRATE_TRIG".Done )
      I_Contact( "DB16003_U2_STA2_MEAS_CLIENT_INTERFACE".U02_STA2_MEAS_Method."Trigger calibration".Outputs.Result )
      wire#w1
      Contact( "DB7255_UNIT_2_STA_2_MEAS_ENABLE_DISABLE".ENABLED )
      wire#w2
      I_Contact( "DB7300_INTERLOCK_GENERAL".GENERAL_MACHINE.FROM_CELL_TO_MACHINE_GENERAL.CELL_CALIBRATION_CYCLE_REQUIRED )
      Coil( "DB16000_OPC_UA_TRIGGER_ALARM".CLIENT.U2_STA2_MEAS.ALARMS.CALIBRATE_METHOD_WORKING_BLOCKED_A )
   END_RUNG
   RUNG wire#powerrail
      Contact( "DB16000_OPC_UA_TRIGGER_ALARM".CLIENT.U2_STA2_MEAS.ALARMS.CALIBRATE_METHOD_WORKING_BLOCKED_A )
      I_Contact( "DB2120_MPP_ITC_IPC".RESET_FAULTS )
   END_RUNG wire#w1
   RUNG wire#w2
      Coil( "DB426_ALARMS_WARNINGS".ALARMS.UNIT_02.STATION_2_MEASURING."720539" )
   END_RUNG
   // the same network as SCL:
   #_w1 := (("DB16325_U2_STA2_MEAS_CALIBRATE_TRIG".Done AND NOT "DB16003_U2_STA2_MEAS_CLIENT_INTERFACE".U02_STA2_MEAS_Method."Trigger calibration".Outputs.Result) OR ("DB16000_OPC_UA_TRIGGER_ALARM".CLIENT.U2_STA2_MEAS.ALARMS.CALIBRATE_METHOD_WORKING_BLOCKED_A AND NOT "DB2120_MPP_ITC_IPC".RESET_FAULTS)) AND "DB7255_UNIT_2_STA_2_MEAS_ENABLE_DISABLE".ENABLED;
   "DB16000_OPC_UA_TRIGGER_ALARM".CLIENT.U2_STA2_MEAS.ALARMS.CALIBRATE_METHOD_WORKING_BLOCKED_A := #_w1 AND NOT "DB7300_INTERLOCK_GENERAL".GENERAL_MACHINE.FROM_CELL_TO_MACHINE_GENERAL.CELL_CALIBRATION_CYCLE_REQUIRED;
   "DB426_ALARMS_WARNINGS".ALARMS.UNIT_02.STATION_2_MEASURING."720539" := #_w1;
END_REGION

REGION Network 51: UNIT 2 STATION 2 RESET METHOD CONNECTION ALARM
   RUNG wire#powerrail
      Contact( "DB16327_U2_STA2_MEAS_RESET_TRIG".Error )
      wire#w1
      Contact( "DB7255_UNIT_2_STA_2_MEAS_ENABLE_DISABLE".ENABLED )
      wire#w2
      Coil( "DB16000_OPC_UA_TRIGGER_ALARM".CLIENT.U2_STA2_MEAS.ALARMS.RESET_CONNECTION_A )
   END_RUNG
   RUNG wire#powerrail
      Contact( "DB16000_OPC_UA_TRIGGER_ALARM".CLIENT.U2_STA2_MEAS.ALARMS.RESET_CONNECTION_A )
      I_Contact( "DB2120_MPP_ITC_IPC".RESET_FAULTS )
   END_RUNG wire#w1
   RUNG wire#w2
      Coil( "DB426_ALARMS_WARNINGS".ALARMS.UNIT_02.STATION_2_MEASURING."720546" )
   END_RUNG
   // the same network as SCL:
   "DB16000_OPC_UA_TRIGGER_ALARM".CLIENT.U2_STA2_MEAS.ALARMS.RESET_CONNECTION_A := ("DB16327_U2_STA2_MEAS_RESET_TRIG".Error OR ("DB16000_OPC_UA_TRIGGER_ALARM".CLIENT.U2_STA2_MEAS.ALARMS.RESET_CONNECTION_A AND NOT "DB2120_MPP_ITC_IPC".RESET_FAULTS)) AND "DB7255_UNIT_2_STA_2_MEAS_ENABLE_DISABLE".ENABLED;
   "DB426_ALARMS_WARNINGS".ALARMS.UNIT_02.STATION_2_MEASURING."720546" := "DB16000_OPC_UA_TRIGGER_ALARM".CLIENT.U2_STA2_MEAS.ALARMS.RESET_CONNECTION_A;
END_REGION

REGION Network 52: UNIT 2 STATION 2 RESET METHOD WORKING OR BLOCKED ALARM
   RUNG wire#powerrail
      Contact( "DB16327_U2_STA2_MEAS_RESET_TRIG".Done )
      I_Contact( "DB16003_U2_STA2_MEAS_CLIENT_INTERFACE".U02_STA2_MEAS_Method."Trigger reset".Outputs.Result )
      wire#w1
      Contact( "DB7255_UNIT_2_STA_2_MEAS_ENABLE_DISABLE".ENABLED )
      wire#w2
      Coil( "DB16000_OPC_UA_TRIGGER_ALARM".CLIENT.U2_STA2_MEAS.ALARMS.RESET_METHOD_WORKING_BLOCKED_A )
   END_RUNG
   RUNG wire#powerrail
      Contact( "DB16000_OPC_UA_TRIGGER_ALARM".CLIENT.U2_STA2_MEAS.ALARMS.RESET_METHOD_WORKING_BLOCKED_A )
      I_Contact( "DB2120_MPP_ITC_IPC".RESET_FAULTS )
   END_RUNG wire#w1
   RUNG wire#w2
      Coil( "DB426_ALARMS_WARNINGS".ALARMS.UNIT_02.STATION_2_MEASURING."720547" )
   END_RUNG
   // the same network as SCL:
   "DB16000_OPC_UA_TRIGGER_ALARM".CLIENT.U2_STA2_MEAS.ALARMS.RESET_METHOD_WORKING_BLOCKED_A := (("DB16327_U2_STA2_MEAS_RESET_TRIG".Done AND NOT "DB16003_U2_STA2_MEAS_CLIENT_INTERFACE".U02_STA2_MEAS_Method."Trigger reset".Outputs.Result) OR ("DB16000_OPC_UA_TRIGGER_ALARM".CLIENT.U2_STA2_MEAS.ALARMS.RESET_METHOD_WORKING_BLOCKED_A AND NOT "DB2120_MPP_ITC_IPC".RESET_FAULTS)) AND "DB7255_UNIT_2_STA_2_MEAS_ENABLE_DISABLE".ENABLED;
   "DB426_ALARMS_WARNINGS".ALARMS.UNIT_02.STATION_2_MEASURING."720547" := "DB16000_OPC_UA_TRIGGER_ALARM".CLIENT.U2_STA2_MEAS.ALARMS.RESET_METHOD_WORKING_BLOCKED_A;
END_REGION

REGION Network 53: UNIT 2 STATION 2 READ VARIABLES CONNECTION ALARM
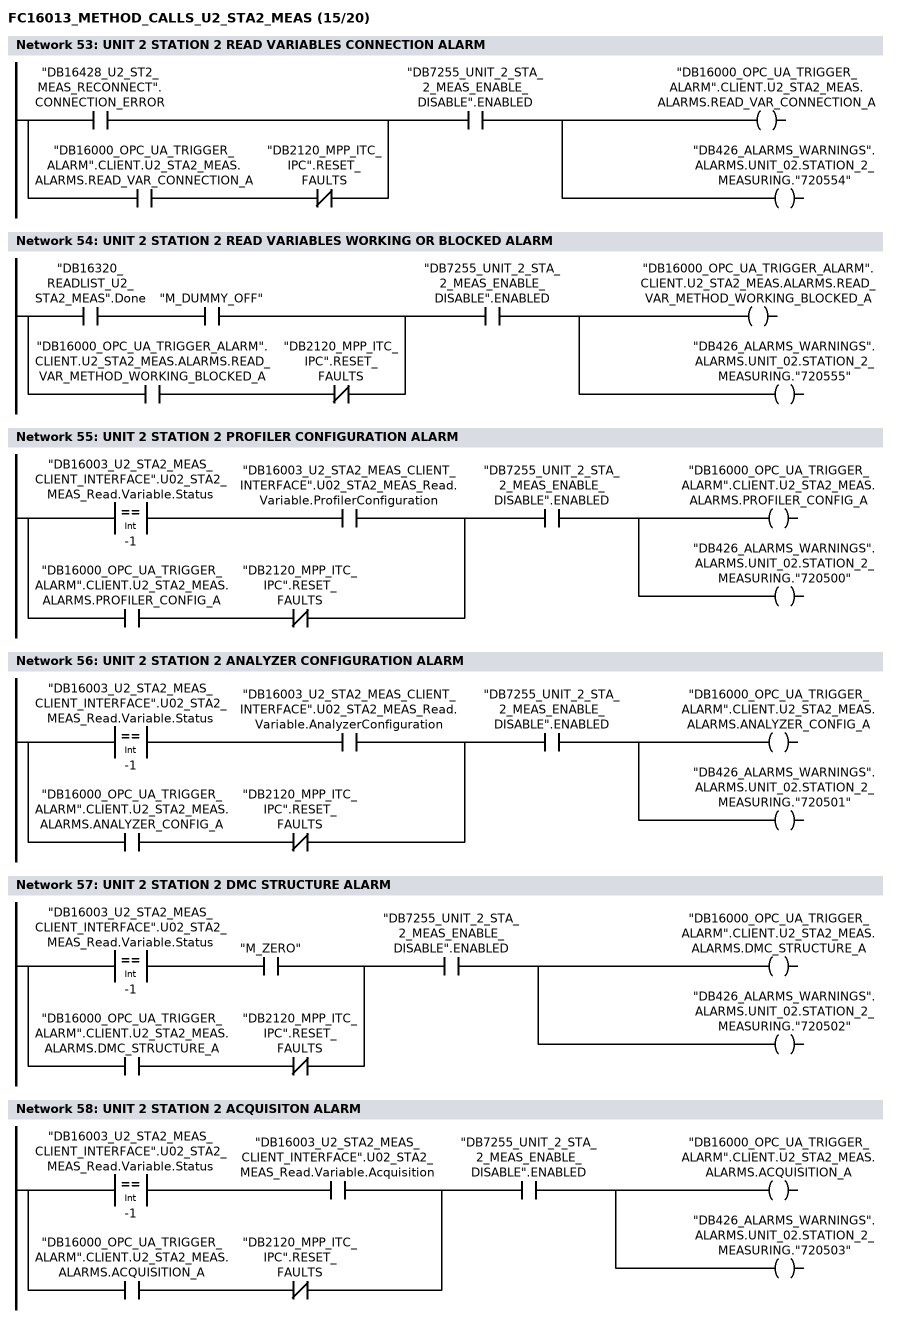
   RUNG wire#powerrail
      Contact( "DB16428_U2_ST2_MEAS_RECONNECT".CONNECTION_ERROR )
      wire#w1
      Contact( "DB7255_UNIT_2_STA_2_MEAS_ENABLE_DISABLE".ENABLED )
      wire#w2
      Coil( "DB16000_OPC_UA_TRIGGER_ALARM".CLIENT.U2_STA2_MEAS.ALARMS.READ_VAR_CONNECTION_A )
   END_RUNG
   RUNG wire#powerrail
      Contact( "DB16000_OPC_UA_TRIGGER_ALARM".CLIENT.U2_STA2_MEAS.ALARMS.READ_VAR_CONNECTION_A )
      I_Contact( "DB2120_MPP_ITC_IPC".RESET_FAULTS )
   END_RUNG wire#w1
   RUNG wire#w2
      Coil( "DB426_ALARMS_WARNINGS".ALARMS.UNIT_02.STATION_2_MEASURING."720554" )
   END_RUNG
   // the same network as SCL:
   "DB16000_OPC_UA_TRIGGER_ALARM".CLIENT.U2_STA2_MEAS.ALARMS.READ_VAR_CONNECTION_A := ("DB16428_U2_ST2_MEAS_RECONNECT".CONNECTION_ERROR OR ("DB16000_OPC_UA_TRIGGER_ALARM".CLIENT.U2_STA2_MEAS.ALARMS.READ_VAR_CONNECTION_A AND NOT "DB2120_MPP_ITC_IPC".RESET_FAULTS)) AND "DB7255_UNIT_2_STA_2_MEAS_ENABLE_DISABLE".ENABLED;
   "DB426_ALARMS_WARNINGS".ALARMS.UNIT_02.STATION_2_MEASURING."720554" := "DB16000_OPC_UA_TRIGGER_ALARM".CLIENT.U2_STA2_MEAS.ALARMS.READ_VAR_CONNECTION_A;
END_REGION

REGION Network 54: UNIT 2 STATION 2 READ VARIABLES WORKING OR BLOCKED ALARM
   RUNG wire#powerrail
      Contact( "DB16320_READLIST_U2_STA2_MEAS".Done )
      Contact( "M_DUMMY_OFF" )
      wire#w1
      Contact( "DB7255_UNIT_2_STA_2_MEAS_ENABLE_DISABLE".ENABLED )
      wire#w2
      Coil( "DB16000_OPC_UA_TRIGGER_ALARM".CLIENT.U2_STA2_MEAS.ALARMS.READ_VAR_METHOD_WORKING_BLOCKED_A )
   END_RUNG
   RUNG wire#powerrail
      Contact( "DB16000_OPC_UA_TRIGGER_ALARM".CLIENT.U2_STA2_MEAS.ALARMS.READ_VAR_METHOD_WORKING_BLOCKED_A )
      I_Contact( "DB2120_MPP_ITC_IPC".RESET_FAULTS )
   END_RUNG wire#w1
   RUNG wire#w2
      Coil( "DB426_ALARMS_WARNINGS".ALARMS.UNIT_02.STATION_2_MEASURING."720555" )
   END_RUNG
   // the same network as SCL:
   "DB16000_OPC_UA_TRIGGER_ALARM".CLIENT.U2_STA2_MEAS.ALARMS.READ_VAR_METHOD_WORKING_BLOCKED_A := (("DB16320_READLIST_U2_STA2_MEAS".Done AND "M_DUMMY_OFF") OR ("DB16000_OPC_UA_TRIGGER_ALARM".CLIENT.U2_STA2_MEAS.ALARMS.READ_VAR_METHOD_WORKING_BLOCKED_A AND NOT "DB2120_MPP_ITC_IPC".RESET_FAULTS)) AND "DB7255_UNIT_2_STA_2_MEAS_ENABLE_DISABLE".ENABLED;
   "DB426_ALARMS_WARNINGS".ALARMS.UNIT_02.STATION_2_MEASURING."720555" := "DB16000_OPC_UA_TRIGGER_ALARM".CLIENT.U2_STA2_MEAS.ALARMS.READ_VAR_METHOD_WORKING_BLOCKED_A;
END_REGION

REGION Network 55: UNIT 2 STATION 2 PROFILER CONFIGURATION ALARM
   RUNG wire#powerrail
      { S7_Templates := "SrcType := Int" } EQ_Contact(in1 := "DB16003_U2_STA2_MEAS_CLIENT_INTERFACE".U02_STA2_MEAS_Read.Variable.Status, in2 := -1)
      Contact( "DB16003_U2_STA2_MEAS_CLIENT_INTERFACE".U02_STA2_MEAS_Read.Variable.ProfilerConfiguration )
      wire#w1
      Contact( "DB7255_UNIT_2_STA_2_MEAS_ENABLE_DISABLE".ENABLED )
      wire#w2
      Coil( "DB16000_OPC_UA_TRIGGER_ALARM".CLIENT.U2_STA2_MEAS.ALARMS.PROFILER_CONFIG_A )
   END_RUNG
   RUNG wire#powerrail
      Contact( "DB16000_OPC_UA_TRIGGER_ALARM".CLIENT.U2_STA2_MEAS.ALARMS.PROFILER_CONFIG_A )
      I_Contact( "DB2120_MPP_ITC_IPC".RESET_FAULTS )
   END_RUNG wire#w1
   RUNG wire#w2
      Coil( "DB426_ALARMS_WARNINGS".ALARMS.UNIT_02.STATION_2_MEASURING."720500" )
   END_RUNG
   // the same network as SCL:
   "DB16000_OPC_UA_TRIGGER_ALARM".CLIENT.U2_STA2_MEAS.ALARMS.PROFILER_CONFIG_A := ((("DB16003_U2_STA2_MEAS_CLIENT_INTERFACE".U02_STA2_MEAS_Read.Variable.Status = (-1)) AND "DB16003_U2_STA2_MEAS_CLIENT_INTERFACE".U02_STA2_MEAS_Read.Variable.ProfilerConfiguration) OR ("DB16000_OPC_UA_TRIGGER_ALARM".CLIENT.U2_STA2_MEAS.ALARMS.PROFILER_CONFIG_A AND NOT "DB2120_MPP_ITC_IPC".RESET_FAULTS)) AND "DB7255_UNIT_2_STA_2_MEAS_ENABLE_DISABLE".ENABLED;
   "DB426_ALARMS_WARNINGS".ALARMS.UNIT_02.STATION_2_MEASURING."720500" := "DB16000_OPC_UA_TRIGGER_ALARM".CLIENT.U2_STA2_MEAS.ALARMS.PROFILER_CONFIG_A;
END_REGION

REGION Network 56: UNIT 2 STATION 2 ANALYZER CONFIGURATION ALARM
   RUNG wire#powerrail
      { S7_Templates := "SrcType := Int" } EQ_Contact(in1 := "DB16003_U2_STA2_MEAS_CLIENT_INTERFACE".U02_STA2_MEAS_Read.Variable.Status, in2 := -1)
      Contact( "DB16003_U2_STA2_MEAS_CLIENT_INTERFACE".U02_STA2_MEAS_Read.Variable.AnalyzerConfiguration )
      wire#w1
      Contact( "DB7255_UNIT_2_STA_2_MEAS_ENABLE_DISABLE".ENABLED )
      wire#w2
      Coil( "DB16000_OPC_UA_TRIGGER_ALARM".CLIENT.U2_STA2_MEAS.ALARMS.ANALYZER_CONFIG_A )
   END_RUNG
   RUNG wire#powerrail
      Contact( "DB16000_OPC_UA_TRIGGER_ALARM".CLIENT.U2_STA2_MEAS.ALARMS.ANALYZER_CONFIG_A )
      I_Contact( "DB2120_MPP_ITC_IPC".RESET_FAULTS )
   END_RUNG wire#w1
   RUNG wire#w2
      Coil( "DB426_ALARMS_WARNINGS".ALARMS.UNIT_02.STATION_2_MEASURING."720501" )
   END_RUNG
   // the same network as SCL:
   "DB16000_OPC_UA_TRIGGER_ALARM".CLIENT.U2_STA2_MEAS.ALARMS.ANALYZER_CONFIG_A := ((("DB16003_U2_STA2_MEAS_CLIENT_INTERFACE".U02_STA2_MEAS_Read.Variable.Status = (-1)) AND "DB16003_U2_STA2_MEAS_CLIENT_INTERFACE".U02_STA2_MEAS_Read.Variable.AnalyzerConfiguration) OR ("DB16000_OPC_UA_TRIGGER_ALARM".CLIENT.U2_STA2_MEAS.ALARMS.ANALYZER_CONFIG_A AND NOT "DB2120_MPP_ITC_IPC".RESET_FAULTS)) AND "DB7255_UNIT_2_STA_2_MEAS_ENABLE_DISABLE".ENABLED;
   "DB426_ALARMS_WARNINGS".ALARMS.UNIT_02.STATION_2_MEASURING."720501" := "DB16000_OPC_UA_TRIGGER_ALARM".CLIENT.U2_STA2_MEAS.ALARMS.ANALYZER_CONFIG_A;
END_REGION

REGION Network 57: UNIT 2 STATION 2 DMC STRUCTURE ALARM
   RUNG wire#powerrail
      { S7_Templates := "SrcType := Int" } EQ_Contact(in1 := "DB16003_U2_STA2_MEAS_CLIENT_INTERFACE".U02_STA2_MEAS_Read.Variable.Status, in2 := -1)
      Contact( "M_ZERO" )
      wire#w1
      Contact( "DB7255_UNIT_2_STA_2_MEAS_ENABLE_DISABLE".ENABLED )
      wire#w2
      Coil( "DB16000_OPC_UA_TRIGGER_ALARM".CLIENT.U2_STA2_MEAS.ALARMS.DMC_STRUCTURE_A )
   END_RUNG
   RUNG wire#powerrail
      Contact( "DB16000_OPC_UA_TRIGGER_ALARM".CLIENT.U2_STA2_MEAS.ALARMS.DMC_STRUCTURE_A )
      I_Contact( "DB2120_MPP_ITC_IPC".RESET_FAULTS )
   END_RUNG wire#w1
   RUNG wire#w2
      Coil( "DB426_ALARMS_WARNINGS".ALARMS.UNIT_02.STATION_2_MEASURING."720502" )
   END_RUNG
   // the same network as SCL:
   "DB16000_OPC_UA_TRIGGER_ALARM".CLIENT.U2_STA2_MEAS.ALARMS.DMC_STRUCTURE_A := ((("DB16003_U2_STA2_MEAS_CLIENT_INTERFACE".U02_STA2_MEAS_Read.Variable.Status = (-1)) AND "M_ZERO") OR ("DB16000_OPC_UA_TRIGGER_ALARM".CLIENT.U2_STA2_MEAS.ALARMS.DMC_STRUCTURE_A AND NOT "DB2120_MPP_ITC_IPC".RESET_FAULTS)) AND "DB7255_UNIT_2_STA_2_MEAS_ENABLE_DISABLE".ENABLED;
   "DB426_ALARMS_WARNINGS".ALARMS.UNIT_02.STATION_2_MEASURING."720502" := "DB16000_OPC_UA_TRIGGER_ALARM".CLIENT.U2_STA2_MEAS.ALARMS.DMC_STRUCTURE_A;
END_REGION

REGION Network 58: UNIT 2 STATION 2 ACQUISITON ALARM
   RUNG wire#powerrail
      { S7_Templates := "SrcType := Int" } EQ_Contact(in1 := "DB16003_U2_STA2_MEAS_CLIENT_INTERFACE".U02_STA2_MEAS_Read.Variable.Status, in2 := -1)
      Contact( "DB16003_U2_STA2_MEAS_CLIENT_INTERFACE".U02_STA2_MEAS_Read.Variable.Acquisition )
      wire#w1
      Contact( "DB7255_UNIT_2_STA_2_MEAS_ENABLE_DISABLE".ENABLED )
      wire#w2
      Coil( "DB16000_OPC_UA_TRIGGER_ALARM".CLIENT.U2_STA2_MEAS.ALARMS.ACQUISITION_A )
   END_RUNG
   RUNG wire#powerrail
      Contact( "DB16000_OPC_UA_TRIGGER_ALARM".CLIENT.U2_STA2_MEAS.ALARMS.ACQUISITION_A )
      I_Contact( "DB2120_MPP_ITC_IPC".RESET_FAULTS )
   END_RUNG wire#w1
   RUNG wire#w2
      Coil( "DB426_ALARMS_WARNINGS".ALARMS.UNIT_02.STATION_2_MEASURING."720503" )
   END_RUNG
   // the same network as SCL:
   "DB16000_OPC_UA_TRIGGER_ALARM".CLIENT.U2_STA2_MEAS.ALARMS.ACQUISITION_A := ((("DB16003_U2_STA2_MEAS_CLIENT_INTERFACE".U02_STA2_MEAS_Read.Variable.Status = (-1)) AND "DB16003_U2_STA2_MEAS_CLIENT_INTERFACE".U02_STA2_MEAS_Read.Variable.Acquisition) OR ("DB16000_OPC_UA_TRIGGER_ALARM".CLIENT.U2_STA2_MEAS.ALARMS.ACQUISITION_A AND NOT "DB2120_MPP_ITC_IPC".RESET_FAULTS)) AND "DB7255_UNIT_2_STA_2_MEAS_ENABLE_DISABLE".ENABLED;
   "DB426_ALARMS_WARNINGS".ALARMS.UNIT_02.STATION_2_MEASURING."720503" := "DB16000_OPC_UA_TRIGGER_ALARM".CLIENT.U2_STA2_MEAS.ALARMS.ACQUISITION_A;
END_REGION

REGION Network 59: UNIT 2 STATION 2 PROFILER INITIALIZTION ALARM
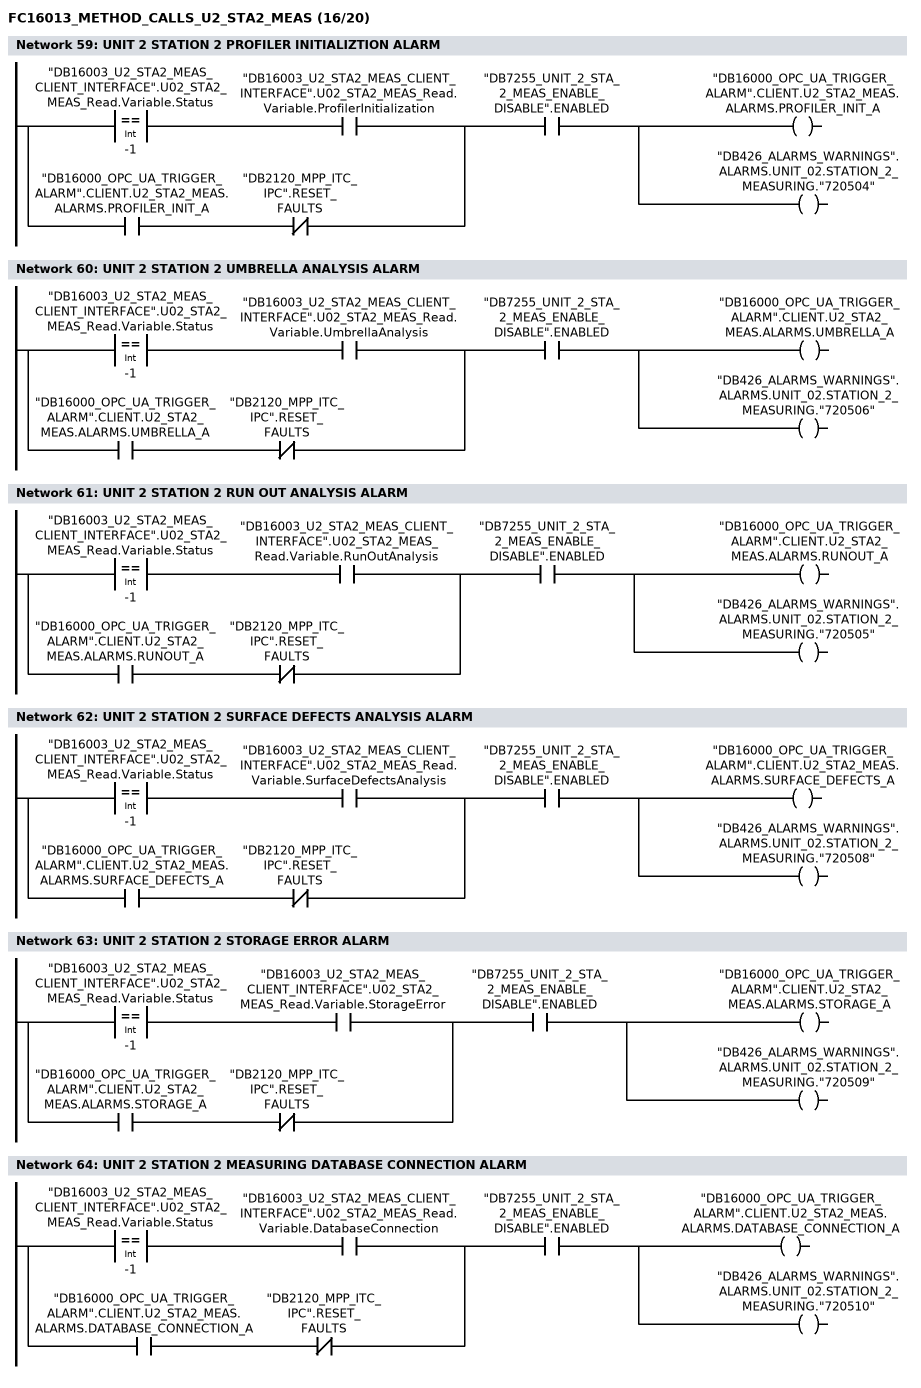
   RUNG wire#powerrail
      { S7_Templates := "SrcType := Int" } EQ_Contact(in1 := "DB16003_U2_STA2_MEAS_CLIENT_INTERFACE".U02_STA2_MEAS_Read.Variable.Status, in2 := -1)
      Contact( "DB16003_U2_STA2_MEAS_CLIENT_INTERFACE".U02_STA2_MEAS_Read.Variable.ProfilerInitialization )
      wire#w1
      Contact( "DB7255_UNIT_2_STA_2_MEAS_ENABLE_DISABLE".ENABLED )
      wire#w2
      Coil( "DB16000_OPC_UA_TRIGGER_ALARM".CLIENT.U2_STA2_MEAS.ALARMS.PROFILER_INIT_A )
   END_RUNG
   RUNG wire#powerrail
      Contact( "DB16000_OPC_UA_TRIGGER_ALARM".CLIENT.U2_STA2_MEAS.ALARMS.PROFILER_INIT_A )
      I_Contact( "DB2120_MPP_ITC_IPC".RESET_FAULTS )
   END_RUNG wire#w1
   RUNG wire#w2
      Coil( "DB426_ALARMS_WARNINGS".ALARMS.UNIT_02.STATION_2_MEASURING."720504" )
   END_RUNG
   // the same network as SCL:
   "DB16000_OPC_UA_TRIGGER_ALARM".CLIENT.U2_STA2_MEAS.ALARMS.PROFILER_INIT_A := ((("DB16003_U2_STA2_MEAS_CLIENT_INTERFACE".U02_STA2_MEAS_Read.Variable.Status = (-1)) AND "DB16003_U2_STA2_MEAS_CLIENT_INTERFACE".U02_STA2_MEAS_Read.Variable.ProfilerInitialization) OR ("DB16000_OPC_UA_TRIGGER_ALARM".CLIENT.U2_STA2_MEAS.ALARMS.PROFILER_INIT_A AND NOT "DB2120_MPP_ITC_IPC".RESET_FAULTS)) AND "DB7255_UNIT_2_STA_2_MEAS_ENABLE_DISABLE".ENABLED;
   "DB426_ALARMS_WARNINGS".ALARMS.UNIT_02.STATION_2_MEASURING."720504" := "DB16000_OPC_UA_TRIGGER_ALARM".CLIENT.U2_STA2_MEAS.ALARMS.PROFILER_INIT_A;
END_REGION

REGION Network 60: UNIT 2 STATION 2 UMBRELLA ANALYSIS ALARM
   RUNG wire#powerrail
      { S7_Templates := "SrcType := Int" } EQ_Contact(in1 := "DB16003_U2_STA2_MEAS_CLIENT_INTERFACE".U02_STA2_MEAS_Read.Variable.Status, in2 := -1)
      Contact( "DB16003_U2_STA2_MEAS_CLIENT_INTERFACE".U02_STA2_MEAS_Read.Variable.UmbrellaAnalysis )
      wire#w1
      Contact( "DB7255_UNIT_2_STA_2_MEAS_ENABLE_DISABLE".ENABLED )
      wire#w2
      Coil( "DB16000_OPC_UA_TRIGGER_ALARM".CLIENT.U2_STA2_MEAS.ALARMS.UMBRELLA_A )
   END_RUNG
   RUNG wire#powerrail
      Contact( "DB16000_OPC_UA_TRIGGER_ALARM".CLIENT.U2_STA2_MEAS.ALARMS.UMBRELLA_A )
      I_Contact( "DB2120_MPP_ITC_IPC".RESET_FAULTS )
   END_RUNG wire#w1
   RUNG wire#w2
      Coil( "DB426_ALARMS_WARNINGS".ALARMS.UNIT_02.STATION_2_MEASURING."720506" )
   END_RUNG
   // the same network as SCL:
   "DB16000_OPC_UA_TRIGGER_ALARM".CLIENT.U2_STA2_MEAS.ALARMS.UMBRELLA_A := ((("DB16003_U2_STA2_MEAS_CLIENT_INTERFACE".U02_STA2_MEAS_Read.Variable.Status = (-1)) AND "DB16003_U2_STA2_MEAS_CLIENT_INTERFACE".U02_STA2_MEAS_Read.Variable.UmbrellaAnalysis) OR ("DB16000_OPC_UA_TRIGGER_ALARM".CLIENT.U2_STA2_MEAS.ALARMS.UMBRELLA_A AND NOT "DB2120_MPP_ITC_IPC".RESET_FAULTS)) AND "DB7255_UNIT_2_STA_2_MEAS_ENABLE_DISABLE".ENABLED;
   "DB426_ALARMS_WARNINGS".ALARMS.UNIT_02.STATION_2_MEASURING."720506" := "DB16000_OPC_UA_TRIGGER_ALARM".CLIENT.U2_STA2_MEAS.ALARMS.UMBRELLA_A;
END_REGION

REGION Network 61: UNIT 2 STATION 2 RUN OUT ANALYSIS ALARM
   RUNG wire#powerrail
      { S7_Templates := "SrcType := Int" } EQ_Contact(in1 := "DB16003_U2_STA2_MEAS_CLIENT_INTERFACE".U02_STA2_MEAS_Read.Variable.Status, in2 := -1)
      Contact( "DB16003_U2_STA2_MEAS_CLIENT_INTERFACE".U02_STA2_MEAS_Read.Variable.RunOutAnalysis )
      wire#w1
      Contact( "DB7255_UNIT_2_STA_2_MEAS_ENABLE_DISABLE".ENABLED )
      wire#w2
      Coil( "DB16000_OPC_UA_TRIGGER_ALARM".CLIENT.U2_STA2_MEAS.ALARMS.RUNOUT_A )
   END_RUNG
   RUNG wire#powerrail
      Contact( "DB16000_OPC_UA_TRIGGER_ALARM".CLIENT.U2_STA2_MEAS.ALARMS.RUNOUT_A )
      I_Contact( "DB2120_MPP_ITC_IPC".RESET_FAULTS )
   END_RUNG wire#w1
   RUNG wire#w2
      Coil( "DB426_ALARMS_WARNINGS".ALARMS.UNIT_02.STATION_2_MEASURING."720505" )
   END_RUNG
   // the same network as SCL:
   "DB16000_OPC_UA_TRIGGER_ALARM".CLIENT.U2_STA2_MEAS.ALARMS.RUNOUT_A := ((("DB16003_U2_STA2_MEAS_CLIENT_INTERFACE".U02_STA2_MEAS_Read.Variable.Status = (-1)) AND "DB16003_U2_STA2_MEAS_CLIENT_INTERFACE".U02_STA2_MEAS_Read.Variable.RunOutAnalysis) OR ("DB16000_OPC_UA_TRIGGER_ALARM".CLIENT.U2_STA2_MEAS.ALARMS.RUNOUT_A AND NOT "DB2120_MPP_ITC_IPC".RESET_FAULTS)) AND "DB7255_UNIT_2_STA_2_MEAS_ENABLE_DISABLE".ENABLED;
   "DB426_ALARMS_WARNINGS".ALARMS.UNIT_02.STATION_2_MEASURING."720505" := "DB16000_OPC_UA_TRIGGER_ALARM".CLIENT.U2_STA2_MEAS.ALARMS.RUNOUT_A;
END_REGION

REGION Network 62: UNIT 2 STATION 2 SURFACE DEFECTS ANALYSIS ALARM
   RUNG wire#powerrail
      { S7_Templates := "SrcType := Int" } EQ_Contact(in1 := "DB16003_U2_STA2_MEAS_CLIENT_INTERFACE".U02_STA2_MEAS_Read.Variable.Status, in2 := -1)
      Contact( "DB16003_U2_STA2_MEAS_CLIENT_INTERFACE".U02_STA2_MEAS_Read.Variable.SurfaceDefectsAnalysis )
      wire#w1
      Contact( "DB7255_UNIT_2_STA_2_MEAS_ENABLE_DISABLE".ENABLED )
      wire#w2
      Coil( "DB16000_OPC_UA_TRIGGER_ALARM".CLIENT.U2_STA2_MEAS.ALARMS.SURFACE_DEFECTS_A )
   END_RUNG
   RUNG wire#powerrail
      Contact( "DB16000_OPC_UA_TRIGGER_ALARM".CLIENT.U2_STA2_MEAS.ALARMS.SURFACE_DEFECTS_A )
      I_Contact( "DB2120_MPP_ITC_IPC".RESET_FAULTS )
   END_RUNG wire#w1
   RUNG wire#w2
      Coil( "DB426_ALARMS_WARNINGS".ALARMS.UNIT_02.STATION_2_MEASURING."720508" )
   END_RUNG
   // the same network as SCL:
   "DB16000_OPC_UA_TRIGGER_ALARM".CLIENT.U2_STA2_MEAS.ALARMS.SURFACE_DEFECTS_A := ((("DB16003_U2_STA2_MEAS_CLIENT_INTERFACE".U02_STA2_MEAS_Read.Variable.Status = (-1)) AND "DB16003_U2_STA2_MEAS_CLIENT_INTERFACE".U02_STA2_MEAS_Read.Variable.SurfaceDefectsAnalysis) OR ("DB16000_OPC_UA_TRIGGER_ALARM".CLIENT.U2_STA2_MEAS.ALARMS.SURFACE_DEFECTS_A AND NOT "DB2120_MPP_ITC_IPC".RESET_FAULTS)) AND "DB7255_UNIT_2_STA_2_MEAS_ENABLE_DISABLE".ENABLED;
   "DB426_ALARMS_WARNINGS".ALARMS.UNIT_02.STATION_2_MEASURING."720508" := "DB16000_OPC_UA_TRIGGER_ALARM".CLIENT.U2_STA2_MEAS.ALARMS.SURFACE_DEFECTS_A;
END_REGION

REGION Network 63: UNIT 2 STATION 2 STORAGE ERROR ALARM
   RUNG wire#powerrail
      { S7_Templates := "SrcType := Int" } EQ_Contact(in1 := "DB16003_U2_STA2_MEAS_CLIENT_INTERFACE".U02_STA2_MEAS_Read.Variable.Status, in2 := -1)
      Contact( "DB16003_U2_STA2_MEAS_CLIENT_INTERFACE".U02_STA2_MEAS_Read.Variable.StorageError )
      wire#w1
      Contact( "DB7255_UNIT_2_STA_2_MEAS_ENABLE_DISABLE".ENABLED )
      wire#w2
      Coil( "DB16000_OPC_UA_TRIGGER_ALARM".CLIENT.U2_STA2_MEAS.ALARMS.STORAGE_A )
   END_RUNG
   RUNG wire#powerrail
      Contact( "DB16000_OPC_UA_TRIGGER_ALARM".CLIENT.U2_STA2_MEAS.ALARMS.STORAGE_A )
      I_Contact( "DB2120_MPP_ITC_IPC".RESET_FAULTS )
   END_RUNG wire#w1
   RUNG wire#w2
      Coil( "DB426_ALARMS_WARNINGS".ALARMS.UNIT_02.STATION_2_MEASURING."720509" )
   END_RUNG
   // the same network as SCL:
   "DB16000_OPC_UA_TRIGGER_ALARM".CLIENT.U2_STA2_MEAS.ALARMS.STORAGE_A := ((("DB16003_U2_STA2_MEAS_CLIENT_INTERFACE".U02_STA2_MEAS_Read.Variable.Status = (-1)) AND "DB16003_U2_STA2_MEAS_CLIENT_INTERFACE".U02_STA2_MEAS_Read.Variable.StorageError) OR ("DB16000_OPC_UA_TRIGGER_ALARM".CLIENT.U2_STA2_MEAS.ALARMS.STORAGE_A AND NOT "DB2120_MPP_ITC_IPC".RESET_FAULTS)) AND "DB7255_UNIT_2_STA_2_MEAS_ENABLE_DISABLE".ENABLED;
   "DB426_ALARMS_WARNINGS".ALARMS.UNIT_02.STATION_2_MEASURING."720509" := "DB16000_OPC_UA_TRIGGER_ALARM".CLIENT.U2_STA2_MEAS.ALARMS.STORAGE_A;
END_REGION

REGION Network 64: UNIT 2 STATION 2 MEASURING DATABASE CONNECTION ALARM
   RUNG wire#powerrail
      { S7_Templates := "SrcType := Int" } EQ_Contact(in1 := "DB16003_U2_STA2_MEAS_CLIENT_INTERFACE".U02_STA2_MEAS_Read.Variable.Status, in2 := -1)
      Contact( "DB16003_U2_STA2_MEAS_CLIENT_INTERFACE".U02_STA2_MEAS_Read.Variable.DatabaseConnection )
      wire#w1
      Contact( "DB7255_UNIT_2_STA_2_MEAS_ENABLE_DISABLE".ENABLED )
      wire#w2
      Coil( "DB16000_OPC_UA_TRIGGER_ALARM".CLIENT.U2_STA2_MEAS.ALARMS.DATABASE_CONNECTION_A )
   END_RUNG
   RUNG wire#powerrail
      Contact( "DB16000_OPC_UA_TRIGGER_ALARM".CLIENT.U2_STA2_MEAS.ALARMS.DATABASE_CONNECTION_A )
      I_Contact( "DB2120_MPP_ITC_IPC".RESET_FAULTS )
   END_RUNG wire#w1
   RUNG wire#w2
      Coil( "DB426_ALARMS_WARNINGS".ALARMS.UNIT_02.STATION_2_MEASURING."720510" )
   END_RUNG
   // the same network as SCL:
   "DB16000_OPC_UA_TRIGGER_ALARM".CLIENT.U2_STA2_MEAS.ALARMS.DATABASE_CONNECTION_A := ((("DB16003_U2_STA2_MEAS_CLIENT_INTERFACE".U02_STA2_MEAS_Read.Variable.Status = (-1)) AND "DB16003_U2_STA2_MEAS_CLIENT_INTERFACE".U02_STA2_MEAS_Read.Variable.DatabaseConnection) OR ("DB16000_OPC_UA_TRIGGER_ALARM".CLIENT.U2_STA2_MEAS.ALARMS.DATABASE_CONNECTION_A AND NOT "DB2120_MPP_ITC_IPC".RESET_FAULTS)) AND "DB7255_UNIT_2_STA_2_MEAS_ENABLE_DISABLE".ENABLED;
   "DB426_ALARMS_WARNINGS".ALARMS.UNIT_02.STATION_2_MEASURING."720510" := "DB16000_OPC_UA_TRIGGER_ALARM".CLIENT.U2_STA2_MEAS.ALARMS.DATABASE_CONNECTION_A;
END_REGION

